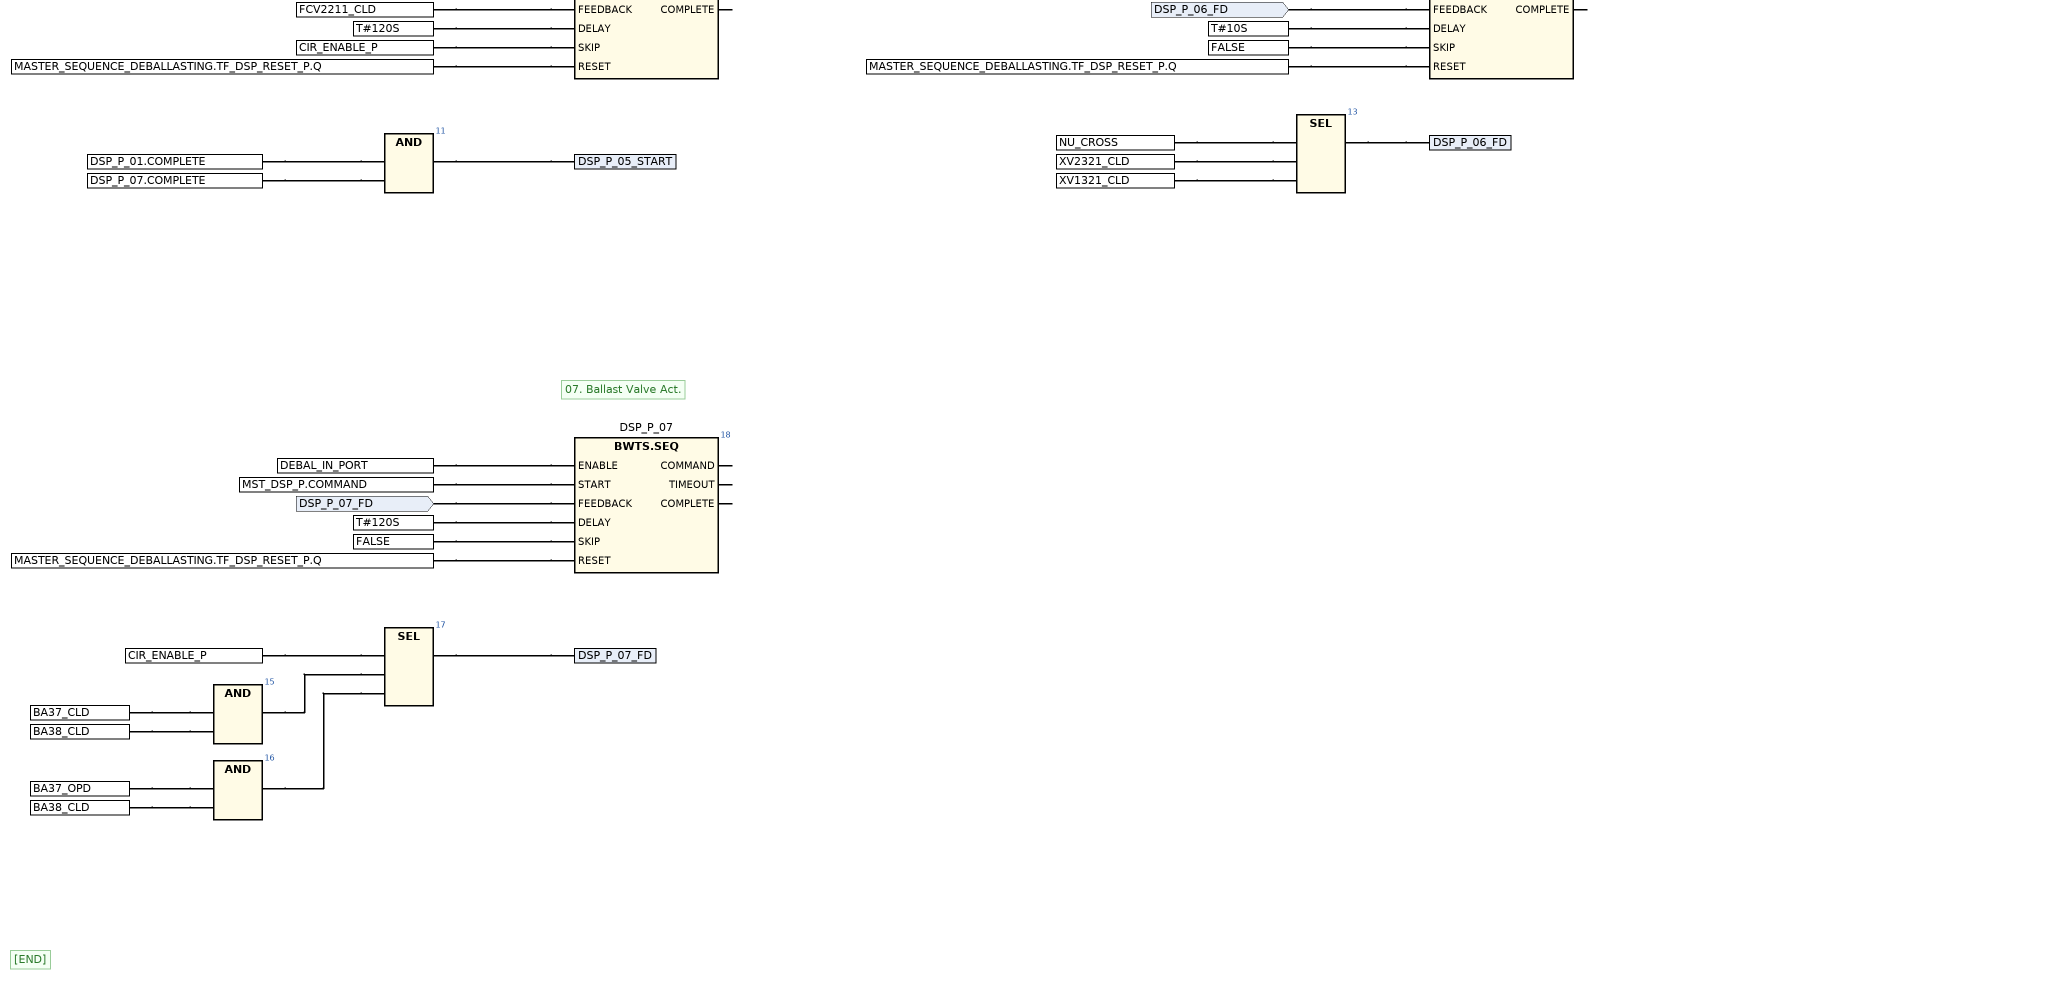
DST_S_ON := DEBAL_IN_STBD AND NOT MST_DSP_S.COMMAND;
(* DSP_P_01.COMPLETE AND DSP_P_07.COMPLETE; result not used *)
(* SEL(NU_CROSS, P232_SPD, P132_SPD); result not used *)
// 02. N/U Pump Stop
DSP_P_02(
    ENABLE := DEBAL_IN_PORT,
    START := _w1,
    FEEDBACK := _w2,
    DELAY := T#10S,
    SKIP := FALSE,
    RESET := MASTER_SEQUENCE_DEBALLASTING.TF_DSP_RESET_P.Q); // BWTS.SEQ
// WATING TIME FOR WBP
TON_0(IN := MST_DSP_P.COMMAND, PT := MS_WBP_SP); // TON
// 01. WBP Stop Request
DSP_P_01(
    ENABLE := DEBAL_IN_PORT,
    START := TON_0.Q,
    FEEDBACK := _w3,
    DELAY := T#120S,
    SKIP := CIR_ENABLE_P,
    RESET := MASTER_SEQUENCE_DEBALLASTING.TF_DSP_RESET_P.Q); // BWTS.SEQ
(* SEL(TRO_CROSS, AIT251_SPD AND XV2512_CLD, AIT151_SPD AND XV1512_CLD); result not used *)
// 03. TRO UNIT STOP
DSP_P_03(
    ENABLE := DEBAL_IN_PORT,
    START := MST_DSP_P.COMMAND,
    FEEDBACK := _w4,
    DELAY := T#10S,
    SKIP := _w4,
    RESET := MASTER_SEQUENCE_DEBALLASTING.TF_DSP_RESET_P.Q); // BWTS.SEQ
(* DSP_P_01.COMPLETE AND DSP_P_07.COMPLETE; result not used *)
// 05. TRC Valve Close
DSP_P_05(
    ENABLE := DEBAL_IN_PORT,
    START := _w5,
    FEEDBACK := FCV2211_CLD,
    DELAY := T#120S,
    SKIP := CIR_ENABLE_P,
    RESET := MASTER_SEQUENCE_DEBALLASTING.TF_DSP_RESET_P.Q); // BWTS.SEQ
(* SEL(NU_CROSS, XV2321_CLD, XV1321_CLD); result not used *)
// 06. N/U Inj. Valve Close
DSP_P_06(
    ENABLE := DEBAL_IN_PORT,
    START := DSP_P_02.COMPLETE,
    FEEDBACK := _w6,
    DELAY := T#10S,
    SKIP := FALSE,
    RESET := MASTER_SEQUENCE_DEBALLASTING.TF_DSP_RESET_P.Q); // BWTS.SEQ
// [END]
(* SEL(CIR_ENABLE_P, BA37_CLD AND BA38_CLD, BA37_OPD AND BA38_CLD); result not used *)
// 07. Ballast Valve Act.
DSP_P_07(
    ENABLE := DEBAL_IN_PORT,
    START := MST_DSP_P.COMMAND,
    FEEDBACK := _w7,
    DELAY := T#120S,
    SKIP := FALSE,
    RESET := MASTER_SEQUENCE_DEBALLASTING.TF_DSP_RESET_P.Q); // BWTS.SEQ

END_PROGRAM

// Device/Application/Logic/2.Sequence/SEQ_DEBAL_SP_S
PROGRAM SEQ_DEBAL_SP_S
VAR
	TON_0: TON;
	DST_P_ON: BOOL;
END_VAR
VAR // added by the converter: edge detectors and wires of the graphical bodies
    _w1, _w2, _w3, _w4, _w5, _w6, _w7 : ANY;
END_VAR

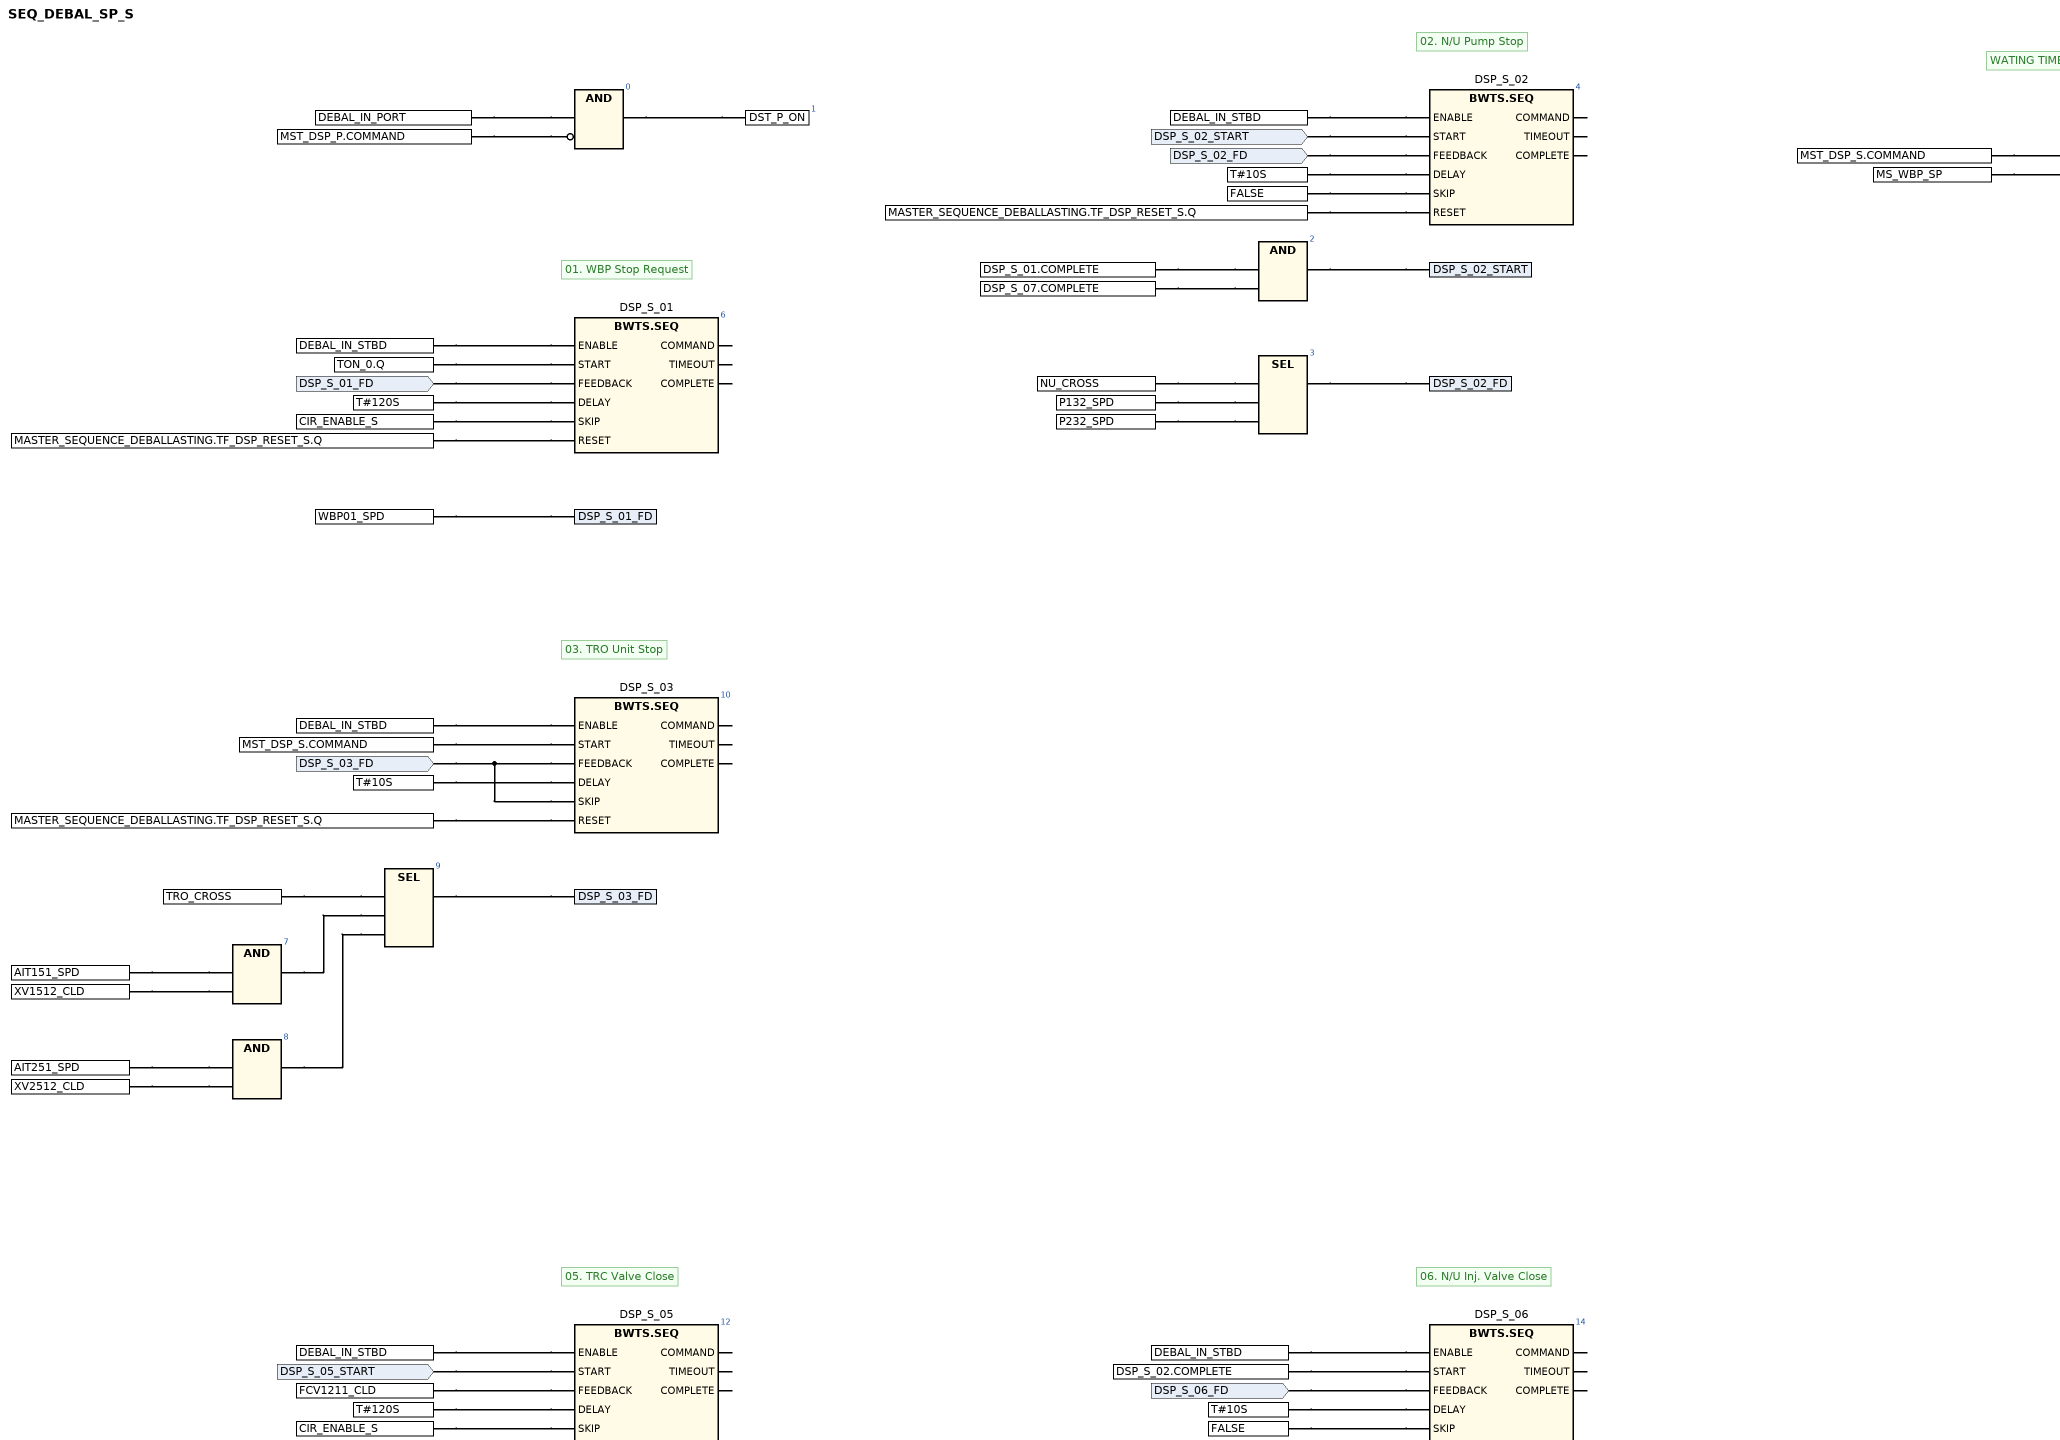
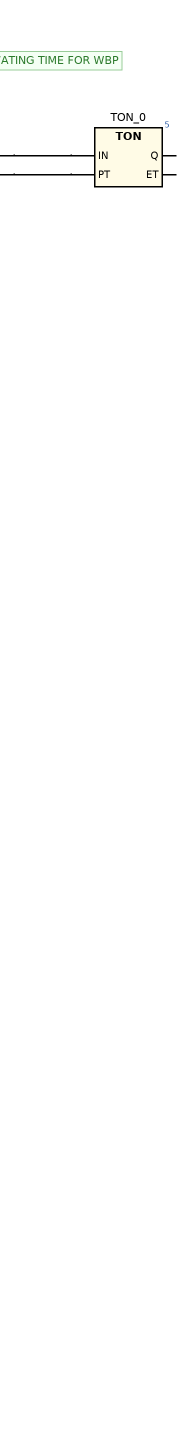
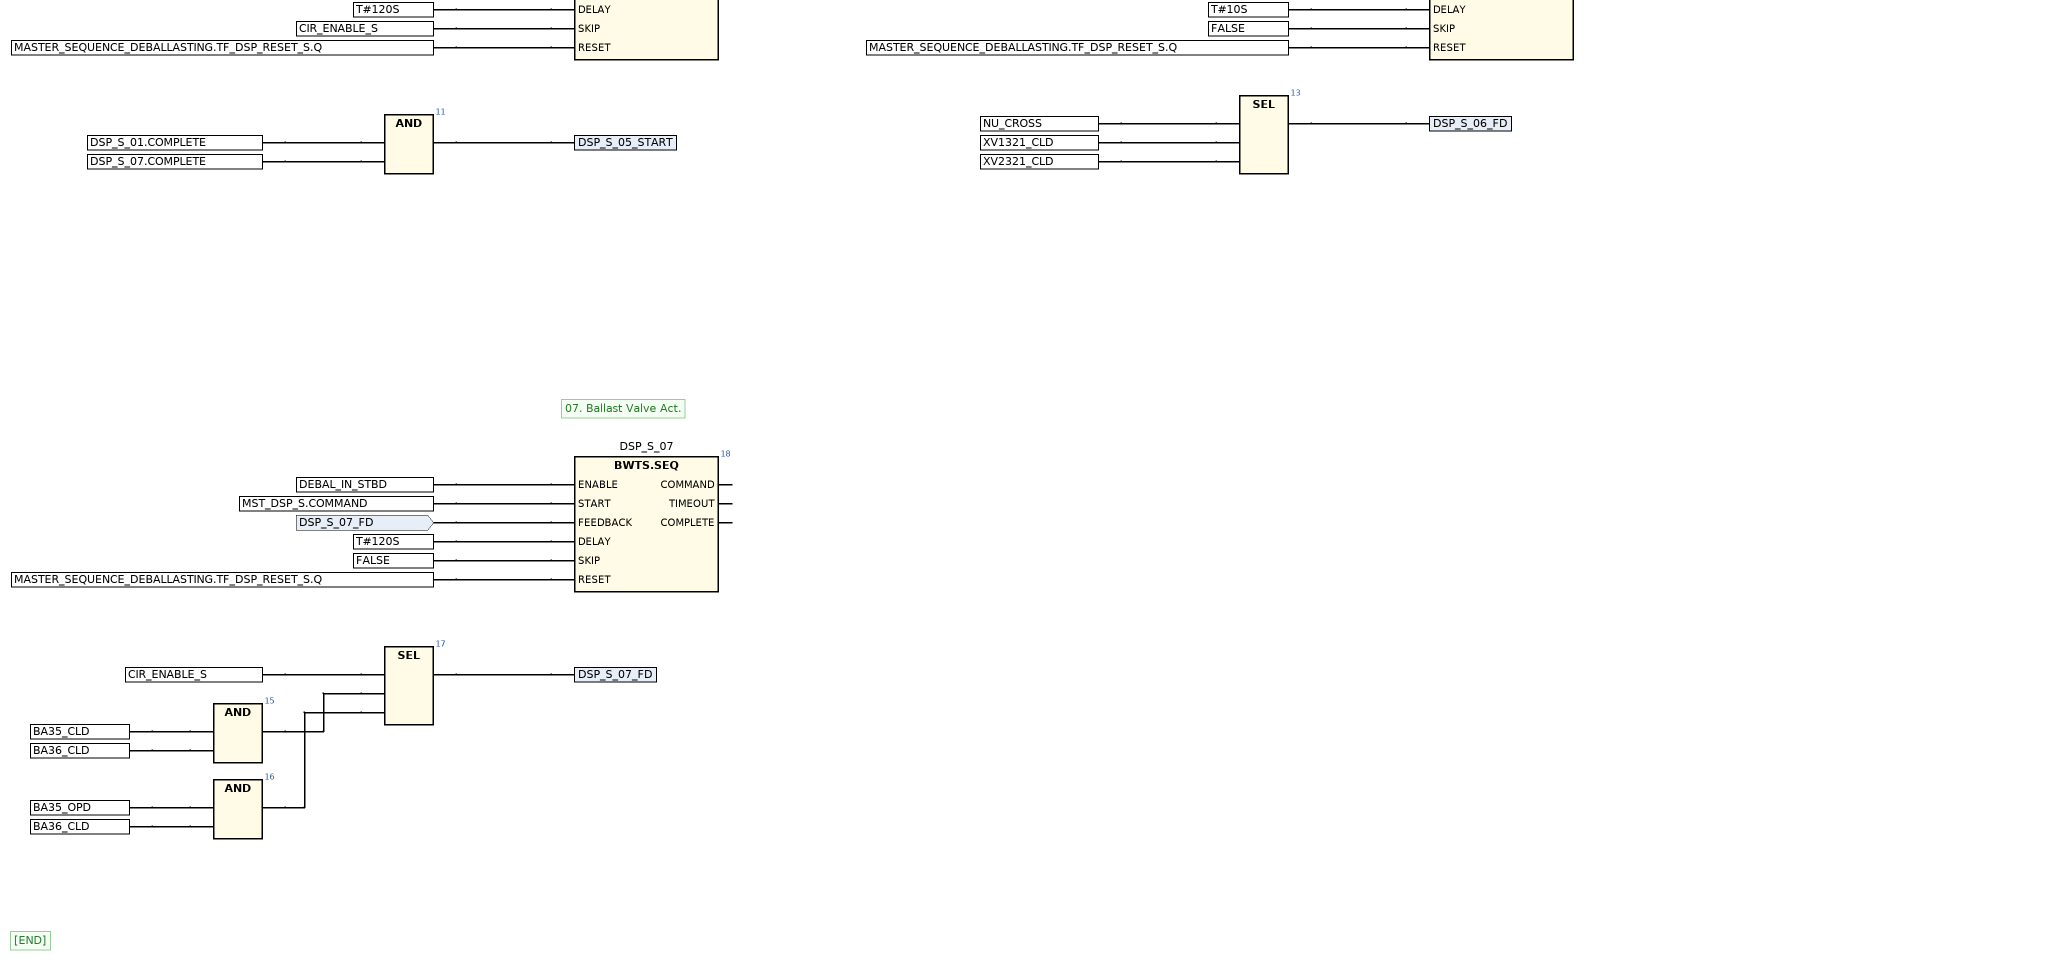
DST_P_ON := DEBAL_IN_PORT AND NOT MST_DSP_P.COMMAND;
(* DSP_S_01.COMPLETE AND DSP_S_07.COMPLETE; result not used *)
(* SEL(NU_CROSS, P132_SPD, P232_SPD); result not used *)
// 02. N/U Pump Stop
DSP_S_02(
    ENABLE := DEBAL_IN_STBD,
    START := _w1,
    FEEDBACK := _w2,
    DELAY := T#10S,
    SKIP := FALSE,
    RESET := MASTER_SEQUENCE_DEBALLASTING.TF_DSP_RESET_S.Q); // BWTS.SEQ
// WATING TIME FOR WBP
TON_0(IN := MST_DSP_S.COMMAND, PT := MS_WBP_SP); // TON
// 01. WBP Stop Request
DSP_S_01(
    ENABLE := DEBAL_IN_STBD,
    START := TON_0.Q,
    FEEDBACK := _w3,
    DELAY := T#120S,
    SKIP := CIR_ENABLE_S,
    RESET := MASTER_SEQUENCE_DEBALLASTING.TF_DSP_RESET_S.Q); // BWTS.SEQ
(* SEL(TRO_CROSS, AIT151_SPD AND XV1512_CLD, AIT251_SPD AND XV2512_CLD); result not used *)
// 03. TRO Unit Stop
DSP_S_03(
    ENABLE := DEBAL_IN_STBD,
    START := MST_DSP_S.COMMAND,
    FEEDBACK := _w4,
    DELAY := T#10S,
    SKIP := _w4,
    RESET := MASTER_SEQUENCE_DEBALLASTING.TF_DSP_RESET_S.Q); // BWTS.SEQ
(* DSP_S_01.COMPLETE AND DSP_S_07.COMPLETE; result not used *)
// 05. TRC Valve Close
DSP_S_05(
    ENABLE := DEBAL_IN_STBD,
    START := _w5,
    FEEDBACK := FCV1211_CLD,
    DELAY := T#120S,
    SKIP := CIR_ENABLE_S,
    RESET := MASTER_SEQUENCE_DEBALLASTING.TF_DSP_RESET_S.Q); // BWTS.SEQ
(* SEL(NU_CROSS, XV1321_CLD, XV2321_CLD); result not used *)
// 06. N/U Inj. Valve Close
DSP_S_06(
    ENABLE := DEBAL_IN_STBD,
    START := DSP_S_02.COMPLETE,
    FEEDBACK := _w6,
    DELAY := T#10S,
    SKIP := FALSE,
    RESET := MASTER_SEQUENCE_DEBALLASTING.TF_DSP_RESET_S.Q); // BWTS.SEQ
// [END]
(* SEL(CIR_ENABLE_S, BA35_CLD AND BA36_CLD, BA35_OPD AND BA36_CLD); result not used *)
// 07. Ballast Valve Act.
DSP_S_07(
    ENABLE := DEBAL_IN_STBD,
    START := MST_DSP_S.COMMAND,
    FEEDBACK := _w7,
    DELAY := T#120S,
    SKIP := FALSE,
    RESET := MASTER_SEQUENCE_DEBALLASTING.TF_DSP_RESET_S.Q); // BWTS.SEQ

END_PROGRAM

// Device/Application/Logic/2.Sequence/SEQ_DEBAL_ST_P
PROGRAM SEQ_DEBAL_ST_P
VAR
	TON_0: TON; //N.A PUMP PRE RUNNING TIME
	TON_2: TON; //TRO SENSOR WAITING TIME
	TON_3: TON;	//RECIRCULATION TIME
END_VAR
VAR // added by the converter: edge detectors and wires of the graphical bodies
    _w1, _w2, _w3, _w4, _w5, _w6, _w7 : ANY;
END_VAR

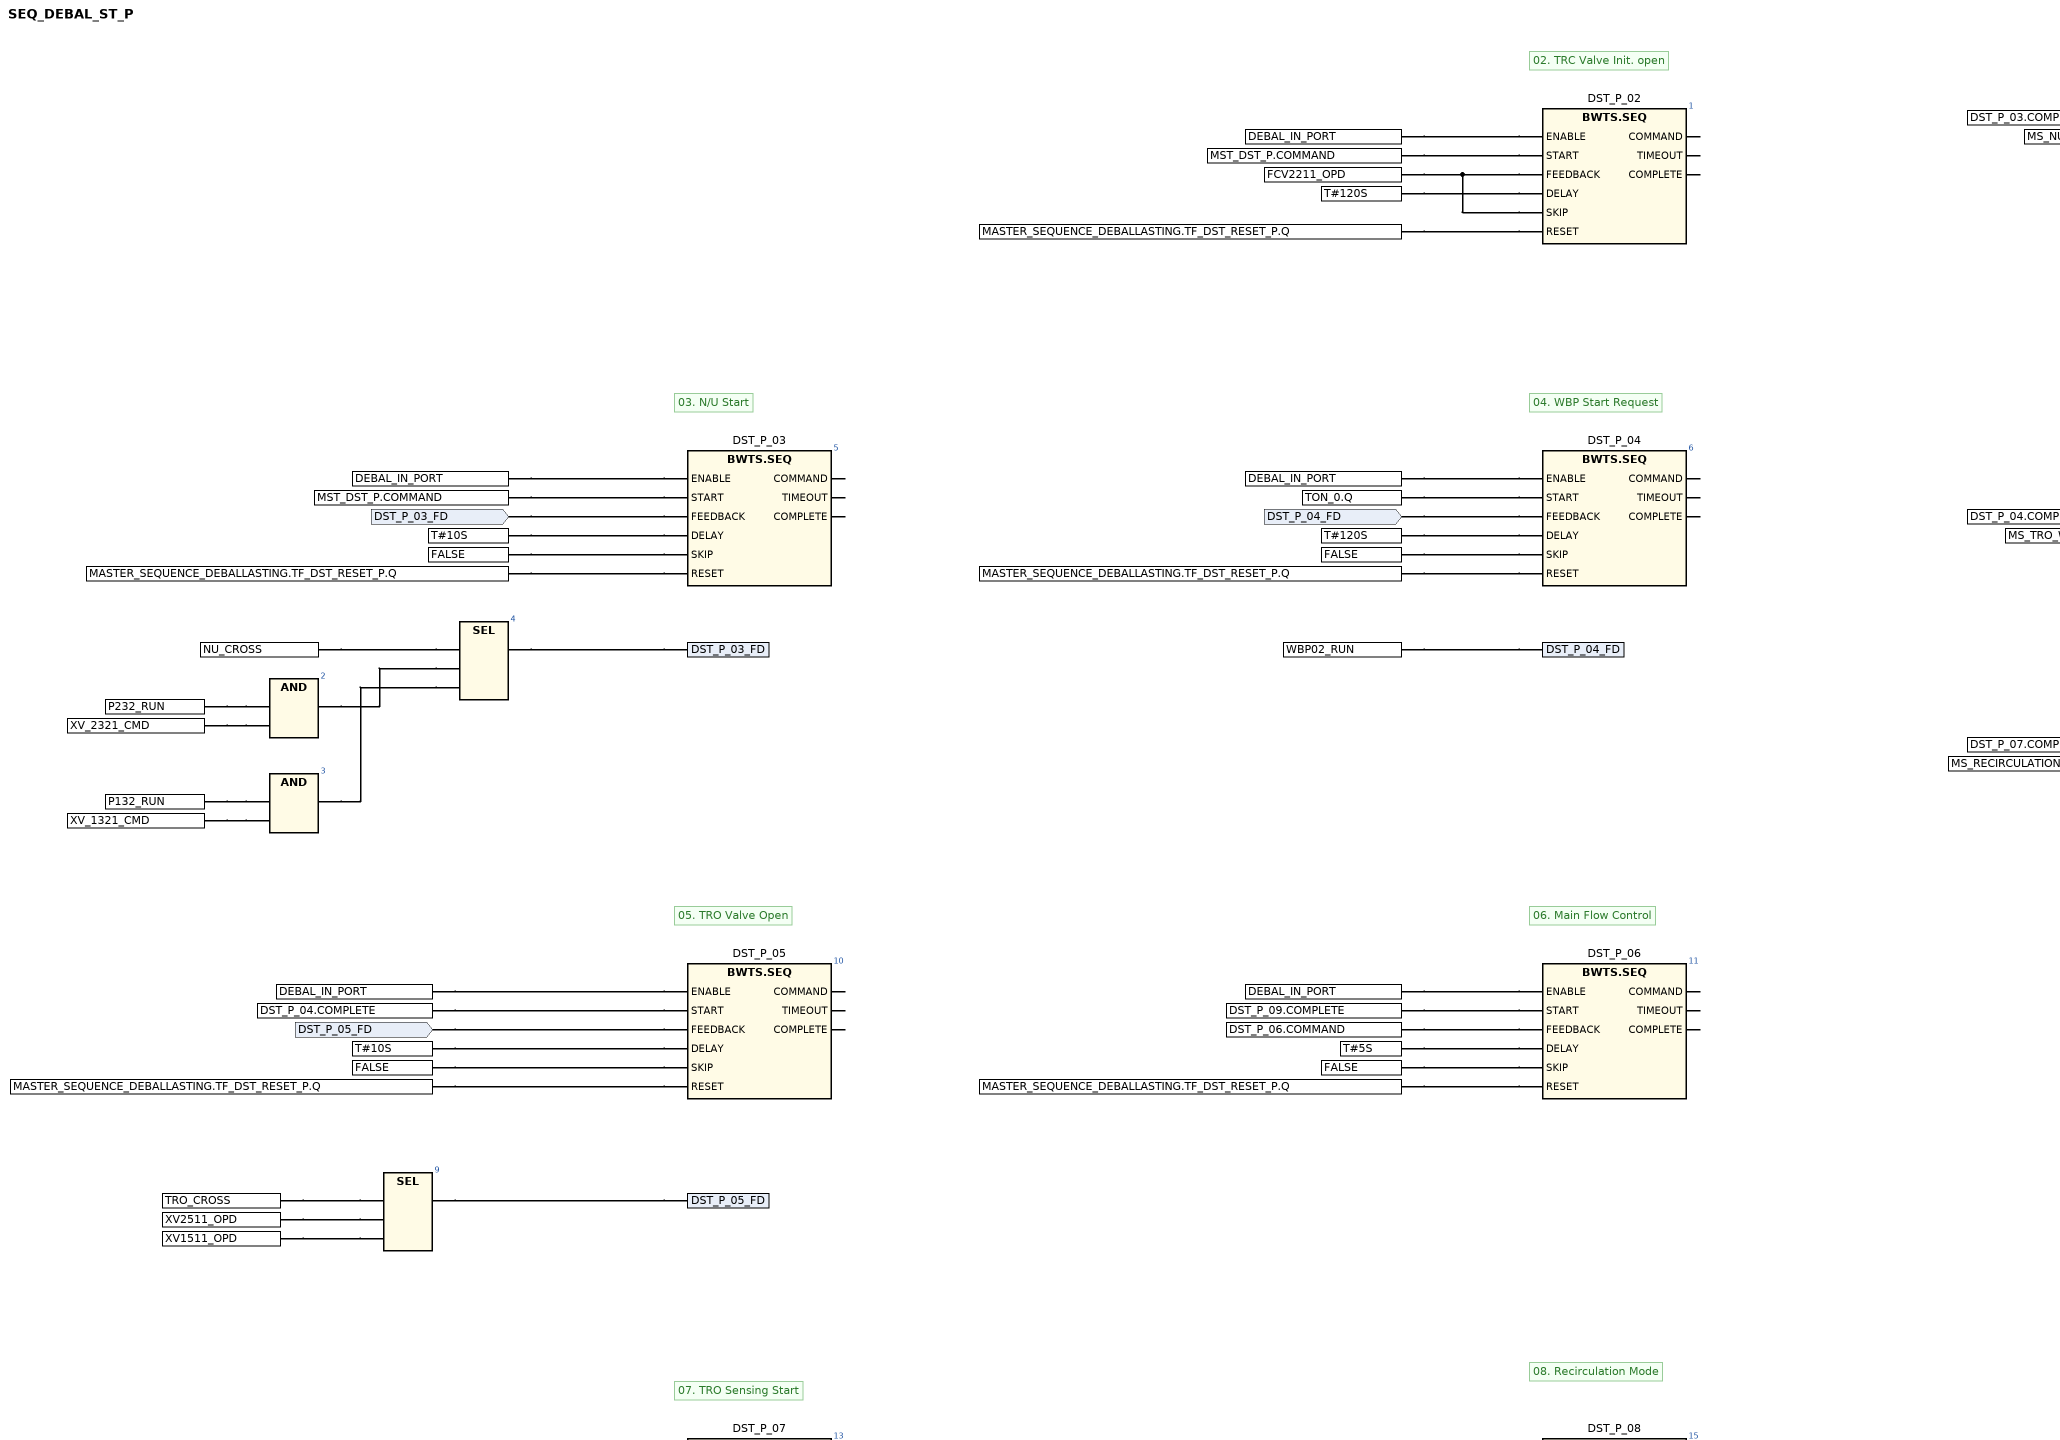
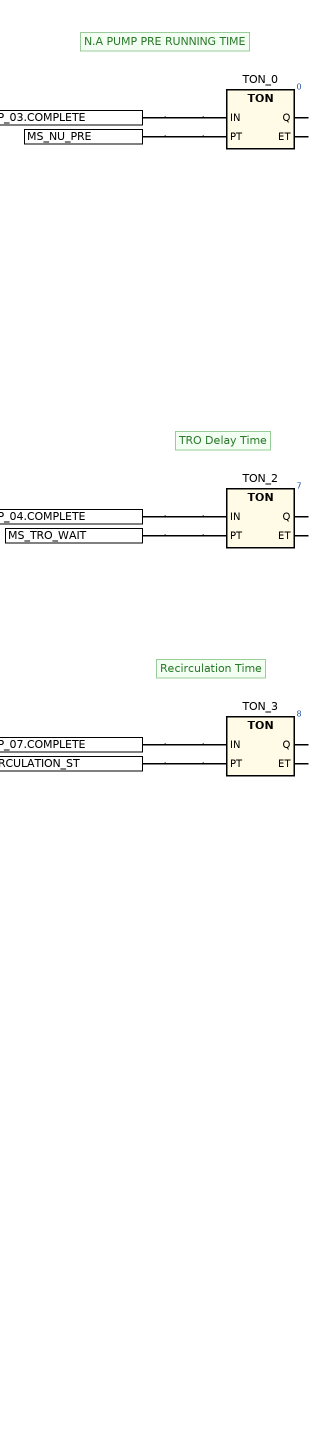
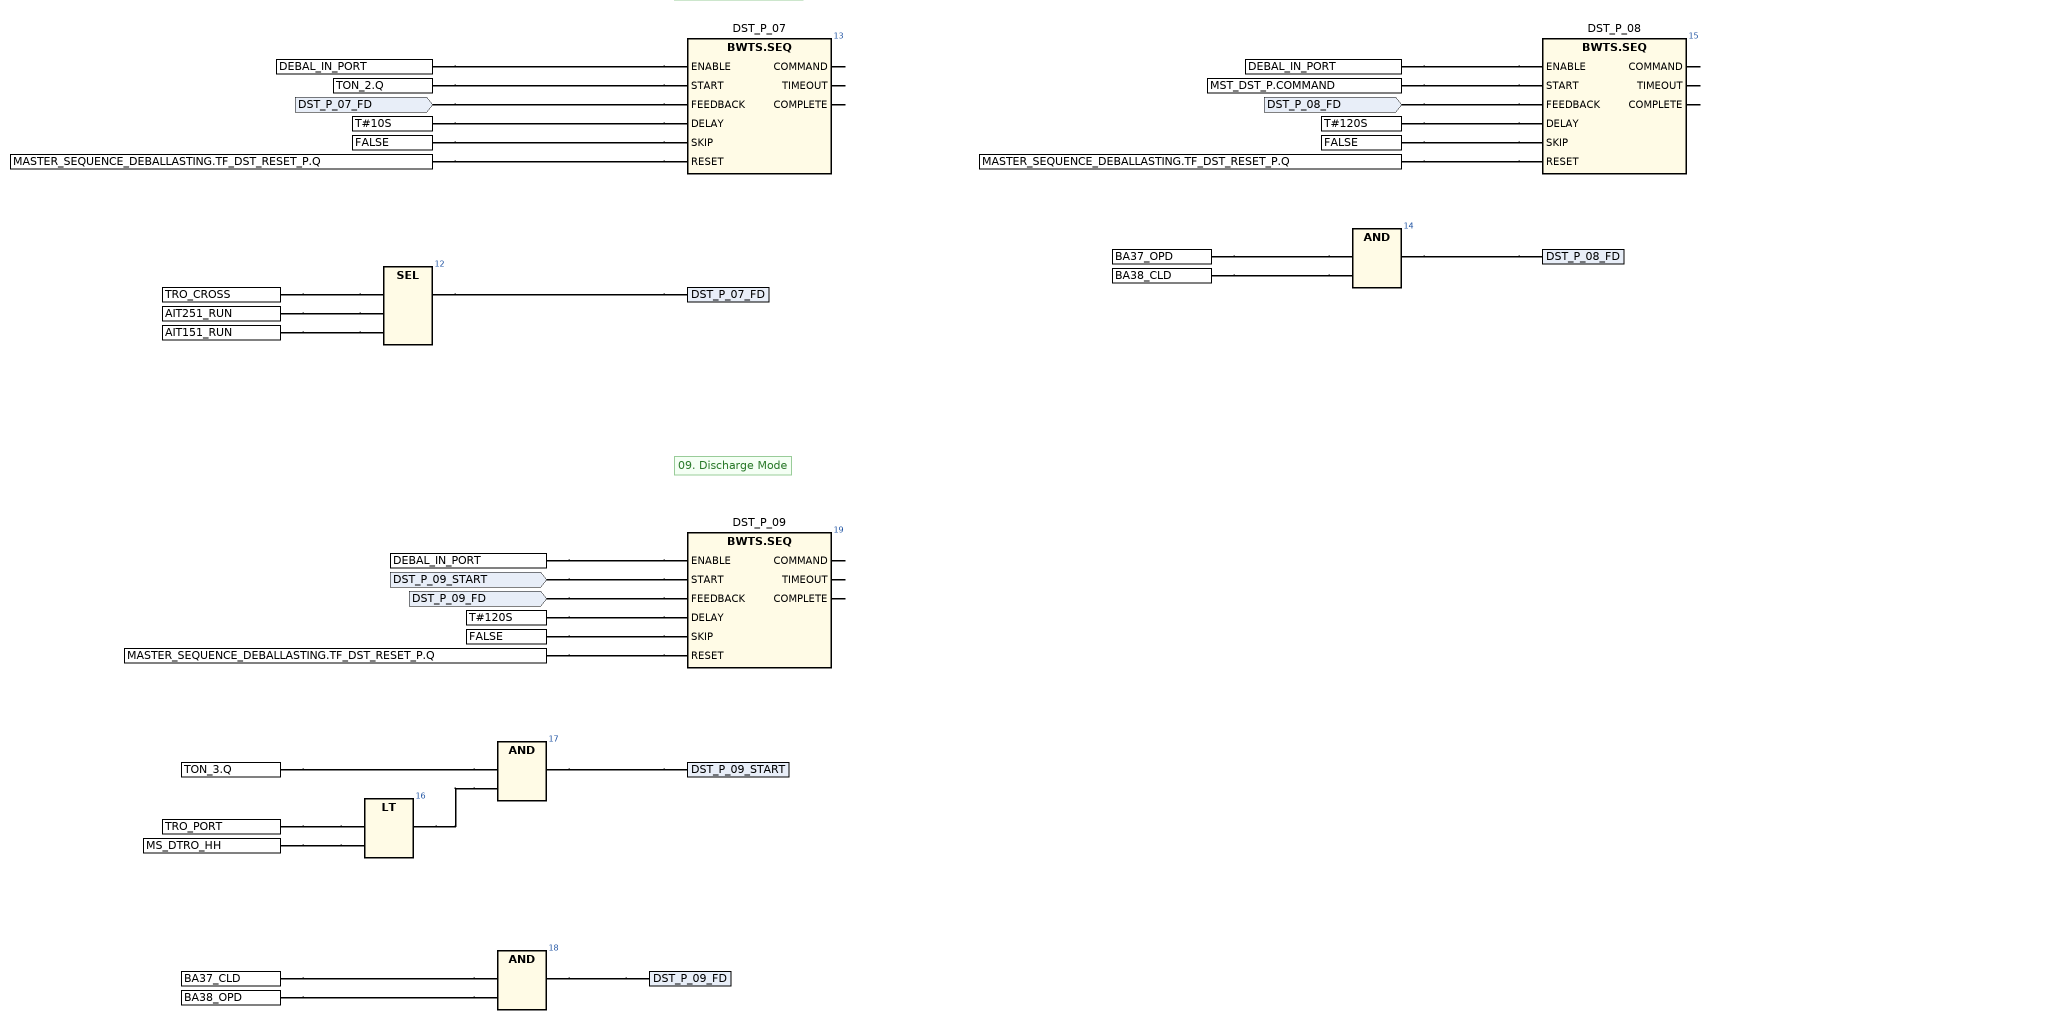
// N.A PUMP PRE RUNNING TIME
TON_0(IN := DST_P_03.COMPLETE, PT := MS_NU_PRE); // TON
// 02. TRC Valve Init. open
DST_P_02(
    ENABLE := DEBAL_IN_PORT,
    START := MST_DST_P.COMMAND,
    FEEDBACK := FCV2211_OPD,
    DELAY := T#120S,
    SKIP := FCV2211_OPD,
    RESET := MASTER_SEQUENCE_DEBALLASTING.TF_DST_RESET_P.Q); // BWTS.SEQ
(* SEL(NU_CROSS, P232_RUN AND XV_2321_CMD, P132_RUN AND XV_1321_CMD); result not used *)
// 03. N/U Start
DST_P_03(
    ENABLE := DEBAL_IN_PORT,
    START := MST_DST_P.COMMAND,
    FEEDBACK := _w1,
    DELAY := T#10S,
    SKIP := FALSE,
    RESET := MASTER_SEQUENCE_DEBALLASTING.TF_DST_RESET_P.Q); // BWTS.SEQ
// 04. WBP Start Request
DST_P_04(
    ENABLE := DEBAL_IN_PORT,
    START := TON_0.Q,
    FEEDBACK := _w2,
    DELAY := T#120S,
    SKIP := FALSE,
    RESET := MASTER_SEQUENCE_DEBALLASTING.TF_DST_RESET_P.Q); // BWTS.SEQ
// TRO Delay Time
TON_2(IN := DST_P_04.COMPLETE, PT := MS_TRO_WAIT); // TON
// Recirculation Time
TON_3(IN := DST_P_07.COMPLETE, PT := MS_RECIRCULATION_ST); // TON
(* SEL(TRO_CROSS, XV2511_OPD, XV1511_OPD); result not used *)
// 05. TRO Valve Open
DST_P_05(
    ENABLE := DEBAL_IN_PORT,
    START := DST_P_04.COMPLETE,
    FEEDBACK := _w3,
    DELAY := T#10S,
    SKIP := FALSE,
    RESET := MASTER_SEQUENCE_DEBALLASTING.TF_DST_RESET_P.Q); // BWTS.SEQ
// 06. Main Flow Control
DST_P_06(
    ENABLE := DEBAL_IN_PORT,
    START := DST_P_09.COMPLETE,
    FEEDBACK := DST_P_06.COMMAND,
    DELAY := T#5S,
    SKIP := FALSE,
    RESET := MASTER_SEQUENCE_DEBALLASTING.TF_DST_RESET_P.Q); // BWTS.SEQ
(* SEL(TRO_CROSS, AIT251_RUN, AIT151_RUN); result not used *)
// 07. TRO Sensing Start
DST_P_07(
    ENABLE := DEBAL_IN_PORT,
    START := TON_2.Q,
    FEEDBACK := _w4,
    DELAY := T#10S,
    SKIP := FALSE,
    RESET := MASTER_SEQUENCE_DEBALLASTING.TF_DST_RESET_P.Q); // BWTS.SEQ
(* BA37_OPD AND BA38_CLD; result not used *)
// 08. Recirculation Mode
DST_P_08(
    ENABLE := DEBAL_IN_PORT,
    START := MST_DST_P.COMMAND,
    FEEDBACK := _w5,
    DELAY := T#120S,
    SKIP := FALSE,
    RESET := MASTER_SEQUENCE_DEBALLASTING.TF_DST_RESET_P.Q); // BWTS.SEQ
(* TON_3.Q AND TRO_PORT < MS_DTRO_HH; result not used *)
(* BA37_CLD AND BA38_OPD; result not used *)
// 09. Discharge Mode
DST_P_09(
    ENABLE := DEBAL_IN_PORT,
    START := _w6,
    FEEDBACK := _w7,
    DELAY := T#120S,
    SKIP := FALSE,
    RESET := MASTER_SEQUENCE_DEBALLASTING.TF_DST_RESET_P.Q); // BWTS.SEQ

END_PROGRAM

// Device/Application/Logic/2.Sequence/SEQ_DEBAL_ST_S
 PROGRAM SEQ_DEBAL_ST_S
VAR
	TON_0: TON; //N.A PUMP PRE RUNNING TIME
	TON_2: TON; //TRO SENSOR WAITING TIME
	TON_3: TON;
END_VAR
VAR // added by the converter: edge detectors and wires of the graphical bodies
    _w1, _w2, _w3, _w4, _w5, _w6, _w7 : ANY;
END_VAR

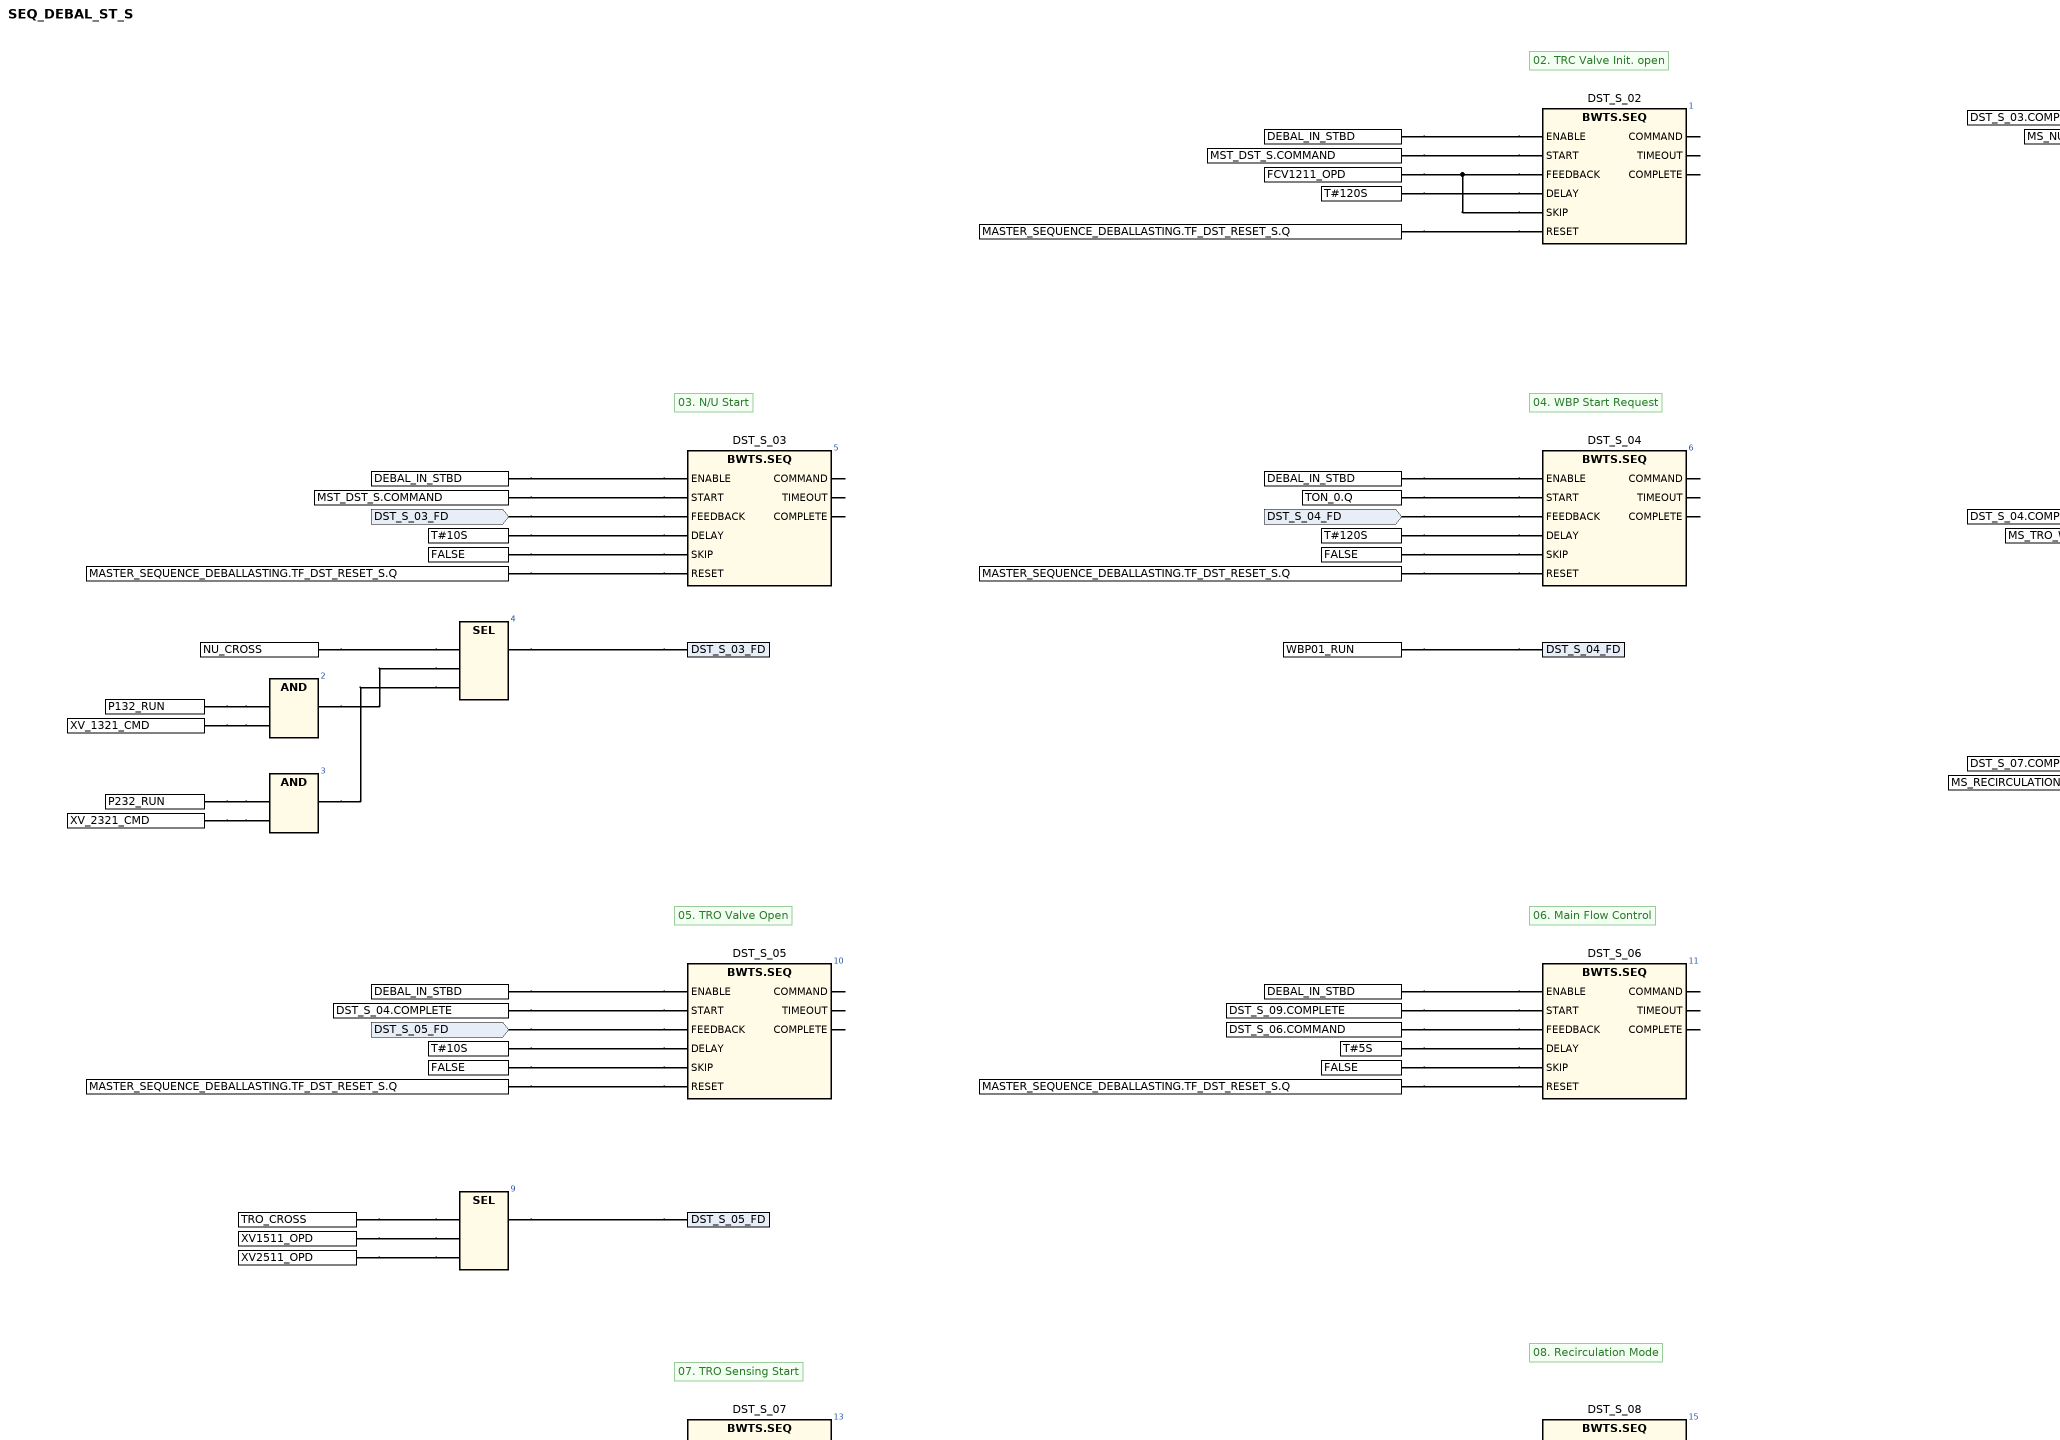
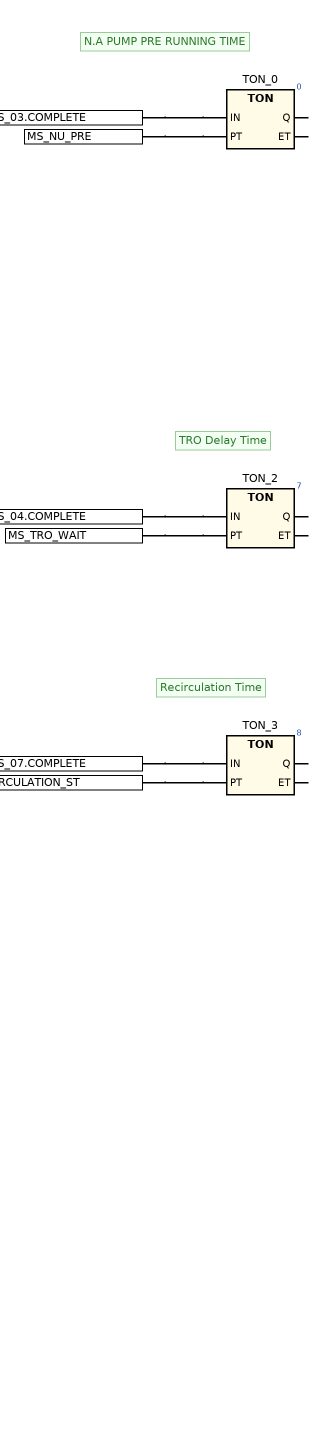
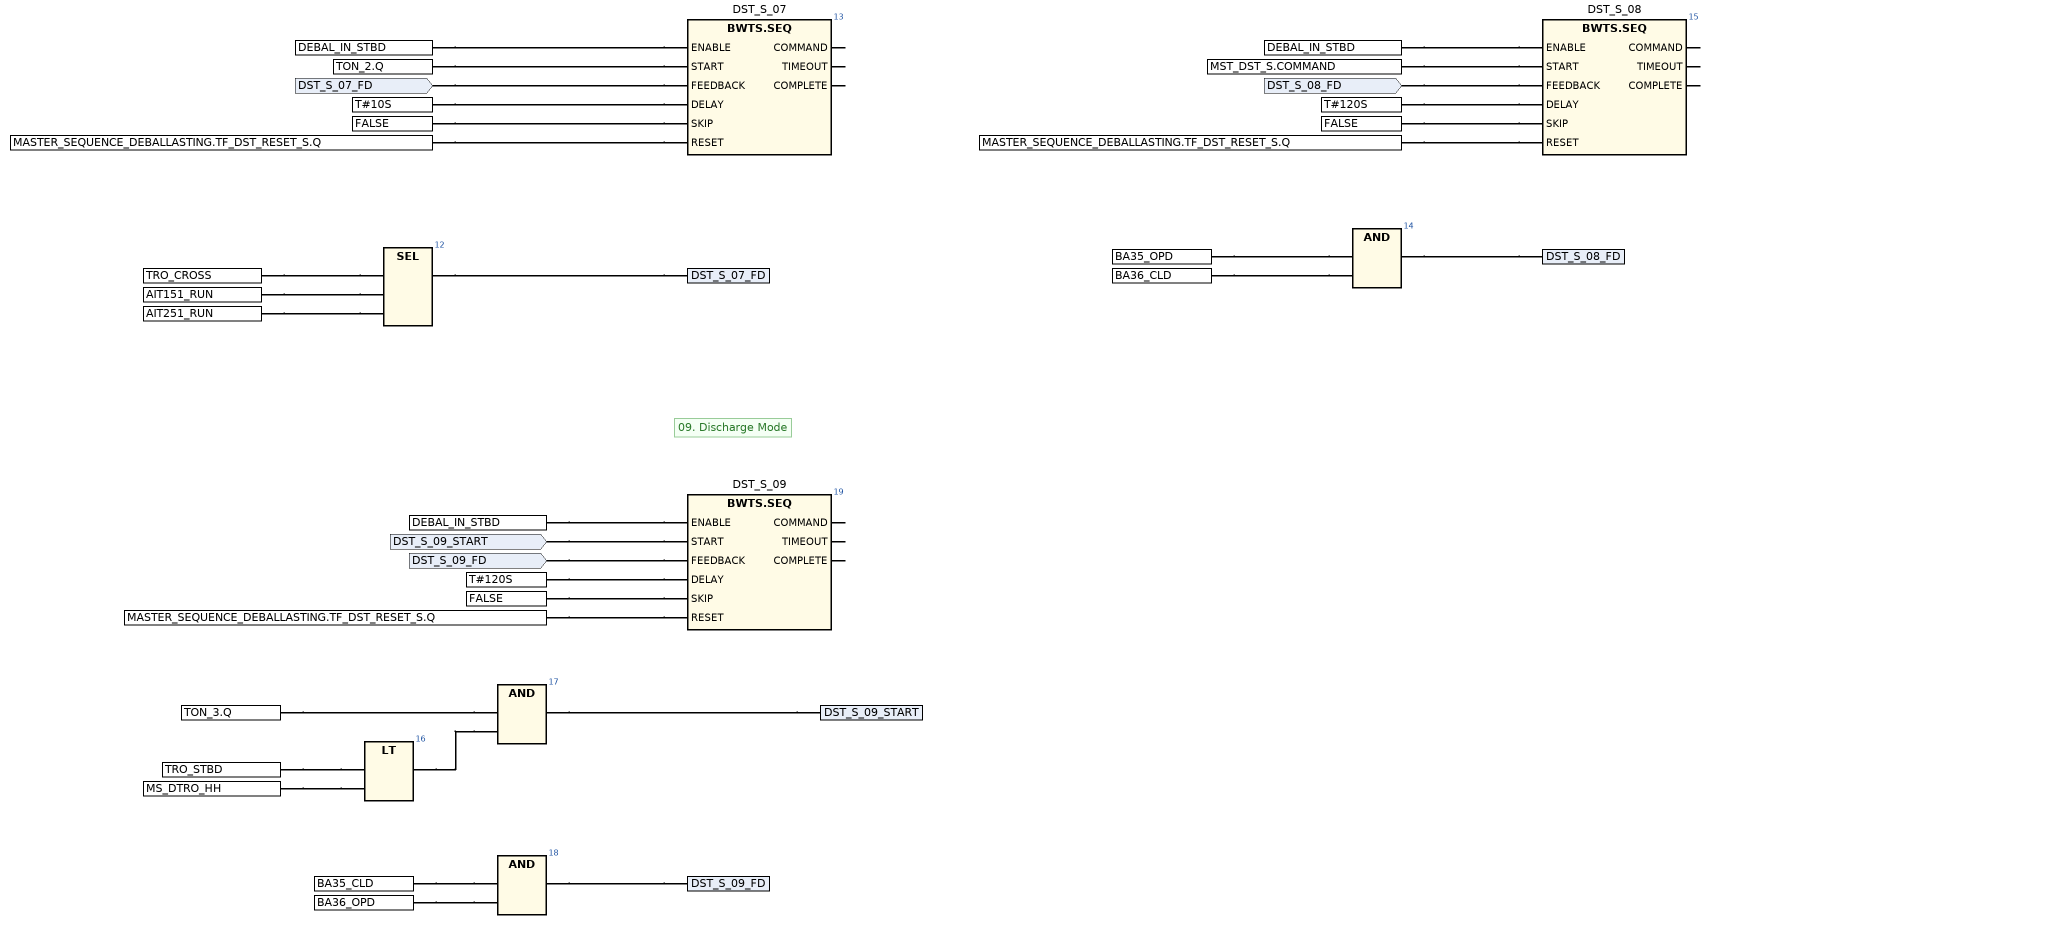
// N.A PUMP PRE RUNNING TIME
TON_0(IN := DST_S_03.COMPLETE, PT := MS_NU_PRE); // TON
// 02. TRC Valve Init. open
DST_S_02(
    ENABLE := DEBAL_IN_STBD,
    START := MST_DST_S.COMMAND,
    FEEDBACK := FCV1211_OPD,
    DELAY := T#120S,
    SKIP := FCV1211_OPD,
    RESET := MASTER_SEQUENCE_DEBALLASTING.TF_DST_RESET_S.Q); // BWTS.SEQ
(* SEL(NU_CROSS, P132_RUN AND XV_1321_CMD, P232_RUN AND XV_2321_CMD); result not used *)
// 03. N/U Start
DST_S_03(
    ENABLE := DEBAL_IN_STBD,
    START := MST_DST_S.COMMAND,
    FEEDBACK := _w1,
    DELAY := T#10S,
    SKIP := FALSE,
    RESET := MASTER_SEQUENCE_DEBALLASTING.TF_DST_RESET_S.Q); // BWTS.SEQ
// 04. WBP Start Request
DST_S_04(
    ENABLE := DEBAL_IN_STBD,
    START := TON_0.Q,
    FEEDBACK := _w2,
    DELAY := T#120S,
    SKIP := FALSE,
    RESET := MASTER_SEQUENCE_DEBALLASTING.TF_DST_RESET_S.Q); // BWTS.SEQ
// TRO Delay Time
TON_2(IN := DST_S_04.COMPLETE, PT := MS_TRO_WAIT); // TON
// Recirculation Time
TON_3(IN := DST_S_07.COMPLETE, PT := MS_RECIRCULATION_ST); // TON
(* SEL(TRO_CROSS, XV1511_OPD, XV2511_OPD); result not used *)
// 05. TRO Valve Open
DST_S_05(
    ENABLE := DEBAL_IN_STBD,
    START := DST_S_04.COMPLETE,
    FEEDBACK := _w3,
    DELAY := T#10S,
    SKIP := FALSE,
    RESET := MASTER_SEQUENCE_DEBALLASTING.TF_DST_RESET_S.Q); // BWTS.SEQ
// 06. Main Flow Control
DST_S_06(
    ENABLE := DEBAL_IN_STBD,
    START := DST_S_09.COMPLETE,
    FEEDBACK := DST_S_06.COMMAND,
    DELAY := T#5S,
    SKIP := FALSE,
    RESET := MASTER_SEQUENCE_DEBALLASTING.TF_DST_RESET_S.Q); // BWTS.SEQ
(* SEL(TRO_CROSS, AIT151_RUN, AIT251_RUN); result not used *)
// 07. TRO Sensing Start
DST_S_07(
    ENABLE := DEBAL_IN_STBD,
    START := TON_2.Q,
    FEEDBACK := _w4,
    DELAY := T#10S,
    SKIP := FALSE,
    RESET := MASTER_SEQUENCE_DEBALLASTING.TF_DST_RESET_S.Q); // BWTS.SEQ
(* BA35_OPD AND BA36_CLD; result not used *)
// 08. Recirculation Mode
DST_S_08(
    ENABLE := DEBAL_IN_STBD,
    START := MST_DST_S.COMMAND,
    FEEDBACK := _w5,
    DELAY := T#120S,
    SKIP := FALSE,
    RESET := MASTER_SEQUENCE_DEBALLASTING.TF_DST_RESET_S.Q); // BWTS.SEQ
(* TON_3.Q AND TRO_STBD < MS_DTRO_HH; result not used *)
(* BA35_CLD AND BA36_OPD; result not used *)
// 09. Discharge Mode
DST_S_09(
    ENABLE := DEBAL_IN_STBD,
    START := _w6,
    FEEDBACK := _w7,
    DELAY := T#120S,
    SKIP := FALSE,
    RESET := MASTER_SEQUENCE_DEBALLASTING.TF_DST_RESET_S.Q); // BWTS.SEQ

END_PROGRAM

// Device/Application/Logic/2.Sequence/SEQ_STRIP_SP
PROGRAM SEQ_STRIP_SP
VAR
	TON_0: TON; //N.A PUMP PRE RUNNING TIME
END_VAR
VAR // added by the converter: edge detectors and wires of the graphical bodies
    _w1, _w2, _w3, _w4, _w5 : ANY;
END_VAR

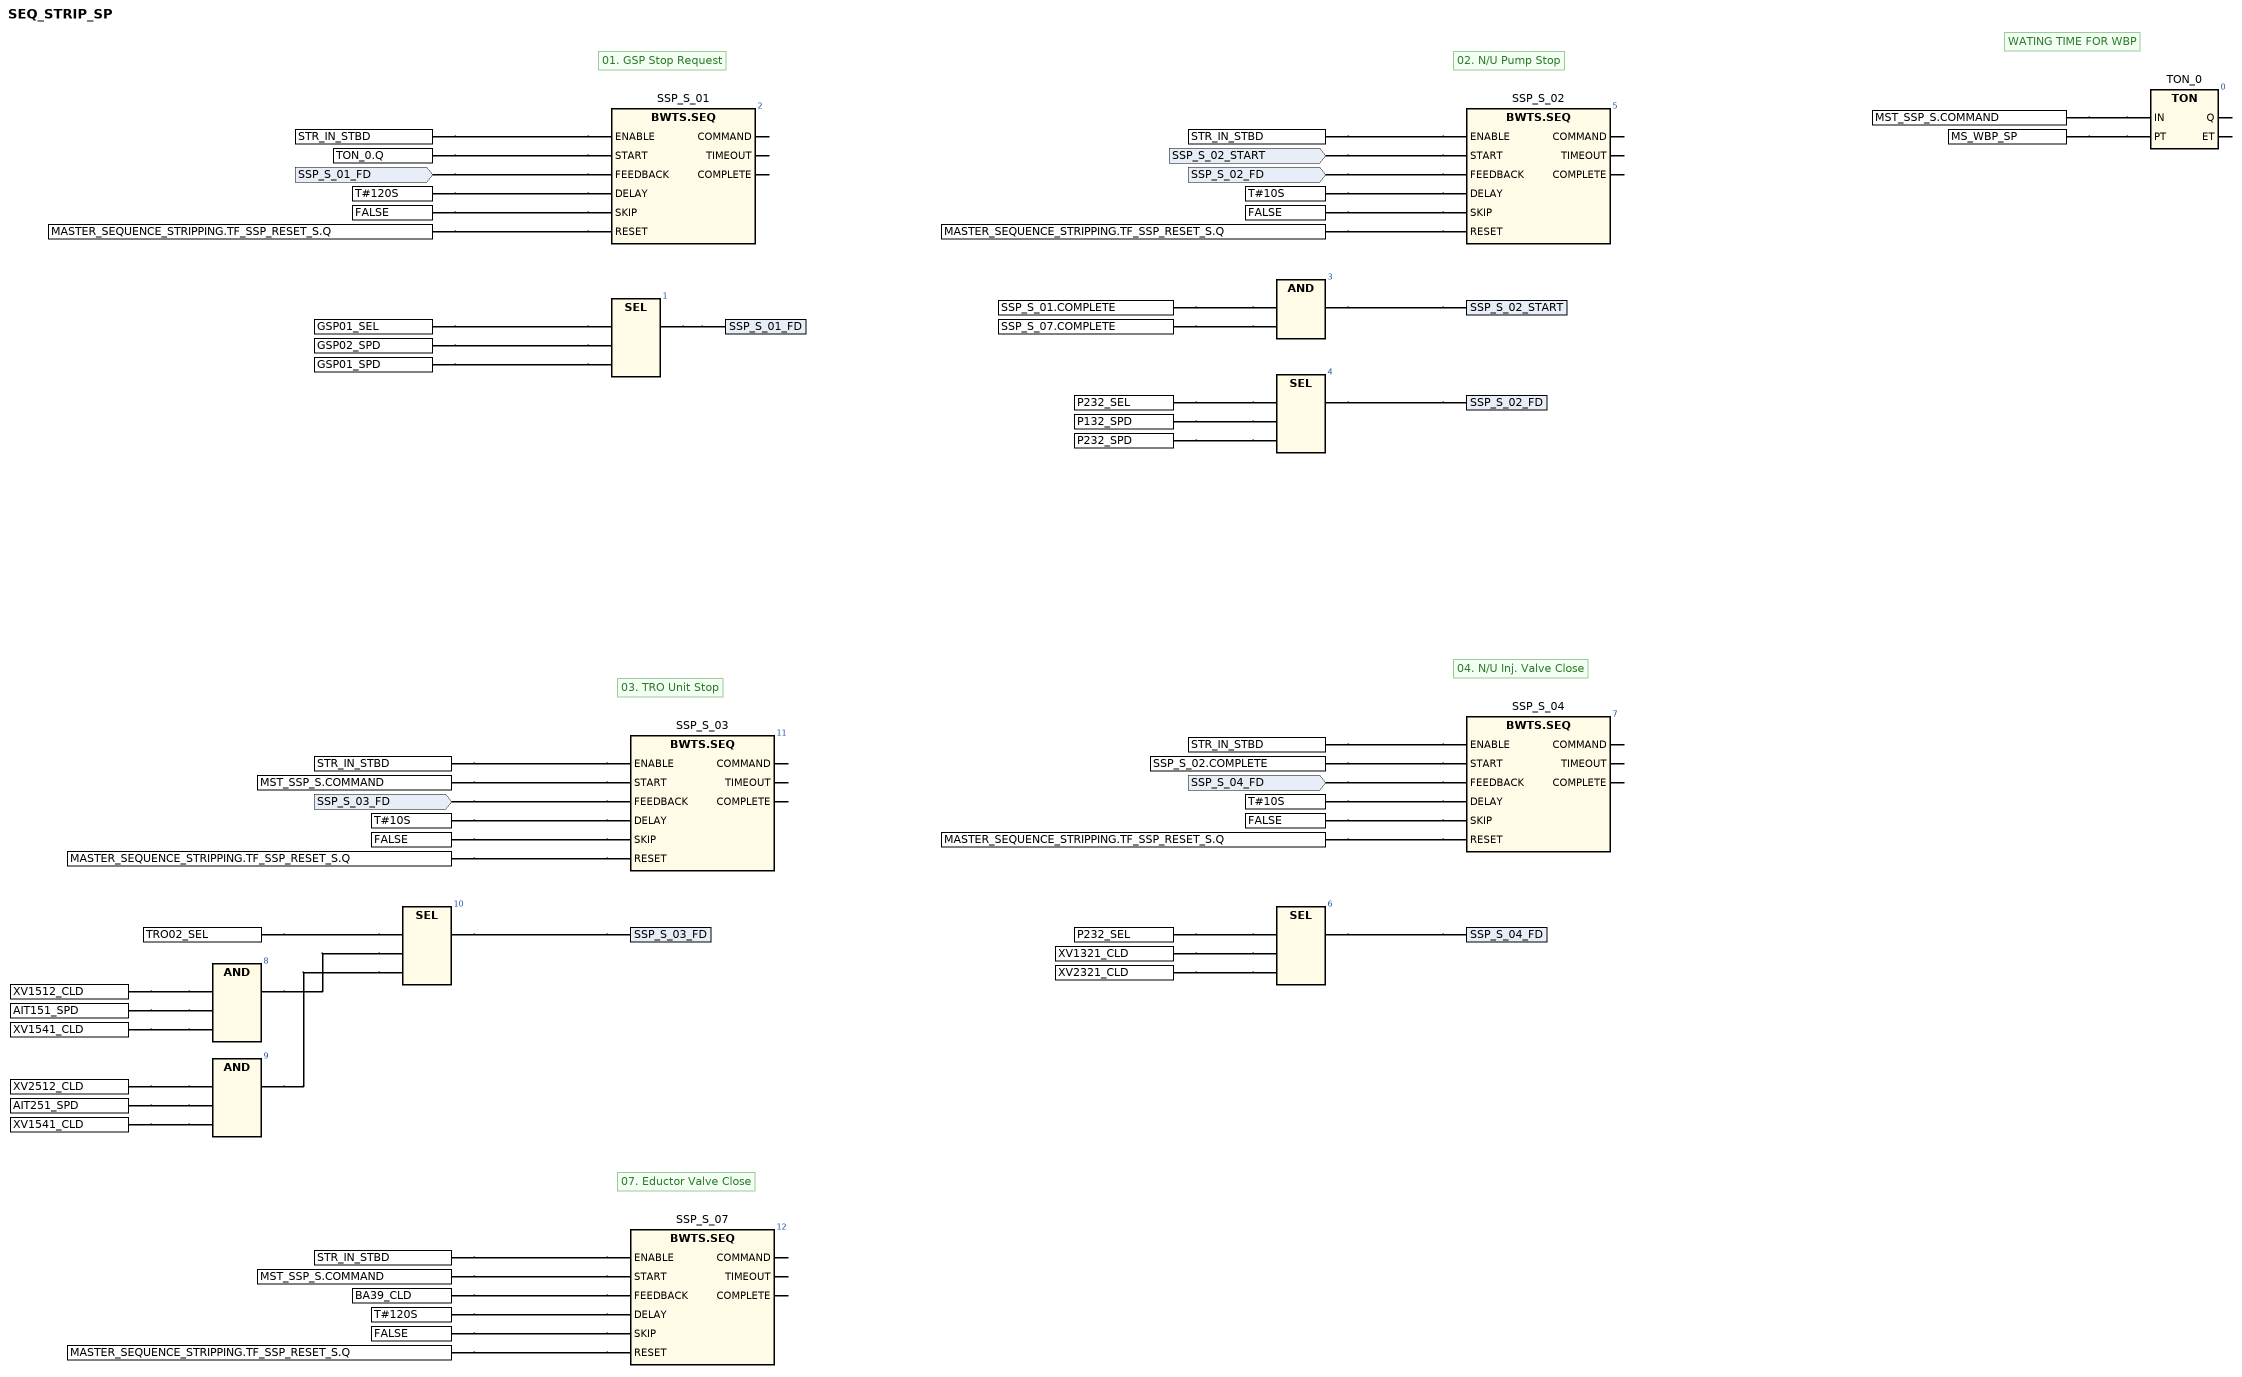
// WATING TIME FOR WBP
TON_0(IN := MST_SSP_S.COMMAND, PT := MS_WBP_SP); // TON
(* SEL(GSP01_SEL, GSP02_SPD, GSP01_SPD); result not used *)
// 01. GSP Stop Request
SSP_S_01(
    ENABLE := STR_IN_STBD,
    START := TON_0.Q,
    FEEDBACK := _w1,
    DELAY := T#120S,
    SKIP := FALSE,
    RESET := MASTER_SEQUENCE_STRIPPING.TF_SSP_RESET_S.Q); // BWTS.SEQ
(* SSP_S_01.COMPLETE AND SSP_S_07.COMPLETE; result not used *)
(* SEL(P232_SEL, P132_SPD, P232_SPD); result not used *)
// 02. N/U Pump Stop
SSP_S_02(
    ENABLE := STR_IN_STBD,
    START := _w2,
    FEEDBACK := _w3,
    DELAY := T#10S,
    SKIP := FALSE,
    RESET := MASTER_SEQUENCE_STRIPPING.TF_SSP_RESET_S.Q); // BWTS.SEQ
(* SEL(P232_SEL, XV1321_CLD, XV2321_CLD); result not used *)
// 04. N/U Inj. Valve Close
SSP_S_04(
    ENABLE := STR_IN_STBD,
    START := SSP_S_02.COMPLETE,
    FEEDBACK := _w4,
    DELAY := T#10S,
    SKIP := FALSE,
    RESET := MASTER_SEQUENCE_STRIPPING.TF_SSP_RESET_S.Q); // BWTS.SEQ
(* SEL(TRO02_SEL, XV1512_CLD AND AIT151_SPD AND XV1541_CLD, XV2512_CLD AND AIT251_SPD AND XV1541_CLD); result not used *)
// 03. TRO Unit Stop
SSP_S_03(
    ENABLE := STR_IN_STBD,
    START := MST_SSP_S.COMMAND,
    FEEDBACK := _w5,
    DELAY := T#10S,
    SKIP := FALSE,
    RESET := MASTER_SEQUENCE_STRIPPING.TF_SSP_RESET_S.Q); // BWTS.SEQ
// 07. Eductor Valve Close
SSP_S_07(
    ENABLE := STR_IN_STBD,
    START := MST_SSP_S.COMMAND,
    FEEDBACK := BA39_CLD,
    DELAY := T#120S,
    SKIP := FALSE,
    RESET := MASTER_SEQUENCE_STRIPPING.TF_SSP_RESET_S.Q); // BWTS.SEQ

END_PROGRAM

// Device/Application/Logic/2.Sequence/SEQ_STRIP_ST
PROGRAM SEQ_STRIP_ST
VAR
	TON_0: TON; //N.A PUMP PRE RUNNING TIME
	TON_1: TON; //TRO Sampling pipe filling time
	TON_2: TON; //TRO SENSOR WAITING TIME
END_VAR
VAR // added by the converter: edge detectors and wires of the graphical bodies
    _w1, _w2, _w3, _w4, _w5 : ANY;
END_VAR

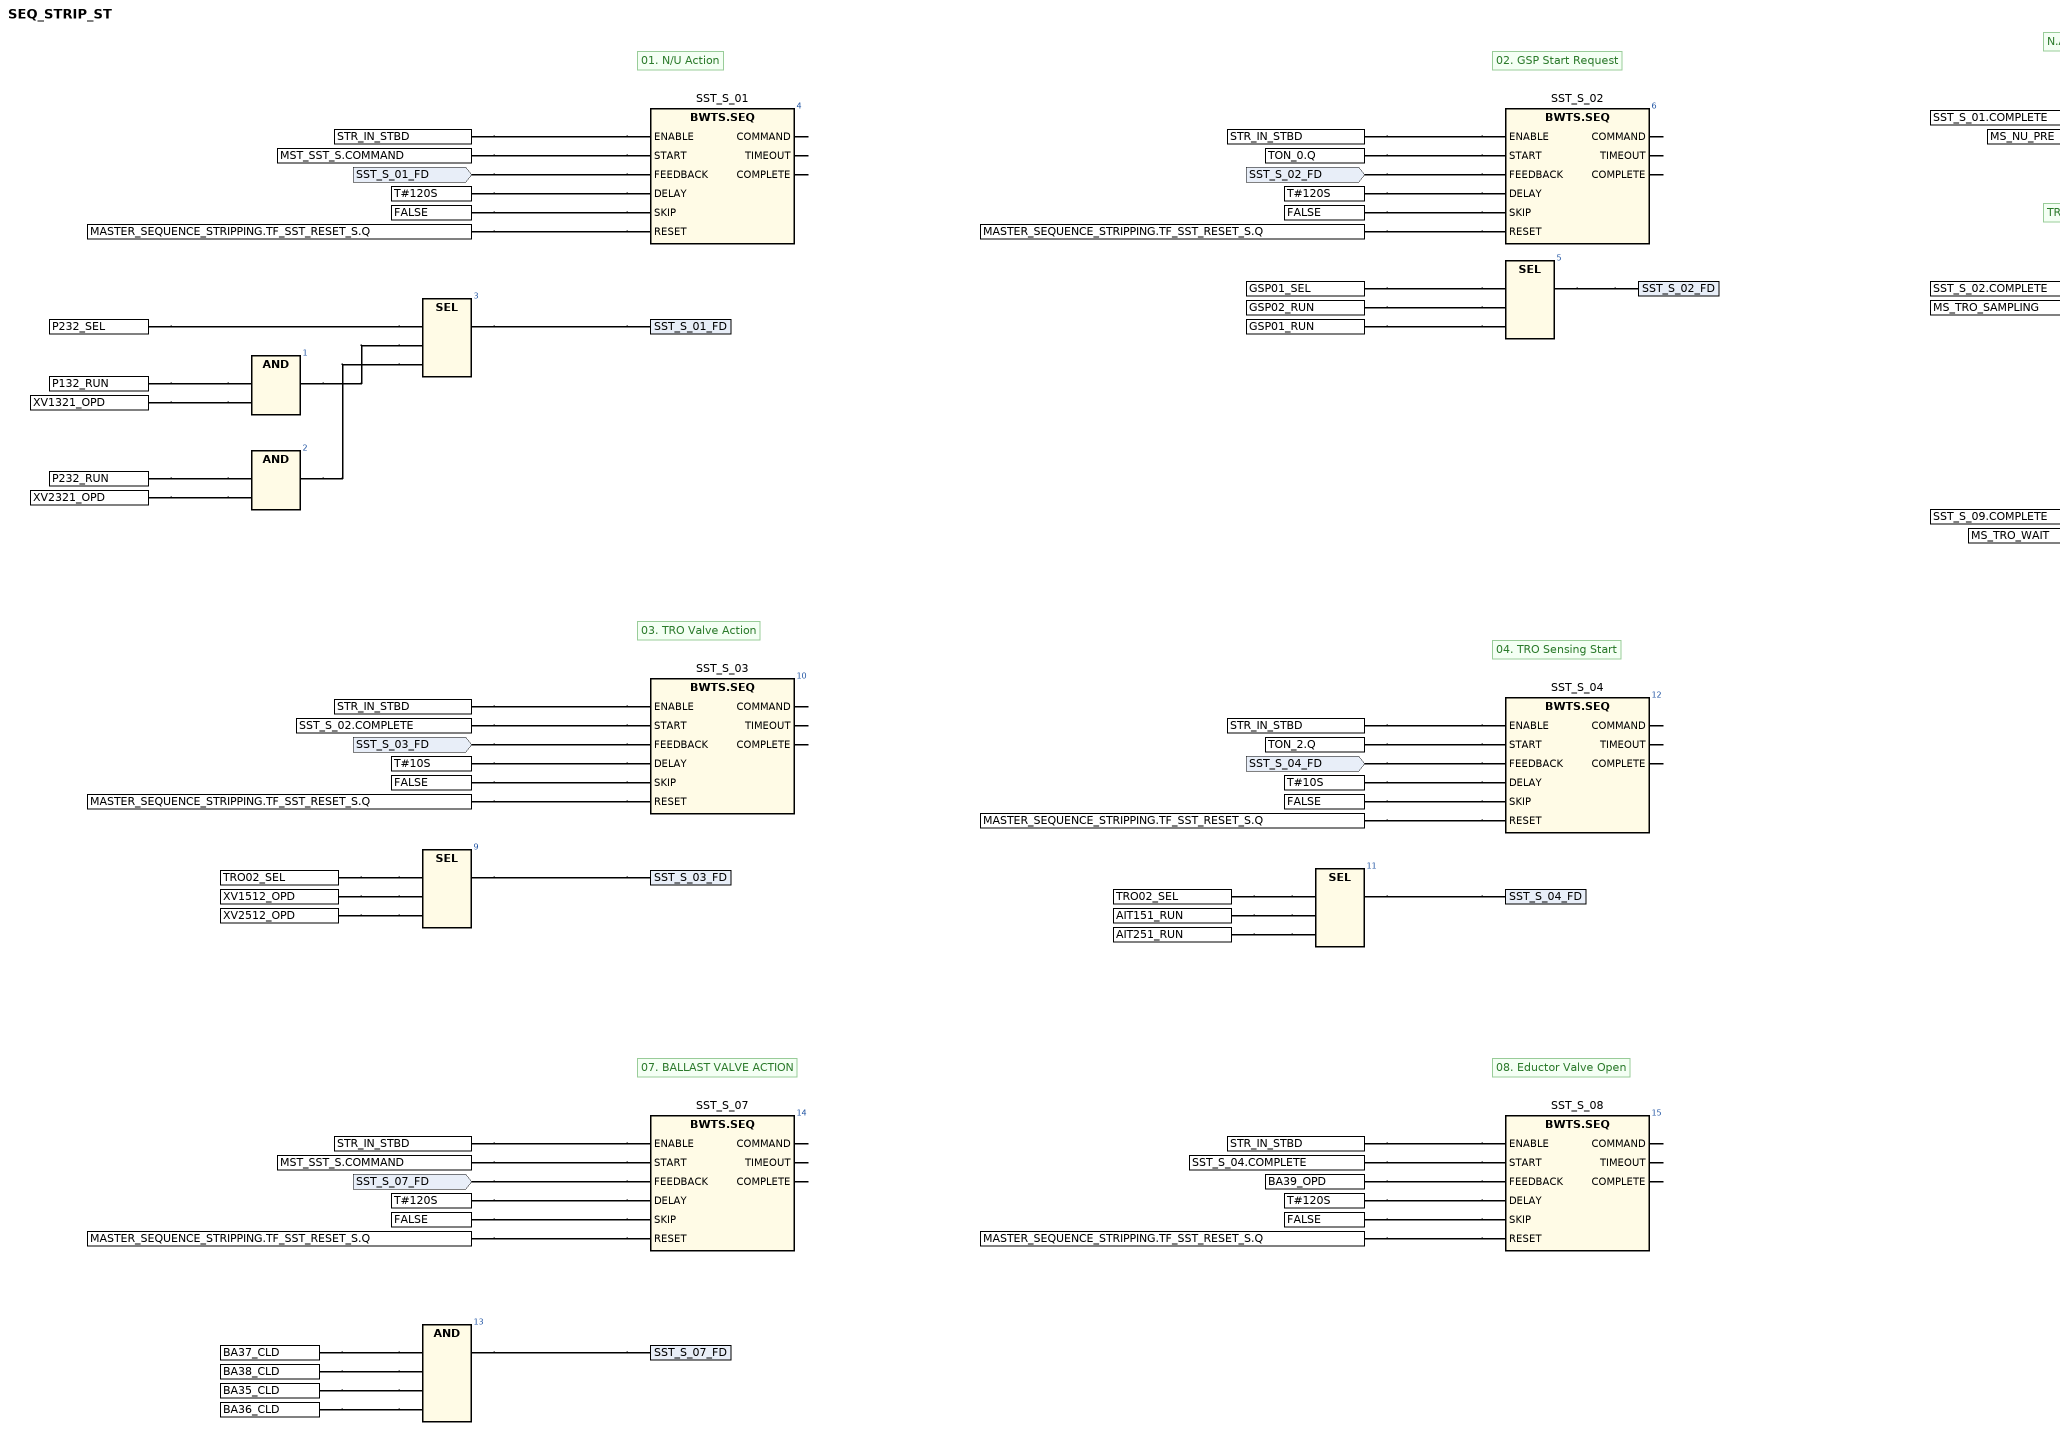
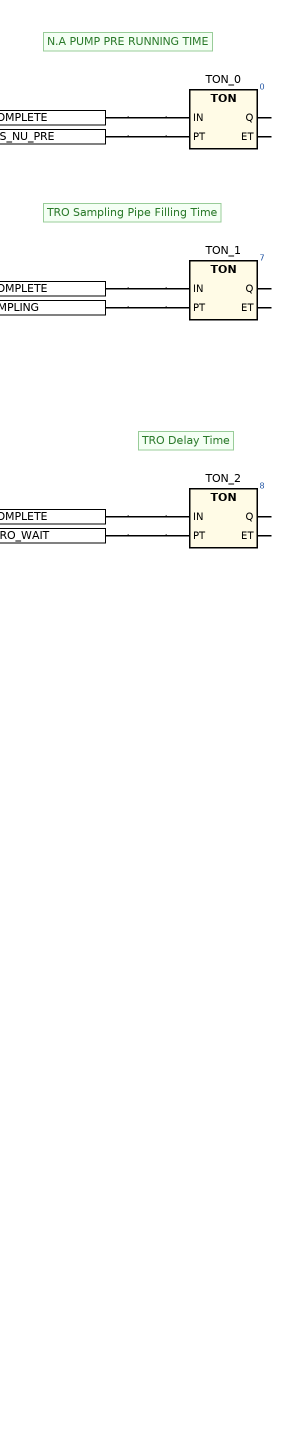
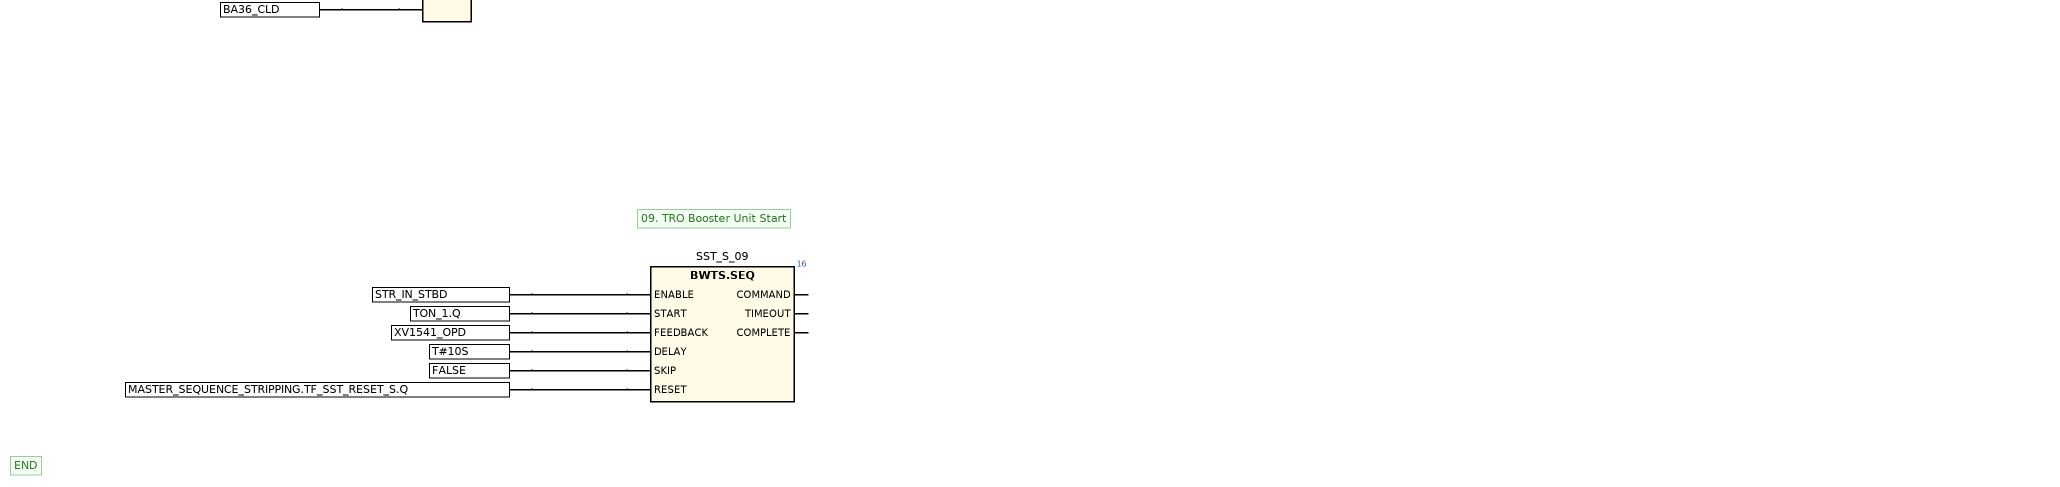
// N.A PUMP PRE RUNNING TIME
TON_0(IN := SST_S_01.COMPLETE, PT := MS_NU_PRE); // TON
(* SEL(P232_SEL, P132_RUN AND XV1321_OPD, P232_RUN AND XV2321_OPD); result not used *)
// 01. N/U Action
SST_S_01(
    ENABLE := STR_IN_STBD,
    START := MST_SST_S.COMMAND,
    FEEDBACK := _w1,
    DELAY := T#120S,
    SKIP := FALSE,
    RESET := MASTER_SEQUENCE_STRIPPING.TF_SST_RESET_S.Q); // BWTS.SEQ
(* SEL(GSP01_SEL, GSP02_RUN, GSP01_RUN); result not used *)
// 02. GSP Start Request
SST_S_02(
    ENABLE := STR_IN_STBD,
    START := TON_0.Q,
    FEEDBACK := _w2,
    DELAY := T#120S,
    SKIP := FALSE,
    RESET := MASTER_SEQUENCE_STRIPPING.TF_SST_RESET_S.Q); // BWTS.SEQ
// TRO Sampling Pipe Filling Time
TON_1(IN := SST_S_02.COMPLETE, PT := MS_TRO_SAMPLING); // TON
// TRO Delay Time
TON_2(IN := SST_S_09.COMPLETE, PT := MS_TRO_WAIT); // TON
(* SEL(TRO02_SEL, XV1512_OPD, XV2512_OPD); result not used *)
// 03. TRO Valve Action
SST_S_03(
    ENABLE := STR_IN_STBD,
    START := SST_S_02.COMPLETE,
    FEEDBACK := _w3,
    DELAY := T#10S,
    SKIP := FALSE,
    RESET := MASTER_SEQUENCE_STRIPPING.TF_SST_RESET_S.Q); // BWTS.SEQ
(* SEL(TRO02_SEL, AIT151_RUN, AIT251_RUN); result not used *)
// 04. TRO Sensing Start
SST_S_04(
    ENABLE := STR_IN_STBD,
    START := TON_2.Q,
    FEEDBACK := _w4,
    DELAY := T#10S,
    SKIP := FALSE,
    RESET := MASTER_SEQUENCE_STRIPPING.TF_SST_RESET_S.Q); // BWTS.SEQ
(* BA37_CLD AND BA38_CLD AND BA35_CLD AND BA36_CLD; result not used *)
// 07. BALLAST VALVE ACTION
SST_S_07(
    ENABLE := STR_IN_STBD,
    START := MST_SST_S.COMMAND,
    FEEDBACK := _w5,
    DELAY := T#120S,
    SKIP := FALSE,
    RESET := MASTER_SEQUENCE_STRIPPING.TF_SST_RESET_S.Q); // BWTS.SEQ
// 08. Eductor Valve Open
SST_S_08(
    ENABLE := STR_IN_STBD,
    START := SST_S_04.COMPLETE,
    FEEDBACK := BA39_OPD,
    DELAY := T#120S,
    SKIP := FALSE,
    RESET := MASTER_SEQUENCE_STRIPPING.TF_SST_RESET_S.Q); // BWTS.SEQ
// 09. TRO Booster Unit Start
// END
SST_S_09(
    ENABLE := STR_IN_STBD,
    START := TON_1.Q,
    FEEDBACK := XV1541_OPD,
    DELAY := T#10S,
    SKIP := FALSE,
    RESET := MASTER_SEQUENCE_STRIPPING.TF_SST_RESET_S.Q); // BWTS.SEQ

END_PROGRAM

// Device/Application/Logic/2.Sequence/MASTER_SEQUENCE_DIAGNOSIS
PROGRAM MASTER_SEQUENCE_DIAGNOSIS  // ADDED BY VER.1
VAR
	
	TON_0: TON;
	TON_DIAG_RESET: TON;
END_VAR

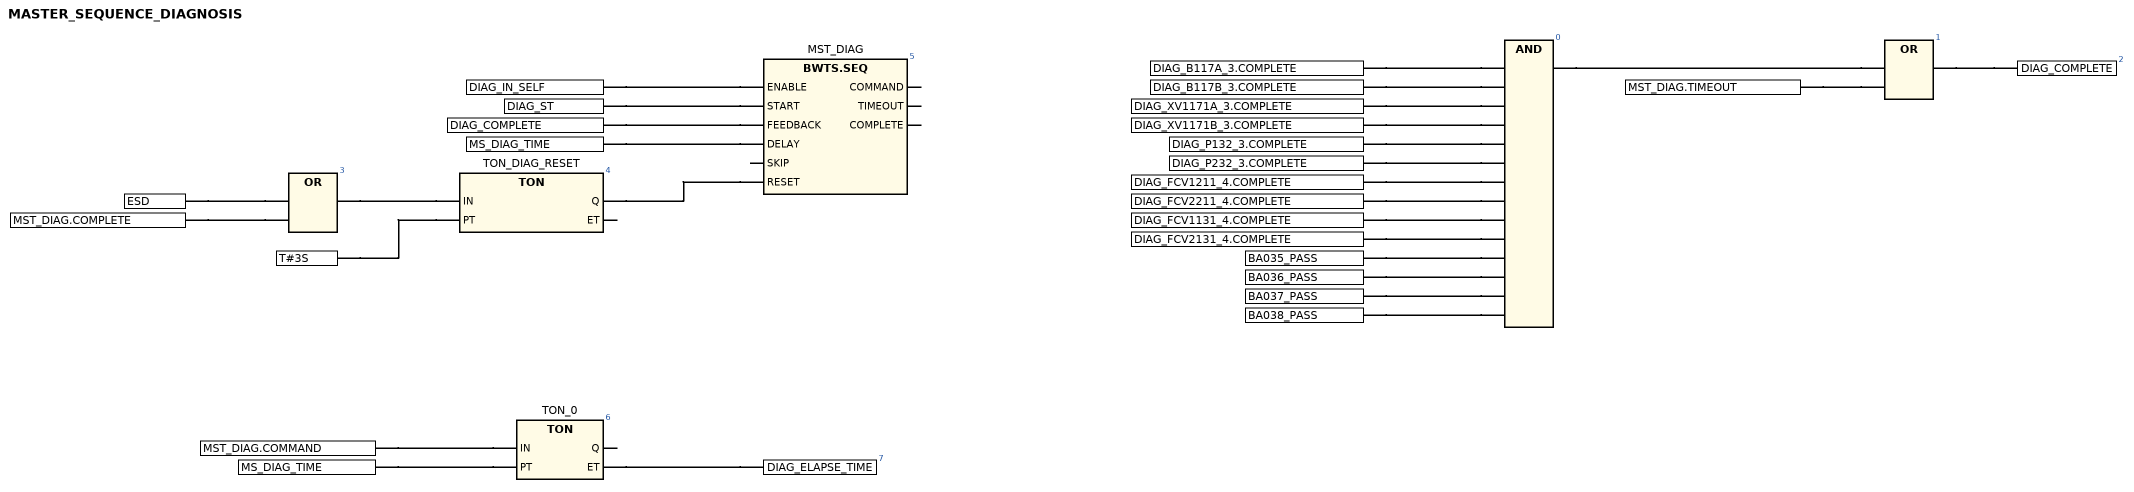
DIAG_COMPLETE := DIAG_B117A_3.COMPLETE AND DIAG_B117B_3.COMPLETE AND DIAG_XV1171A_3.COMPLETE AND DIAG_XV1171B_3.COMPLETE AND DIAG_P132_3.COMPLETE AND DIAG_P232_3.COMPLETE AND DIAG_FCV1211_4.COMPLETE AND DIAG_FCV2211_4.COMPLETE AND DIAG_FCV1131_4.COMPLETE AND DIAG_FCV2131_4.COMPLETE AND BA035_PASS AND BA036_PASS AND BA037_PASS AND BA038_PASS OR MST_DIAG.TIMEOUT;
TON_DIAG_RESET(IN := ESD OR MST_DIAG.COMPLETE, PT := T#3S); // TON
MST_DIAG(
    ENABLE := DIAG_IN_SELF,
    START := DIAG_ST,
    FEEDBACK := DIAG_COMPLETE,
    DELAY := MS_DIAG_TIME,
    RESET := TON_DIAG_RESET.Q); // BWTS.SEQ
TON_0(IN := MST_DIAG.COMMAND, PT := MS_DIAG_TIME); // TON
DIAG_ELAPSE_TIME := TON_0.ET;

END_PROGRAM

// Device/Application/Logic/2.Sequence/SEQ_DIAG_DEVICE
PROGRAM SEQ_DIAG_DEVICE
VAR
	B117A_1_TON: TON;
	B117A_2_TON: TON;
	B117A_RS : RS;
	B117B_1_TON: TON;
	B117B_2_TON: TON;
	B117B_RS : RS;
	
	XV1171A_1_TON: TON;
	XV1171A_2_TON: TON;
	XV1171A_RS : RS;
	XV1171B_1_TON: TON;
	XV1171B_2_TON: TON;
	XV1171B_RS : RS;
	
	P132_1_TON: TON;
	P132_2_TON: TON;
	P132_RS: RS;
	P232_1_TON: TON;
	P232_2_TON: TON;
	P232_RS: RS;
	
	FCV1211_1_TON: TON;
	FCV1211_2_TON: TON;
	FCV1211_3_TON: TON;
	FCV1211_RS: RS;
	FCV2211_1_TON: TON;
	FCV2211_2_TON: TON;
	FCV2211_3_TON: TON;
	FCV2211_RS: RS;
	
	FCV1131_1_TON: TON;
	FCV1131_2_TON: TON;
	FCV1131_3_TON: TON;
	FCV1131_RS: RS;
	FCV2131_1_TON: TON;
	FCV2131_2_TON: TON;
	FCV2131_3_TON: TON;
	FCV2131_RS: RS;
	
	BA35_1_TON: TON;
	BA35_2_TON: TON;
	BA35_RS : RS;
	BA36_1_TON: TON;
	BA36_2_TON: TON;
	BA36_RS : RS;
	BA37_1_TON: TON;
	BA37_2_TON: TON;
	BA37_RS : RS;
	BA38_1_TON: TON;
	BA38_2_TON: TON;
	BA38_RS : RS;
END_VAR

// B117A
DIAG_B117A_1(ENABLE:=DIAG_IN_SELF, START:=DIAG_ST, FEEDBACK:=B117A_SPD, RESET:=MASTER_SEQUENCE_DIAGNOSIS.TON_DIAG_RESET.Q);
B117A_1_TON(IN:=DIAG_B117A_1.COMPLETE, PT:=T#5S);
DIAG_B117A_2(ENABLE:=DIAG_IN_SELF, START:=B117A_1_TON.Q, FEEDBACK:=B117A_RUN, RESET:=MASTER_SEQUENCE_DIAGNOSIS.TON_DIAG_RESET.Q);
B117A_2_TON(IN:=DIAG_B117A_2.COMPLETE, PT:=T#5S);
DIAG_B117A_3(ENABLE:=DIAG_IN_SELF, START:=B117A_2_TON.Q, FEEDBACK:=B117A_SPD, RESET:=MASTER_SEQUENCE_DIAGNOSIS.TON_DIAG_RESET.Q);
B117A_RS(SET:=DIAG_B117A_3.COMPLETE, RESET1:= DIAG_ST, Q1=> B117A_PASS);
// B117B
DIAG_B117B_1(ENABLE:=DIAG_IN_SELF, START:=DIAG_ST, FEEDBACK:=B117B_SPD, RESET:=MASTER_SEQUENCE_DIAGNOSIS.TON_DIAG_RESET.Q);
B117B_1_TON(IN:=DIAG_B117B_1.COMPLETE, PT:=T#5S);
DIAG_B117B_2(ENABLE:=DIAG_IN_SELF, START:=B117B_1_TON.Q, FEEDBACK:=B117B_RUN, RESET:=MASTER_SEQUENCE_DIAGNOSIS.TON_DIAG_RESET.Q);
B117B_2_TON(IN:=DIAG_B117B_2.COMPLETE, PT:=T#5S);
DIAG_B117B_3(ENABLE:=DIAG_IN_SELF, START:=B117B_2_TON.Q, FEEDBACK:=B117B_SPD, RESET:=MASTER_SEQUENCE_DIAGNOSIS.TON_DIAG_RESET.Q);
B117B_RS(SET:=DIAG_B117B_3.COMPLETE, RESET1:= DIAG_ST, Q1=> B117B_PASS);
// XV1171A
DIAG_XV1171A_1(ENABLE:=DIAG_IN_SELF, START:=DIAG_ST, FEEDBACK:=XV1171A_CLD, RESET:=MASTER_SEQUENCE_DIAGNOSIS.TON_DIAG_RESET.Q);
XV1171A_1_TON(IN:=DIAG_XV1171A_1.COMPLETE, PT:=T#5S);
DIAG_XV1171A_2(ENABLE:=DIAG_IN_SELF, START:=XV1171A_1_TON.Q, FEEDBACK:=XV1171A_OPD, RESET:=MASTER_SEQUENCE_DIAGNOSIS.TON_DIAG_RESET.Q);
XV1171A_2_TON(IN:=DIAG_XV1171A_2.COMPLETE, PT:=T#5S);
DIAG_XV1171A_3(ENABLE:=DIAG_IN_SELF, START:=XV1171A_2_TON.Q, FEEDBACK:=XV1171A_CLD, RESET:=MASTER_SEQUENCE_DIAGNOSIS.TON_DIAG_RESET.Q);
XV1171A_RS(SET:=DIAG_XV1171A_3.COMPLETE, RESET1:= DIAG_ST, Q1=> XV1171A_PASS);
// XV1171B
DIAG_XV1171B_1(ENABLE:=DIAG_IN_SELF, START:=DIAG_ST, FEEDBACK:=XV1171B_CLD, RESET:=MASTER_SEQUENCE_DIAGNOSIS.TON_DIAG_RESET.Q);
XV1171B_1_TON(IN:=DIAG_XV1171B_1.COMPLETE, PT:=T#5S);
DIAG_XV1171B_2(ENABLE:=DIAG_IN_SELF, START:=XV1171B_1_TON.Q, FEEDBACK:=XV1171B_OPD, RESET:=MASTER_SEQUENCE_DIAGNOSIS.TON_DIAG_RESET.Q);
XV1171B_2_TON(IN:=DIAG_XV1171B_2.COMPLETE, PT:=T#5S);
DIAG_XV1171B_3(ENABLE:=DIAG_IN_SELF, START:=XV1171B_2_TON.Q, FEEDBACK:=XV1171B_CLD, RESET:=MASTER_SEQUENCE_DIAGNOSIS.TON_DIAG_RESET.Q);
XV1171B_RS(SET:=DIAG_XV1171B_3.COMPLETE, RESET1:= DIAG_ST, Q1=> XV1171B_PASS);
// P132
DIAG_P132_1(ENABLE:=DIAG_IN_SELF, START:=DIAG_ST, FEEDBACK:=P132_SPD, RESET:=MASTER_SEQUENCE_DIAGNOSIS.TON_DIAG_RESET.Q);
P132_1_TON(IN:=DIAG_P132_1.COMPLETE, PT:=T#5S);
DIAG_P132_2(ENABLE:=DIAG_IN_SELF, START:=P132_1_TON.Q, FEEDBACK:=P132_RUN, RESET:=MASTER_SEQUENCE_DIAGNOSIS.TON_DIAG_RESET.Q);
P132_2_TON(IN:=DIAG_P132_2.COMPLETE, PT:=T#5S);
DIAG_P132_3(ENABLE:=DIAG_IN_SELF, START:=P132_2_TON.Q, FEEDBACK:=P132_SPD, RESET:=MASTER_SEQUENCE_DIAGNOSIS.TON_DIAG_RESET.Q);
P132_RS(SET:=DIAG_P132_3.COMPLETE, RESET1:= DIAG_ST, Q1=> P132_PASS);
// P232
DIAG_P232_1(ENABLE:=DIAG_IN_SELF, START:=DIAG_ST, FEEDBACK:=P232_SPD, RESET:=MASTER_SEQUENCE_DIAGNOSIS.TON_DIAG_RESET.Q);
P232_1_TON(IN:=DIAG_P232_1.COMPLETE, PT:=T#5S);
DIAG_P232_2(ENABLE:=DIAG_IN_SELF, START:=P232_1_TON.Q, FEEDBACK:=P232_RUN, RESET:=MASTER_SEQUENCE_DIAGNOSIS.TON_DIAG_RESET.Q);
P232_2_TON(IN:=DIAG_P232_2.COMPLETE, PT:=T#5S);
DIAG_P232_3(ENABLE:=DIAG_IN_SELF, START:=P232_2_TON.Q, FEEDBACK:=P232_SPD, RESET:=MASTER_SEQUENCE_DIAGNOSIS.TON_DIAG_RESET.Q);
P232_RS(SET:=DIAG_P232_3.COMPLETE, RESET1:= DIAG_ST, Q1=> P232_PASS);

// FCV1211
DIAG_FCV1211_1(ENABLE:=DIAG_IN_SELF, START:=DIAG_ST, FEEDBACK:=FCV_1211_FD<=5, RESET:=MASTER_SEQUENCE_DIAGNOSIS.TON_DIAG_RESET.Q);
FCV1211_1_TON(IN:=DIAG_FCV1211_1.COMPLETE, PT:=T#5S);
DIAG_FCV1211_2(ENABLE:=DIAG_IN_SELF, START:=FCV1211_1_TON.Q, FEEDBACK:=FCV_1211_FD>=45 AND FCV_1211_FD<=55, RESET:=MASTER_SEQUENCE_DIAGNOSIS.TON_DIAG_RESET.Q);
FCV1211_2_TON(IN:=DIAG_FCV1211_2.COMPLETE, PT:=T#5S);
DIAG_FCV1211_3(ENABLE:=DIAG_IN_SELF, START:=FCV1211_2_TON.Q, FEEDBACK:=FCV_1211_FD>=95, RESET:=MASTER_SEQUENCE_DIAGNOSIS.TON_DIAG_RESET.Q);
FCV1211_3_TON(IN:=DIAG_FCV1211_3.COMPLETE, PT:=T#5S);
DIAG_FCV1211_4(ENABLE:=DIAG_IN_SELF, START:=FCV1211_3_TON.Q, FEEDBACK:=FCV_1211_FD<=5, RESET:=MASTER_SEQUENCE_DIAGNOSIS.TON_DIAG_RESET.Q);
FCV1211_RS(SET:=DIAG_FCV1211_4.COMPLETE, RESET1:= DIAG_ST, Q1=> FCV1211_PASS);
// FCV2211
DIAG_FCV2211_1(ENABLE:=DIAG_IN_SELF, START:=DIAG_ST, FEEDBACK:=FCV_2211_FD<=5, RESET:=MASTER_SEQUENCE_DIAGNOSIS.TON_DIAG_RESET.Q);
FCV2211_1_TON(IN:=DIAG_FCV2211_1.COMPLETE, PT:=T#5S);
DIAG_FCV2211_2(ENABLE:=DIAG_IN_SELF, START:=FCV2211_1_TON.Q, FEEDBACK:=FCV_2211_FD>=45 AND FCV_2211_FD<=55, RESET:=MASTER_SEQUENCE_DIAGNOSIS.TON_DIAG_RESET.Q);
FCV2211_2_TON(IN:=DIAG_FCV2211_2.COMPLETE, PT:=T#5S);
DIAG_FCV2211_3(ENABLE:=DIAG_IN_SELF, START:=FCV2211_2_TON.Q, FEEDBACK:=FCV_2211_FD>=95, RESET:=MASTER_SEQUENCE_DIAGNOSIS.TON_DIAG_RESET.Q);
FCV2211_3_TON(IN:=DIAG_FCV2211_3.COMPLETE, PT:=T#5S);
DIAG_FCV2211_4(ENABLE:=DIAG_IN_SELF, START:=FCV2211_3_TON.Q, FEEDBACK:=FCV_2211_FD<=5, RESET:=MASTER_SEQUENCE_DIAGNOSIS.TON_DIAG_RESET.Q);
FCV2211_RS(SET:=DIAG_FCV2211_4.COMPLETE, RESET1:= DIAG_ST, Q1=> FCV2211_PASS);

// FCV1131
DIAG_FCV1131_1(ENABLE:=DIAG_IN_SELF, START:=DIAG_ST, FEEDBACK:=FCV_1131_FD<=5, RESET:=MASTER_SEQUENCE_DIAGNOSIS.TON_DIAG_RESET.Q);
FCV1131_1_TON(IN:=DIAG_FCV1131_1.COMPLETE, PT:=T#5S);
DIAG_FCV1131_2(ENABLE:=DIAG_IN_SELF, START:=FCV1131_1_TON.Q, FEEDBACK:=FCV_1131_FD>=45 AND FCV_1131_FD<=55, RESET:=MASTER_SEQUENCE_DIAGNOSIS.TON_DIAG_RESET.Q);
FCV1131_2_TON(IN:=DIAG_FCV1131_2.COMPLETE, PT:=T#5S);
DIAG_FCV1131_3(ENABLE:=DIAG_IN_SELF, START:=FCV1131_2_TON.Q, FEEDBACK:=FCV_1131_FD>=95, RESET:=MASTER_SEQUENCE_DIAGNOSIS.TON_DIAG_RESET.Q);
FCV1131_3_TON(IN:=DIAG_FCV1131_3.COMPLETE, PT:=T#5S);
DIAG_FCV1131_4(ENABLE:=DIAG_IN_SELF, START:=FCV1131_3_TON.Q, FEEDBACK:=FCV_1131_FD<=5, RESET:=MASTER_SEQUENCE_DIAGNOSIS.TON_DIAG_RESET.Q);
FCV1131_RS(SET:=DIAG_FCV1131_4.COMPLETE, RESET1:= DIAG_ST, Q1=> FCV1131_PASS);
// FCV2131
DIAG_FCV2131_1(ENABLE:=DIAG_IN_SELF, START:=DIAG_ST, FEEDBACK:=FCV_2131_FD<=5, RESET:=MASTER_SEQUENCE_DIAGNOSIS.TON_DIAG_RESET.Q);
FCV2131_1_TON(IN:=DIAG_FCV2131_1.COMPLETE, PT:=T#5S);
DIAG_FCV2131_2(ENABLE:=DIAG_IN_SELF, START:=FCV2131_1_TON.Q, FEEDBACK:=FCV_2131_FD>=45 AND FCV_2131_FD<=55, RESET:=MASTER_SEQUENCE_DIAGNOSIS.TON_DIAG_RESET.Q);
FCV2131_2_TON(IN:=DIAG_FCV2131_2.COMPLETE, PT:=T#5S);
DIAG_FCV2131_3(ENABLE:=DIAG_IN_SELF, START:=FCV2131_2_TON.Q, FEEDBACK:=FCV_2131_FD>=95, RESET:=MASTER_SEQUENCE_DIAGNOSIS.TON_DIAG_RESET.Q);
FCV2131_3_TON(IN:=DIAG_FCV2131_3.COMPLETE, PT:=T#5S);
DIAG_FCV2131_4(ENABLE:=DIAG_IN_SELF, START:=FCV2131_3_TON.Q, FEEDBACK:=FCV_2131_FD<=5, RESET:=MASTER_SEQUENCE_DIAGNOSIS.TON_DIAG_RESET.Q);
FCV2131_RS(SET:=DIAG_FCV2131_4.COMPLETE, RESET1:= DIAG_ST, Q1=> FCV2131_PASS);

// BA35
DIAG_BA35_1(ENABLE:=DIAG_IN_SELF, START:=DIAG_ST, FEEDBACK:=BA35_CLD, RESET:=MASTER_SEQUENCE_DIAGNOSIS.TON_DIAG_RESET.Q);
BA35_1_TON(IN:=DIAG_BA35_1.COMPLETE, PT:=T#5S);
DIAG_BA35_2(ENABLE:=DIAG_IN_SELF, START:=BA35_1_TON.Q, FEEDBACK:=BA35_OPD, RESET:=MASTER_SEQUENCE_DIAGNOSIS.TON_DIAG_RESET.Q);
BA35_2_TON(IN:=DIAG_BA35_2.COMPLETE, PT:=T#5S);
DIAG_BA35_3(ENABLE:=DIAG_IN_SELF, START:=BA35_2_TON.Q, FEEDBACK:=BA35_CLD, RESET:=MASTER_SEQUENCE_DIAGNOSIS.TON_DIAG_RESET.Q);
BA35_RS(SET:=DIAG_BA35_3.COMPLETE, RESET1:= DIAG_ST, Q1=> BA035_PASS);

// BA36
DIAG_BA36_1(ENABLE:=DIAG_IN_SELF, START:=DIAG_ST, FEEDBACK:=BA36_CLD, RESET:=MASTER_SEQUENCE_DIAGNOSIS.TON_DIAG_RESET.Q);
BA36_1_TON(IN:=DIAG_BA36_1.COMPLETE, PT:=T#5S);
DIAG_BA36_2(ENABLE:=DIAG_IN_SELF, START:=BA36_1_TON.Q, FEEDBACK:=BA36_OPD, RESET:=MASTER_SEQUENCE_DIAGNOSIS.TON_DIAG_RESET.Q);
BA36_2_TON(IN:=DIAG_BA36_2.COMPLETE, PT:=T#5S);
DIAG_BA36_3(ENABLE:=DIAG_IN_SELF, START:=BA36_2_TON.Q, FEEDBACK:=BA36_CLD, RESET:=MASTER_SEQUENCE_DIAGNOSIS.TON_DIAG_RESET.Q);
BA36_RS(SET:=DIAG_BA36_3.COMPLETE, RESET1:= DIAG_ST, Q1=> BA036_PASS);

// BA37
DIAG_BA37_1(ENABLE:=DIAG_IN_SELF, START:=DIAG_ST, FEEDBACK:=BA37_CLD, RESET:=MASTER_SEQUENCE_DIAGNOSIS.TON_DIAG_RESET.Q);
BA37_1_TON(IN:=DIAG_BA37_1.COMPLETE, PT:=T#5S);
DIAG_BA37_2(ENABLE:=DIAG_IN_SELF, START:=BA37_1_TON.Q, FEEDBACK:=BA37_OPD, RESET:=MASTER_SEQUENCE_DIAGNOSIS.TON_DIAG_RESET.Q);
BA37_2_TON(IN:=DIAG_BA37_2.COMPLETE, PT:=T#5S);
DIAG_BA37_3(ENABLE:=DIAG_IN_SELF, START:=BA37_2_TON.Q, FEEDBACK:=BA37_CLD, RESET:=MASTER_SEQUENCE_DIAGNOSIS.TON_DIAG_RESET.Q);
BA37_RS(SET:=DIAG_BA37_3.COMPLETE, RESET1:= DIAG_ST, Q1=> BA037_PASS);

// BA38
DIAG_BA38_1(ENABLE:=DIAG_IN_SELF, START:=DIAG_ST, FEEDBACK:=BA38_CLD, RESET:=MASTER_SEQUENCE_DIAGNOSIS.TON_DIAG_RESET.Q);
BA38_1_TON(IN:=DIAG_BA38_1.COMPLETE, PT:=T#5S);
DIAG_BA38_2(ENABLE:=DIAG_IN_SELF, START:=BA38_1_TON.Q, FEEDBACK:=BA38_OPD, RESET:=MASTER_SEQUENCE_DIAGNOSIS.TON_DIAG_RESET.Q);
BA38_2_TON(IN:=DIAG_BA38_2.COMPLETE, PT:=T#5S);
DIAG_BA38_3(ENABLE:=DIAG_IN_SELF, START:=BA38_2_TON.Q, FEEDBACK:=BA38_CLD, RESET:=MASTER_SEQUENCE_DIAGNOSIS.TON_DIAG_RESET.Q);
BA38_RS(SET:=DIAG_BA38_3.COMPLETE, RESET1:= DIAG_ST, Q1=> BA038_PASS);

END_PROGRAM

// Device/Application/Logic/2.Sequence/SEQ_DIAG_INSTRUMENT
PROGRAM SEQ_DIAG_INSTRUMENT
VAR
END_VAR

RF142A_PASS := 1 ;
RF142B_PASS := 1 ;
RF142C_PASS := 1 ;

AIT151_PASS := 1 ;
AIT251_PASS := 1 ;

TE1111_PASS := 1 ;
CT1111_PASS := 1 ;

PT1721_PASS := 1 ;
PT1722_PASS := 1 ;

AIT1121_PASS := 1 ;
AIT1122_PASS := 1 ;
AIT1123_PASS := 1 ;

PT1121_PASS := 1 ;

FIT1211_PASS := 1 ;
FIT2211_PASS := 1 ;

FIT1131_PASS := 1 ;
FIT2131_PASS := 1 ;

LIT1311_PASS := 1 ;

END_PROGRAM

// Device/Application/Logic/0.ALARM/ALARM_BUZZER_1
PROGRAM ALARM_BUZZER_1
VAR
	// EU
	R_TRIG_B117A_STF, R_TRIG_B117A_SPF, R_TRIG_B117B_STF, R_TRIG_B117B_SPF, R_TRIG_XV1171A_OPF, R_TRIG_XV1171A_CLF, R_TRIG_XV1171B_OPF, R_TRIG_XV1171B_CLF,
	R_TRIG_B_117A_F, R_TRIG_B_117B_F, R_TRIG_B_117A_OFF, R_TRIG_B_117B_OFF, R_TRIG_BLR_BYPASS, R_TRIG_BLR_BOTH_F,
	R_TRIG_PT_1121_HI, R_TRIG_PT_1121_LO, R_TRIG_PT_1121_LL, R_TRIG_LS_1111_LL, R_TRIG_LS_1141_HI, R_TRIG_ER_FAN_OFF,
	R_TRIG_AIT_1121_HH, R_TRIG_AIT_1121_HI, R_TRIG_AIT_1122_HH, R_TRIG_AIT_1122_HI, R_TRIG_AIT_1123_HH, R_TRIG_AIT_1123_HI, 
	R_TRIG_TE_1111_HI, R_TRIG_TE_1111_LO, R_TRIG_TE_1111_LL, R_TRIG_CT_1111_LO, R_TRIG_CT_1111_LL,
	R_TRIG_ZS_1112A_CL, R_TRIG_ZS_1112A_OP, R_TRIG_ZS_1113A_CL, R_TRIG_ZS_1113A_OP, R_TRIG_ZS_1114A_CL, R_TRIG_ZS_1114A_OP, 
	
	// SWFU
	R_TRIG_P171A_STF, R_TRIG_P171A_SPF, R_TRIG_P171B_STF, R_TRIG_P171B_SPF, R_TRIG_SWFP_BOTH_F,
	R_TRIG_P_171A_F, R_TRIG_P_171B_F, R_TRIG_P_171A_OFF, R_TRIG_P_171B_OFF,
	R_TRIG_PT_1721_HI, R_TRIG_PT_1721_LO, R_TRIG_PT_1721_LL, R_TRIG_PT_1722_HH, R_TRIG_PT_1722_HI, R_TRIG_PT_1722_LO, R_TRIG_SWFU_DP_HI,  R_TRIG_SWFU_DP_HH,

	// INJECTION
	R_TRIG_FCV1131_CF, R_TRIG_FIT_1131_LO, R_TRIG_FIT_1131_LL, R_TRIG_RFS_1131,
	R_TRIG_FCV2131_CF, R_TRIG_FIT_2131_LO, R_TRIG_FIT_2131_LL, R_TRIG_RFS_2131,
	
 
	// MAIN TRC
	R_TRIG_FCV1211_CF,	R_TRIG_FIT_1211_HH, R_TRIG_FIT_1211_HI, R_TRIG_FIT_1211_LO,
	R_TRIG_FCV2211_CF,	R_TRIG_FIT_2211_HH, R_TRIG_FIT_2211_HI, R_TRIG_FIT_2211_LO,
		
	// NU
	R_TRIG_P_132_TRIP, R_TRIG_P132_STF, R_TRIG_P132_SPF, R_TRIG_DPS_1321,
	R_TRIG_P_232_TRIP, R_TRIG_P232_STF, R_TRIG_P232_SPF, R_TRIG_DPS_2321,   
	
	R_TRIG_LIT_1311_HI, R_TRIG_LIT_1311_LO, R_TRIG_LIT_1311_LL,
	
	// RECTIFIER
	R_TRIG_RF142A_STF, R_TRIG_RF142A_SPF, R_TRIG_RF142B_STF, R_TRIG_RF142B_SPF, R_TRIG_RF142C_STF, R_TRIG_RF142C_SPF,  
	R_TRIG_RF_142A_E, R_TRIG_RF_142B_E, R_TRIG_RF_142C_E, R_TRIG_RF_ALL_SPD,
	R_TRIG_REC1001, R_TRIG_REC1002, R_TRIG_REC1003, R_TRIG_REC1004, R_TRIG_REC1005, R_TRIG_REC1006, R_TRIG_REC1007, R_TRIG_REC1008, R_TRIG_REC1009, R_TRIG_REC1010, R_TRIG_REC1011,
	R_TRIG_REC1012, R_TRIG_REC1013, R_TRIG_REC1014, R_TRIG_REC1015, R_TRIG_REC1022, R_TRIG_REC1023, R_TRIG_REC1024, R_TRIG_REC1025, R_TRIG_REC1026, R_TRIG_REC1032, R_TRIG_REC1033,
	R_TRIG_REC1017_HH, R_TRIG_REC1017_HI, R_TRIG_REC1018_HH, R_TRIG_REC1018_HI, R_TRIG_REC1019_HH, R_TRIG_REC1019_HI,
	R_TRIG_REC1020_HH, R_TRIG_REC1020_HI, R_TRIG_REC1021_HH, R_TRIG_REC1021_HI, R_TRIG_REC1027_HH, R_TRIG_REC1027_HI,
	R_TRIG_REC2001, R_TRIG_REC2002, R_TRIG_REC2003, R_TRIG_REC2004, R_TRIG_REC2005, R_TRIG_REC2006, R_TRIG_REC2007, R_TRIG_REC2008, R_TRIG_REC2009, R_TRIG_REC2010, R_TRIG_REC2011,
	R_TRIG_REC2012, R_TRIG_REC2013, R_TRIG_REC2014, R_TRIG_REC2015, R_TRIG_REC2022, R_TRIG_REC2023, R_TRIG_REC2024, R_TRIG_REC2025, R_TRIG_REC2026, R_TRIG_REC2032, R_TRIG_REC2033,
	R_TRIG_REC2017_HH, R_TRIG_REC2017_HI, R_TRIG_REC2018_HH, R_TRIG_REC2018_HI, R_TRIG_REC2019_HH, R_TRIG_REC2019_HI,
	R_TRIG_REC2020_HH, R_TRIG_REC2020_HI, R_TRIG_REC2021_HH, R_TRIG_REC2021_HI, R_TRIG_REC2027_HH, R_TRIG_REC2027_HI,
	R_TRIG_REC3001, R_TRIG_REC3002, R_TRIG_REC3003, R_TRIG_REC3004, R_TRIG_REC3005, R_TRIG_REC3006, R_TRIG_REC3007, R_TRIG_REC3008, R_TRIG_REC3009, R_TRIG_REC3010, R_TRIG_REC3011,
	R_TRIG_REC3012, R_TRIG_REC3013, R_TRIG_REC3014, R_TRIG_REC3015, R_TRIG_REC3022, R_TRIG_REC3023, R_TRIG_REC3024, R_TRIG_REC3025, R_TRIG_REC3026, R_TRIG_REC3032, R_TRIG_REC3033,
	R_TRIG_REC3017_HH, R_TRIG_REC3017_HI, R_TRIG_REC3018_HH, R_TRIG_REC3018_HI, R_TRIG_REC3019_HH, R_TRIG_REC3019_HI,
	R_TRIG_REC3020_HH, R_TRIG_REC3020_HI, R_TRIG_REC3021_HH, R_TRIG_REC3021_HI, R_TRIG_REC3027_HH, R_TRIG_REC3027_HI,
		
	// TRO
	R_TRIG_AIT_151_E, R_TRIG_AIT_151_F,
	R_TRIG_AIT_251_E, R_TRIG_AIT_251_F,
	R_TRIG_BTRO_HH_S, R_TRIG_BTRO_HI_S, R_TRIG_BTRO_LO_S, R_TRIG_BTRO_LL_S, R_TRIG_DTRO_HH_S, R_TRIG_DTRO_HI_S,
	R_TRIG_BTRO_HH_P, R_TRIG_BTRO_HI_P, R_TRIG_BTRO_LO_P, R_TRIG_BTRO_LL_P, R_TRIG_DTRO_HH_P, R_TRIG_DTRO_HI_P,
	R_TRIG_STRO_HH, R_TRIG_STRO_HI,
	R_TRIG_LS_1901_HH,
		
	// BALLAST SYSTEM
	R_TRIG_WBP01_STF, R_TRIG_WBP01_SPF, R_TRIG_WBP_01_AL, R_TRIG_WBP_01_FAULT,
	R_TRIG_WBP02_STF, R_TRIG_WBP02_SPF, R_TRIG_WBP_02_AL, R_TRIG_WBP_02_FAULT,
	R_TRIG_GSP01_STF, R_TRIG_GSP01_SPF, R_TRIG_GSP_01_AL, R_TRIG_GSP_01_FAULT,
	R_TRIG_GSP02_STF, R_TRIG_GSP02_SPF, R_TRIG_GSP_02_AL, R_TRIG_GSP_02_FAULT,
	
	R_TRIG_SYS_BYPASS_1, R_TRIG_SYS_BYPASS_2, R_TRIG_SYS_BYPASS_3, R_TRIG_SYS_BYPASS_4,
	 
	R_TRIG_BAL_VV_AL_S, R_TRIG_BAL_VV_AL_P, R_TRIG_DEBAL_VV_AL_S, R_TRIG_DEBAL_VV_AL_P, R_TRIG_STR_VV_AL_S,
	
	R_TRIG_AP_LVL_LO, R_TRIG_AP_LVL_LL,
	R_GAS_LEAK_AL, 
		
	R_FU_BYPASS_1, R_FU_BYPASS_2, R_FU_BYPASS_3,  
	
	// SD
	R_TRIG_ESD, R_TRIG_PSD_11, R_TRIG_PSD_12, R_TRIG_PSD_21, R_TRIG_PSD_22, R_TRIG_PSD_31, R_TRIG_PSD_41, R_TRIG_PSD_42,
	
	// SYSTEM
	R_TRIG_DISABLE1,
	R_TRIG_DISABLE2,
	R_TRIG_DISABLE3,
	R_TRIG_DISABLE4, 
	R_TRIG_MM_AIT1121, 
	R_TRIG_MM_AIT1122, 
	R_TRIG_MM_AIT1123, 
	R_TRIG_MM_REPAIR,

	R_TRIG_MCC_100_OFF,
	R_TRIG_PR_FAN_OFF,
	R_TRIG_RH_EU_AL, 
	R_TRIG_RH_AIT1121_AL,
	R_TRIG_RH_AIT1122_AL, 
	R_TRIG_RH_AIT1123_AL, 
	R_TRIG_RH_AIT151_AL, 
	R_TRIG_RH_AIT251_AL, 

	R_TRIG_RH_P132_AL, 
	R_TRIG_RH_P232_AL, 
	
	R_TRIG_RH_P171A_AL, 
	R_TRIG_RH_P171B_AL,
	R_TRIG_CC100_TEMP_HI, 
	R_TRIG_ESTOP_HMI, 
	R_TRIG_ESTOP_CC, 
	R_TRIG_ESTOP_RF, 
	R_TRIG_GPS_ALARM,
		
	// SEQUENCE TIME-OUT BALLASTING START
	R_TRIG_BST_S_T01, R_TRIG_BST_P_T01,
	R_TRIG_BST_S_T03, R_TRIG_BST_P_T03,
	R_TRIG_BST_S_T04, R_TRIG_BST_P_T04,
	R_TRIG_BST_S_T05, R_TRIG_BST_P_T05,
	R_TRIG_BST_S_T06, R_TRIG_BST_P_T06,
	R_TRIG_BST_S_T07, R_TRIG_BST_P_T07,
	R_TRIG_BST_S_T08, R_TRIG_BST_P_T08,
	R_TRIG_BST_S_T10, R_TRIG_BST_P_T10,
	R_TRIG_BST_S_T12, R_TRIG_BST_P_T12,
	R_TRIG_BST_S_T13, R_TRIG_BST_P_T13,
	R_TRIG_BST_S_T14, R_TRIG_BST_P_T14,
	R_TRIG_BST_S_T15, R_TRIG_BST_P_T15,
	R_TRIG_BST_S_T16, R_TRIG_BST_P_T16,
	R_TRIG_BST_S_T18, R_TRIG_BST_P_T18,
	
	// SEQUENCE TIME-OUT BALLASTING STOP
	R_TRIG_BSP_S_T01, R_TRIG_BSP_P_T01,
	R_TRIG_BSP_S_T03, R_TRIG_BSP_P_T03,
	R_TRIG_BSP_S_T04, R_TRIG_BSP_P_T04,
	R_TRIG_BSP_S_T05, R_TRIG_BSP_P_T05,
	R_TRIG_BSP_S_T07, R_TRIG_BSP_P_T07,
	R_TRIG_BSP_S_T08, R_TRIG_BSP_P_T08,
	R_TRIG_BSP_S_T09, R_TRIG_BSP_P_T09,
	R_TRIG_BSP_S_T10, R_TRIG_BSP_P_T10,
	R_TRIG_BSP_S_T12, R_TRIG_BSP_P_T12,
	
	// SEQUENCE TIME-OUT DEBALLASTING START
	
	R_TRIG_DST_S_T02, R_TRIG_DST_P_T02, 
	R_TRIG_DST_S_T03, R_TRIG_DST_P_T03, 
	R_TRIG_DST_S_T04, R_TRIG_DST_P_T04, 
	R_TRIG_DST_S_T05, R_TRIG_DST_P_T05, 
	R_TRIG_DST_S_T06, R_TRIG_DST_P_T06, 
	R_TRIG_DST_S_T07, R_TRIG_DST_P_T07, 
	R_TRIG_DST_S_T08, R_TRIG_DST_P_T08, 
	R_TRIG_DST_S_T09, R_TRIG_DST_P_T09, 
	
	// SEQUENCE TIME-OUT DEBALLASTING STOP
	R_TRIG_DSP_S_T01, R_TRIG_DSP_P_T01, 
	R_TRIG_DSP_S_T02, R_TRIG_DSP_P_T02, 
	R_TRIG_DSP_S_T03, R_TRIG_DSP_P_T03, 
	
	R_TRIG_DSP_S_T05, R_TRIG_DSP_P_T05, 
	R_TRIG_DSP_S_T06, R_TRIG_DSP_P_T06, 
	R_TRIG_DSP_S_T07, R_TRIG_DSP_P_T07, 
	
	// SEQUENCE TIME-OUT STRIPPING START
	R_TRIG_SST_S_T01,
	R_TRIG_SST_S_T02,
	R_TRIG_SST_S_T03,
	R_TRIG_SST_S_T04,
	R_TRIG_SST_S_T06,
	R_TRIG_SST_S_T07,
	R_TRIG_SST_S_T08,
	R_TRIG_SST_S_T09,
	
	// SEQUENCE TIME-OUT STRIPPING STOP
	R_TRIG_SSP_S_T01,
	R_TRIG_SSP_S_T02,
	R_TRIG_SSP_S_T03,
	R_TRIG_SSP_S_T04,
	R_TRIG_SSP_S_T06,
	R_TRIG_SSP_S_T07
	: R_TRIG; 
END_VAR

// EU
R_TRIG_B117A_STF(CLK:=B117A_STF);
R_TRIG_B117A_SPF(CLK:=B117A_SPF);
R_TRIG_B117B_STF(CLK:=B117B_STF);
R_TRIG_B117B_SPF(CLK:=B117B_SPF);
R_TRIG_XV1171A_OPF(CLK:=XV1171A_OPF);
R_TRIG_XV1171A_CLF(CLK:=XV1171A_CLF);
R_TRIG_XV1171B_OPF(CLK:=XV1171B_OPF);
R_TRIG_XV1171B_CLF(CLK:=XV1171B_CLF);
R_TRIG_B_117A_F(CLK:=B_117A_F);
R_TRIG_B_117A_OFF(CLK:=B_117A_OFF);
R_TRIG_B_117B_F(CLK:=B_117B_F);
R_TRIG_B_117B_OFF(CLK:=B_117B_OFF); R_TRIG_BLR_BYPASS(CLK:=BLR_BYPASS); R_TRIG_BLR_BOTH_F(CLK:=BLR_BOTH_F);
R_TRIG_PT_1121_HI(CLK:=PT_1121_HI); R_TRIG_PT_1121_LO(CLK:=PT_1121_LO); R_TRIG_PT_1121_LL(CLK:=PT_1121_LL); R_TRIG_LS_1111_LL(CLK:=LS_1111_LL); R_TRIG_LS_1141_HI(CLK:=LS_1141_HI); R_TRIG_ER_FAN_OFF(CLK:=ER_FAN_OFF);
R_TRIG_AIT_1121_HH(CLK:=AIT_1121_HH); R_TRIG_AIT_1121_HI(CLK:=AIT_1121_HI); R_TRIG_AIT_1122_HH(CLK:=AIT_1122_HH); R_TRIG_AIT_1122_HI(CLK:=AIT_1122_HI); R_TRIG_AIT_1123_HH(CLK:=AIT_1123_HH); R_TRIG_AIT_1123_HI(CLK:=AIT_1123_HI);
R_TRIG_TE_1111_HI(CLK:=TE_1111_HI); R_TRIG_TE_1111_LO(CLK:=TE_1111_LO); R_TRIG_TE_1111_LL(CLK:=TE_1111_LL); R_TRIG_CT_1111_LO(CLK:=CT_1111_LO); R_TRIG_CT_1111_LL(CLK:=CT_1111_LL);
R_TRIG_ZS_1112A_CL(CLK:=ZS_1112A_CL); R_TRIG_ZS_1112A_OP(CLK:=ZS_1112A_OP);
R_TRIG_ZS_1113A_CL(CLK:=ZS_1113A_CL); R_TRIG_ZS_1113A_OP(CLK:=ZS_1113A_OP);
R_TRIG_ZS_1114A_CL(CLK:=ZS_1114A_CL); R_TRIG_ZS_1114A_OP(CLK:=ZS_1114A_OP); 

// SWFU
R_TRIG_P171A_STF(CLK:=P171A_STF);
R_TRIG_P171A_SPF(CLK:=P171A_SPF);
R_TRIG_P171B_STF(CLK:=P171B_STF);
R_TRIG_P171B_SPF(CLK:=P171B_SPF);

R_TRIG_SWFP_BOTH_F(CLK:=SWFP_BOTH_F);
R_TRIG_P_171A_F(CLK:=P_171A_F);
R_TRIG_P_171A_OFF(CLK:=P_171A_OFF);
R_TRIG_P_171B_F(CLK:=P_171B_F);
R_TRIG_P_171B_OFF(CLK:=P_171B_OFF);

R_TRIG_PT_1721_HI(CLK:=PT_1721_HI);
R_TRIG_PT_1721_LO(CLK:=PT_1721_LO);
R_TRIG_PT_1721_LL(CLK:=PT_1721_LL);
R_TRIG_PT_1722_HH(CLK:=PT_1722_HH);
R_TRIG_PT_1722_HI(CLK:=PT_1722_HI);
R_TRIG_PT_1722_LO(CLK:=PT_1722_LO);

R_TRIG_SWFU_DP_HI(CLK:=SWFU_DP_HI);
R_TRIG_SWFU_DP_HH(CLK:=SWFU_DP_HH);

// INJECTION
R_TRIG_FCV1131_CF(CLK:=FCV1131_CF);
R_TRIG_FIT_1131_LO(CLK:=FIT_1131_LO);
R_TRIG_FIT_1131_LL(CLK:=FIT_1131_LL);
R_TRIG_RFS_1131(CLK:=RFS_1131);

R_TRIG_FCV2131_CF(CLK:=FCV2131_CF);
R_TRIG_FIT_2131_LO(CLK:=FIT_2131_LO);
R_TRIG_FIT_2131_LL(CLK:=FIT_2131_LL);
R_TRIG_RFS_2131(CLK:=RFS_2131);

// MAIN TRC
R_TRIG_FCV1211_CF(CLK:=FCV1211_CF);
R_TRIG_FIT_1211_HH(CLK:=FIT_1211_HH);
R_TRIG_FIT_1211_HI(CLK:=FIT_1211_HI);
R_TRIG_FIT_1211_LO(CLK:=FIT_1211_LO);

R_TRIG_FCV2211_CF(CLK:=FCV2211_CF);
R_TRIG_FIT_2211_HH(CLK:=FIT_2211_HH);
R_TRIG_FIT_2211_HI(CLK:=FIT_2211_HI);
R_TRIG_FIT_2211_LO(CLK:=FIT_2211_LO);

// NU
R_TRIG_P_132_TRIP(CLK:=P_132_TRIP);
R_TRIG_P132_STF(CLK:=P132_STF);
R_TRIG_P132_SPF(CLK:=P132_SPF);
R_TRIG_DPS_1321(CLK:=DPS_1321);

R_TRIG_P_232_TRIP(CLK:=P_232_TRIP); 
R_TRIG_P232_STF(CLK:=P232_STF);
R_TRIG_P232_SPF(CLK:=P232_SPF);
R_TRIG_DPS_2321(CLK:=DPS_2321);

R_TRIG_LIT_1311_HI(CLK:=LIT_1311_HI);
R_TRIG_LIT_1311_LO(CLK:=LIT_1311_LO);
R_TRIG_LIT_1311_LL(CLK:=LIT_1311_LL);

// RECTIFIER
R_TRIG_RF142A_STF(CLK:=RF142A_STF);
R_TRIG_RF142A_SPF(CLK:=RF142A_SPF);
R_TRIG_RF142B_STF(CLK:=RF142B_STF);
R_TRIG_RF142B_SPF(CLK:=RF142B_SPF);
R_TRIG_RF142C_STF(CLK:=RF142C_STF);
R_TRIG_RF142C_SPF(CLK:=RF142C_SPF);
R_TRIG_RF_142A_E(CLK:=RF_142A_E);
R_TRIG_RF_142B_E(CLK:=RF_142B_E);
R_TRIG_RF_142C_E(CLK:=RF_142C_E);
R_TRIG_RF_ALL_SPD(CLK:=RF_ALL_SPD);

R_TRIG_REC1001(CLK:=REC1001);
R_TRIG_REC1002(CLK:=REC1002);
R_TRIG_REC1003(CLK:=REC1003);
R_TRIG_REC1004(CLK:=REC1004);
R_TRIG_REC1005(CLK:=REC1005);
R_TRIG_REC1006(CLK:=REC1006);
R_TRIG_REC1007(CLK:=REC1007);
R_TRIG_REC1008(CLK:=REC1008);
R_TRIG_REC1009(CLK:=REC1009);
R_TRIG_REC1010(CLK:=REC1010);
R_TRIG_REC1011(CLK:=REC1011);
R_TRIG_REC1012(CLK:=REC1012);
R_TRIG_REC1013(CLK:=REC1013);
R_TRIG_REC1014(CLK:=REC1014);
R_TRIG_REC1015(CLK:=REC1015);
R_TRIG_REC1022(CLK:=REC1022);
R_TRIG_REC1023(CLK:=REC1023);
R_TRIG_REC1024(CLK:=REC1024);
R_TRIG_REC1025(CLK:=REC1025);
R_TRIG_REC1026(CLK:=REC1026);
R_TRIG_REC1032(CLK:=REC1032);
R_TRIG_REC1033(CLK:=REC1033);
R_TRIG_REC1017_HH(CLK:=REC1017_HH);
R_TRIG_REC1017_HI(CLK:=REC1017_HI);
R_TRIG_REC1018_HH(CLK:=REC1018_HH);
R_TRIG_REC1018_HI(CLK:=REC1018_HI);
R_TRIG_REC1019_HH(CLK:=REC1019_HH);
R_TRIG_REC1019_HI(CLK:=REC1019_HI);
R_TRIG_REC1020_HH(CLK:=REC1020_HH);
R_TRIG_REC1020_HI(CLK:=REC1020_HI);
R_TRIG_REC1021_HH(CLK:=REC1021_HH);
R_TRIG_REC1021_HI(CLK:=REC1021_HI);
R_TRIG_REC1027_HH(CLK:=REC1027_HH);
R_TRIG_REC1027_HI(CLK:=REC1027_HI);

R_TRIG_REC2001(CLK:=REC2001);
R_TRIG_REC2002(CLK:=REC2002);
R_TRIG_REC2003(CLK:=REC2003);
R_TRIG_REC2004(CLK:=REC2004);
R_TRIG_REC2005(CLK:=REC2005);
R_TRIG_REC2006(CLK:=REC2006);
R_TRIG_REC2007(CLK:=REC2007);
R_TRIG_REC2008(CLK:=REC2008);
R_TRIG_REC2009(CLK:=REC2009);
R_TRIG_REC2010(CLK:=REC2010);
R_TRIG_REC2011(CLK:=REC2011);
R_TRIG_REC2012(CLK:=REC2012);
R_TRIG_REC2013(CLK:=REC2013);
R_TRIG_REC2014(CLK:=REC2014);
R_TRIG_REC2015(CLK:=REC2015);
R_TRIG_REC2022(CLK:=REC2022);
R_TRIG_REC2023(CLK:=REC2023);
R_TRIG_REC2024(CLK:=REC2024);
R_TRIG_REC2025(CLK:=REC2025);
R_TRIG_REC2026(CLK:=REC2026);
R_TRIG_REC2032(CLK:=REC2032);
R_TRIG_REC2033(CLK:=REC2033);
R_TRIG_REC2017_HH(CLK:=REC2017_HH);
R_TRIG_REC2017_HI(CLK:=REC2017_HI);
R_TRIG_REC2018_HH(CLK:=REC2018_HH);
R_TRIG_REC2018_HI(CLK:=REC2018_HI);
R_TRIG_REC2019_HH(CLK:=REC2019_HH);
R_TRIG_REC2019_HI(CLK:=REC2019_HI);
R_TRIG_REC2020_HH(CLK:=REC2020_HH);
R_TRIG_REC2020_HI(CLK:=REC2020_HI);
R_TRIG_REC2021_HH(CLK:=REC2021_HH);
R_TRIG_REC2021_HI(CLK:=REC2021_HI);
R_TRIG_REC2027_HH(CLK:=REC2027_HH);
R_TRIG_REC2027_HI(CLK:=REC2027_HI);

R_TRIG_REC3001(CLK:=REC3001);
R_TRIG_REC3002(CLK:=REC3002);
R_TRIG_REC3003(CLK:=REC3003);
R_TRIG_REC3004(CLK:=REC3004);
R_TRIG_REC3005(CLK:=REC3005);
R_TRIG_REC3006(CLK:=REC3006);
R_TRIG_REC3007(CLK:=REC3007);
R_TRIG_REC3008(CLK:=REC3008);
R_TRIG_REC3009(CLK:=REC3009);
R_TRIG_REC3010(CLK:=REC3010);
R_TRIG_REC3011(CLK:=REC3011);
R_TRIG_REC3012(CLK:=REC3012);
R_TRIG_REC3013(CLK:=REC3013);
R_TRIG_REC3014(CLK:=REC3014);
R_TRIG_REC3015(CLK:=REC3015);
R_TRIG_REC3022(CLK:=REC3022);
R_TRIG_REC3023(CLK:=REC3023);
R_TRIG_REC3024(CLK:=REC3024);
R_TRIG_REC3025(CLK:=REC3025);
R_TRIG_REC3026(CLK:=REC3026);
R_TRIG_REC3032(CLK:=REC3032);
R_TRIG_REC3033(CLK:=REC3033);
R_TRIG_REC3017_HH(CLK:=REC3017_HH);
R_TRIG_REC3017_HI(CLK:=REC3017_HI);
R_TRIG_REC3018_HH(CLK:=REC3018_HH);
R_TRIG_REC3018_HI(CLK:=REC3018_HI);
R_TRIG_REC3019_HH(CLK:=REC3019_HH);
R_TRIG_REC3019_HI(CLK:=REC3019_HI);
R_TRIG_REC3020_HH(CLK:=REC3020_HH);
R_TRIG_REC3020_HI(CLK:=REC3020_HI);
R_TRIG_REC3021_HH(CLK:=REC3021_HH);
R_TRIG_REC3021_HI(CLK:=REC3021_HI);
R_TRIG_REC3027_HH(CLK:=REC3027_HH);
R_TRIG_REC3027_HI(CLK:=REC3027_HI);

// TRO
R_TRIG_AIT_151_E(CLK:=AIT_151_E);
R_TRIG_AIT_151_F(CLK:=AIT_151_F);
R_TRIG_AIT_251_E(CLK:=AIT_251_E);
R_TRIG_AIT_251_F(CLK:=AIT_251_F);

R_TRIG_BTRO_HH_S(CLK:=BTRO_HH_S);
R_TRIG_BTRO_HI_S(CLK:=BTRO_HI_S);
R_TRIG_BTRO_LO_S(CLK:=BTRO_LO_S);
R_TRIG_BTRO_LL_S(CLK:=BTRO_LL_S);
R_TRIG_DTRO_HH_S(CLK:=DTRO_HH_S);
R_TRIG_DTRO_HI_S(CLK:=DTRO_HI_S);

R_TRIG_BTRO_HH_P(CLK:=BTRO_HH_P);
R_TRIG_BTRO_HI_P(CLK:=BTRO_HI_P);
R_TRIG_BTRO_LO_P(CLK:=BTRO_LO_P);
R_TRIG_BTRO_LL_P(CLK:=BTRO_LL_P);
R_TRIG_DTRO_HH_P(CLK:=DTRO_HH_P);
R_TRIG_DTRO_HI_P(CLK:=DTRO_HI_P);

R_TRIG_STRO_HH(CLK:=STRO_HH);
R_TRIG_STRO_HI(CLK:=STRO_HI);


R_TRIG_LS_1901_HH(CLK:=LS_1901_HH);

// BALLAST SYSTEM
R_TRIG_WBP01_STF(CLK:=WBP01_STF);
R_TRIG_WBP01_SPF(CLK:=WBP01_SPF);
R_TRIG_WBP_01_AL(CLK:=WBP_01_AL);
R_TRIG_WBP_01_FAULT(CLK:=WBP_01_FAULT);

R_TRIG_WBP02_STF(CLK:=WBP02_STF);
R_TRIG_WBP02_SPF(CLK:=WBP02_SPF); 
R_TRIG_WBP_02_AL(CLK:=WBP_02_AL);
R_TRIG_WBP_02_FAULT(CLK:=WBP_02_FAULT);

R_TRIG_GSP01_STF(CLK:=GSP01_STF);
R_TRIG_GSP01_SPF(CLK:=GSP01_SPF);
R_TRIG_GSP_01_AL(CLK:=GSP_01_AL);
R_TRIG_GSP_01_FAULT(CLK:=GSP_01_FAULT);

R_TRIG_GSP02_STF(CLK:=GSP02_STF);
R_TRIG_GSP02_SPF(CLK:=GSP02_SPF); 
R_TRIG_GSP_02_AL(CLK:=GSP_02_AL);
R_TRIG_GSP_02_FAULT(CLK:=GSP_02_FAULT);

R_TRIG_SYS_BYPASS_1(CLK:=SYS_BYPASS_1);
R_TRIG_SYS_BYPASS_2(CLK:=SYS_BYPASS_2);
R_TRIG_SYS_BYPASS_3(CLK:=SYS_BYPASS_3);
R_TRIG_SYS_BYPASS_4(CLK:=SYS_BYPASS_4);

R_TRIG_BAL_VV_AL_S(CLK:=BAL_VV_AL_S);
R_TRIG_BAL_VV_AL_P(CLK:=BAL_VV_AL_P);

R_TRIG_DEBAL_VV_AL_S(CLK:=DEBAL_VV_AL_S);
R_TRIG_DEBAL_VV_AL_P(CLK:=DEBAL_VV_AL_P);

R_TRIG_STR_VV_AL_S(CLK:=STR_VV_AL_S);

R_TRIG_AP_LVL_LO(CLK:=AP_LVL_LO);
R_TRIG_AP_LVL_LL(CLK:=AP_LVL_LL);

R_GAS_LEAK_AL(CLK:=GAS_LEAK_AL);

// SD
R_TRIG_ESD(CLK:=ESD);
R_TRIG_PSD_11(CLK:=PSD_11);
R_TRIG_PSD_12(CLK:=PSD_12);

R_TRIG_PSD_21(CLK:=PSD_21);
R_TRIG_PSD_22(CLK:=PSD_22);

R_TRIG_PSD_31(CLK:=PSD_31);
R_TRIG_PSD_41(CLK:=PSD_41);
R_TRIG_PSD_42(CLK:=PSD_42);

// SYSTEM
R_TRIG_CC100_TEMP_HI(CLK:=CC100_TEMP_HI); R_TRIG_ESTOP_HMI(CLK:=ESTOP_HMI); R_TRIG_ESTOP_CC(CLK:=ESTOP_CC); R_TRIG_ESTOP_RF(CLK:=ESTOP_RF);
R_TRIG_DISABLE1(CLK:=DISABLE1); R_TRIG_DISABLE2(CLK:=DISABLE2); R_TRIG_DISABLE3(CLK:=DISABLE3); R_TRIG_DISABLE4(CLK:=DISABLE4);
R_TRIG_MM_AIT1121(CLK:=MM_AIT1121); R_TRIG_MM_AIT1122(CLK:=MM_AIT1122); R_TRIG_MM_AIT1123(CLK:=MM_AIT1123); R_TRIG_MM_REPAIR(CLK:=MM_REPAIR);

R_TRIG_MCC_100_OFF(CLK:=MCC_100_OFF); 
R_TRIG_PR_FAN_OFF(CLK:=PR_FAN_OFF);
R_TRIG_GPS_ALARM(CLK:=GPS_ALARM);

R_TRIG_RH_EU_AL(CLK:=RH_EU_AL);
R_TRIG_RH_AIT1121_AL(CLK:=RH_AIT1121_AL);
R_TRIG_RH_AIT1122_AL(CLK:=RH_AIT1122_AL);
R_TRIG_RH_AIT1123_AL(CLK:=RH_AIT1123_AL);
R_TRIG_RH_AIT151_AL(CLK:=RH_AIT151_AL);
R_TRIG_RH_AIT251_AL(CLK:=RH_AIT251_AL);


R_TRIG_RH_P132_AL(CLK:=RH_P132_AL);
R_TRIG_RH_P232_AL(CLK:=RH_P232_AL);

R_TRIG_RH_P171A_AL(CLK:=RH_P171A_AL);
R_TRIG_RH_P171B_AL(CLK:=RH_P171B_AL);

// SEQUENCE TIME-OUT BALLASTING START
R_TRIG_BST_S_T01(CLK:=BST_S_01.TIMEOUT);     R_TRIG_BST_P_T01(CLK:=BST_P_01.TIMEOUT);
R_TRIG_BST_S_T03(CLK:=BST_S_03.TIMEOUT);     R_TRIG_BST_P_T03(CLK:=BST_P_03.TIMEOUT);
R_TRIG_BST_S_T04(CLK:=BST_S_04.TIMEOUT);     R_TRIG_BST_P_T04(CLK:=BST_P_04.TIMEOUT);
R_TRIG_BST_S_T05(CLK:=BST_S_05.TIMEOUT);     R_TRIG_BST_P_T05(CLK:=BST_P_05.TIMEOUT);
R_TRIG_BST_S_T06(CLK:=BST_S_06.TIMEOUT);     R_TRIG_BST_P_T06(CLK:=BST_P_06.TIMEOUT);
R_TRIG_BST_S_T07(CLK:=BST_S_07.TIMEOUT);     R_TRIG_BST_P_T07(CLK:=BST_P_07.TIMEOUT);
R_TRIG_BST_S_T08(CLK:=BST_S_08.TIMEOUT);     R_TRIG_BST_P_T08(CLK:=BST_P_08.TIMEOUT);
R_TRIG_BST_S_T10(CLK:=BST_S_10.TIMEOUT);     R_TRIG_BST_P_T10(CLK:=BST_P_10.TIMEOUT);
R_TRIG_BST_S_T12(CLK:=BST_S_12.TIMEOUT);     R_TRIG_BST_P_T12(CLK:=BST_P_12.TIMEOUT);
R_TRIG_BST_S_T13(CLK:=BST_S_13.TIMEOUT);     R_TRIG_BST_P_T13(CLK:=BST_P_13.TIMEOUT);
R_TRIG_BST_S_T14(CLK:=BST_S_14.TIMEOUT);     R_TRIG_BST_P_T14(CLK:=BST_P_14.TIMEOUT);
R_TRIG_BST_S_T15(CLK:=BST_S_15.TIMEOUT);     R_TRIG_BST_P_T15(CLK:=BST_P_15.TIMEOUT);
R_TRIG_BST_S_T16(CLK:=BST_S_16.TIMEOUT);     R_TRIG_BST_P_T16(CLK:=BST_P_16.TIMEOUT);
R_TRIG_BST_S_T18(CLK:=BST_S_18.TIMEOUT);     R_TRIG_BST_P_T18(CLK:=BST_P_18.TIMEOUT);
                                                                                     
// SEQUENCE TIME-OUT BALLASTING STOP                                                 
R_TRIG_BSP_S_T01(CLK:=BSP_S_01.TIMEOUT);     R_TRIG_BSP_P_T01(CLK:=BSP_P_01.TIMEOUT);
R_TRIG_BSP_S_T03(CLK:=BSP_S_03.TIMEOUT);     R_TRIG_BSP_P_T03(CLK:=BSP_P_03.TIMEOUT);
R_TRIG_BSP_S_T04(CLK:=BSP_S_04.TIMEOUT);     R_TRIG_BSP_P_T04(CLK:=BSP_P_04.TIMEOUT);
R_TRIG_BSP_S_T05(CLK:=BSP_S_05.TIMEOUT);     R_TRIG_BSP_P_T05(CLK:=BSP_P_05.TIMEOUT);
R_TRIG_BSP_S_T07(CLK:=BSP_S_07.TIMEOUT);     R_TRIG_BSP_P_T07(CLK:=BSP_P_07.TIMEOUT);
R_TRIG_BSP_S_T08(CLK:=BSP_S_08.TIMEOUT);     R_TRIG_BSP_P_T08(CLK:=BSP_P_08.TIMEOUT);
R_TRIG_BSP_S_T09(CLK:=BSP_S_09.TIMEOUT);     R_TRIG_BSP_P_T09(CLK:=BSP_P_09.TIMEOUT);
R_TRIG_BSP_S_T10(CLK:=BSP_S_10.TIMEOUT);     R_TRIG_BSP_P_T10(CLK:=BSP_P_10.TIMEOUT);
R_TRIG_BSP_S_T12(CLK:=BSP_S_12.TIMEOUT);     R_TRIG_BSP_P_T12(CLK:=BSP_P_12.TIMEOUT);

// SEQUENCE TIME-OUT DEBALLASTING START

R_TRIG_DST_S_T02(CLK:=DST_S_02.TIMEOUT);     R_TRIG_DST_P_T02(CLK:=DST_P_02.TIMEOUT);
R_TRIG_DST_S_T03(CLK:=DST_S_03.TIMEOUT);     R_TRIG_DST_P_T03(CLK:=DST_P_03.TIMEOUT);
R_TRIG_DST_S_T04(CLK:=DST_S_04.TIMEOUT);     R_TRIG_DST_P_T04(CLK:=DST_P_04.TIMEOUT);
R_TRIG_DST_S_T05(CLK:=DST_S_05.TIMEOUT);     R_TRIG_DST_P_T05(CLK:=DST_P_05.TIMEOUT);
R_TRIG_DST_S_T06(CLK:=DST_S_06.TIMEOUT);     R_TRIG_DST_P_T06(CLK:=DST_P_06.TIMEOUT);
R_TRIG_DST_S_T07(CLK:=DST_S_07.TIMEOUT);     R_TRIG_DST_P_T07(CLK:=DST_P_07.TIMEOUT);
R_TRIG_DST_S_T08(CLK:=DST_S_08.TIMEOUT);     R_TRIG_DST_P_T08(CLK:=DST_P_08.TIMEOUT);
R_TRIG_DST_S_T09(CLK:=DST_S_09.TIMEOUT);     R_TRIG_DST_P_T09(CLK:=DST_P_09.TIMEOUT);
                                                                                     
// SEQUENCE TIME-OUT DEBALLASTING STOP                                               
R_TRIG_DSP_S_T01(CLK:=DSP_S_01.TIMEOUT);     R_TRIG_DSP_P_T01(CLK:=DSP_P_01.TIMEOUT);
R_TRIG_DSP_S_T02(CLK:=DSP_S_02.TIMEOUT);     R_TRIG_DSP_P_T02(CLK:=DSP_P_02.TIMEOUT);
R_TRIG_DSP_S_T03(CLK:=DSP_S_03.TIMEOUT);     R_TRIG_DSP_P_T03(CLK:=DSP_P_03.TIMEOUT);
R_TRIG_DSP_S_T05(CLK:=DSP_S_05.TIMEOUT);     R_TRIG_DSP_P_T05(CLK:=DSP_P_05.TIMEOUT);
R_TRIG_DSP_S_T06(CLK:=DSP_S_06.TIMEOUT);     R_TRIG_DSP_P_T06(CLK:=DSP_P_06.TIMEOUT);
R_TRIG_DSP_S_T07(CLK:=DSP_S_07.TIMEOUT);     R_TRIG_DSP_P_T07(CLK:=DSP_P_07.TIMEOUT);

// SEQUENCE TIME-OUT STRIPPING START
R_TRIG_SST_S_T01(CLK:=SST_S_01.TIMEOUT);
R_TRIG_SST_S_T02(CLK:=SST_S_02.TIMEOUT);
R_TRIG_SST_S_T03(CLK:=SST_S_03.TIMEOUT);
R_TRIG_SST_S_T04(CLK:=SST_S_04.TIMEOUT);
R_TRIG_SST_S_T06(CLK:=SST_S_06.TIMEOUT);
R_TRIG_SST_S_T07(CLK:=SST_S_07.TIMEOUT);
R_TRIG_SST_S_T08(CLK:=SST_S_08.TIMEOUT);
R_TRIG_SST_S_T09(CLK:=SST_S_09.TIMEOUT);

// SEQUENCE TIME-OUT STRIPPING STOP
R_TRIG_SSP_S_T01(CLK:=SSP_S_01.TIMEOUT);
R_TRIG_SSP_S_T02(CLK:=SSP_S_02.TIMEOUT);
R_TRIG_SSP_S_T03(CLK:=SSP_S_03.TIMEOUT);
R_TRIG_SSP_S_T04(CLK:=SSP_S_04.TIMEOUT);
R_TRIG_SSP_S_T06(CLK:=SSP_S_06.TIMEOUT);
R_TRIG_SSP_S_T07(CLK:=SSP_S_07.TIMEOUT);

END_PROGRAM

// Device/Application/Logic/0.ALARM/ALARM_BUZZER_2
PROGRAM ALARM_BUZZER_2
VAR
	BUZZER_ON : BOOL;
	SR_0 : SR;
	SR_1 : SR;
	SR_2 : SR;
	SR_3 : SR;
	SR_4 : SR;
	SR_5 : SR;
	SR_6 : SR;
	SR_7 : SR;
	SR_8 : SR;
	SR_9 : SR;
	SR_10 : SR;
	SR_11 : SR;
	SR_12 : SR;
	SR_13 : SR;
	// SENSOR FAULT
	GROUP01, GROUP01_1, GROUP01_2 : BOOL;		
	// EU
    GROUP02, GROUP02_1, GROUP02_2 : BOOL;
	// SWFU	
	GROUP03 : BOOL;
	// INJECTION
	GROUP04 : BOOL;
	// MAIN TRC
	GROUP05 : BOOL;
	// NU	
	GROUP06 : BOOL;
	// RECTIFIER
	GROUP07, GROUP07_1, GROUP07_2, GROUP07_3, GROUP07_4, GROUP07_5, GROUP07_6, GROUP07_7, GROUP07_8 : BOOL;
	// FU
	GROUP08, GROUP08_1, GROUP08_2 : BOOL;
	// TRO
	GROUP09 : BOOL;
	// BALLAST SYSTEM
	GROUP10, GROUP10_1, GROUP10_2 : BOOL;
	// SD
	GROUP11 : BOOL;
	// SYSTEM
	GROUP12, GROUP12_1, GROUP12_2, GROUP12_3, GROUP12_4, GROUP12_5 : BOOL; 
	// SEQUENCE FAIL
	GROUP13, GROUP13_1, GROUP13_2, GROUP13_3, GROUP13_4, GROUP13_5, GROUP13_6, GROUP13_7, GROUP13_8, GROUP13_9, GROUP13_10,	GROUP13_11, GROUP13_12, GROUP13_13, GROUP13_14 : BOOL;
END_VAR

SR_0(SET1:= BUZZER_ON, RESET := MP_SOUNDOFF OR BWTS_002, Q1=> BWTS_007);
 
BUZZER_ON :=
GROUP01 OR GROUP02 OR GROUP03 OR GROUP04 OR GROUP05 OR GROUP06 OR GROUP07 OR GROUP08 OR GROUP09 OR GROUP10 OR GROUP11 OR GROUP12 OR GROUP13;

// SENSOR FAIL

// EU
GROUP02 := GROUP02_1 OR GROUP02_2;
GROUP02_1 :=
ALARM_BUZZER_1.R_TRIG_B117A_STF.Q OR ALARM_BUZZER_1.R_TRIG_B117A_SPF.Q OR ALARM_BUZZER_1.R_TRIG_B117B_STF.Q OR ALARM_BUZZER_1.R_TRIG_B117B_SPF.Q OR ALARM_BUZZER_1.R_TRIG_XV1171A_OPF.Q OR
ALARM_BUZZER_1.R_TRIG_XV1171A_CLF.Q OR ALARM_BUZZER_1.R_TRIG_XV1171B_OPF.Q OR ALARM_BUZZER_1.R_TRIG_XV1171B_CLF.Q OR ALARM_BUZZER_1.R_TRIG_B_117A_F.Q OR ALARM_BUZZER_1.R_TRIG_B_117B_F.Q OR
ALARM_BUZZER_1.R_TRIG_B_117A_OFF.Q OR ALARM_BUZZER_1.R_TRIG_B_117B_OFF.Q OR ALARM_BUZZER_1.R_TRIG_BLR_BYPASS.Q OR ALARM_BUZZER_1.R_TRIG_BLR_BOTH_F.Q OR ALARM_BUZZER_1.R_TRIG_PT_1121_HI.Q OR
ALARM_BUZZER_1.R_TRIG_PT_1121_LO.Q OR ALARM_BUZZER_1.R_TRIG_PT_1121_LL.Q OR ALARM_BUZZER_1.R_TRIG_LS_1111_LL.Q OR ALARM_BUZZER_1.R_TRIG_LS_1141_HI.Q OR ALARM_BUZZER_1.R_TRIG_ER_FAN_OFF.Q OR 
ALARM_BUZZER_1.R_TRIG_AIT_1121_HH.Q OR ALARM_BUZZER_1.R_TRIG_AIT_1121_HI.Q OR ALARM_BUZZER_1.R_TRIG_AIT_1122_HH.Q OR ALARM_BUZZER_1.R_TRIG_AIT_1122_HI.Q OR ALARM_BUZZER_1.R_TRIG_AIT_1123_HH.Q;
GROUP02_2 :=
ALARM_BUZZER_1.R_TRIG_AIT_1123_HI.Q OR ALARM_BUZZER_1.R_TRIG_TE_1111_HI.Q OR ALARM_BUZZER_1.R_TRIG_TE_1111_LO.Q OR ALARM_BUZZER_1.R_TRIG_TE_1111_LL.Q OR ALARM_BUZZER_1.R_TRIG_CT_1111_LO.Q OR
ALARM_BUZZER_1.R_TRIG_CT_1111_LL.Q OR 
ALARM_BUZZER_1.R_TRIG_ZS_1112A_CL.Q OR ALARM_BUZZER_1.R_TRIG_ZS_1112A_OP.Q OR 
ALARM_BUZZER_1.R_TRIG_ZS_1113A_CL.Q OR ALARM_BUZZER_1.R_TRIG_ZS_1113A_OP.Q OR
ALARM_BUZZER_1.R_TRIG_ZS_1114A_CL.Q OR ALARM_BUZZER_1.R_TRIG_ZS_1114A_OP.Q;

// SWFU
GROUP03 :=
ALARM_BUZZER_1.R_TRIG_P171A_STF.Q OR ALARM_BUZZER_1.R_TRIG_P171A_SPF.Q OR ALARM_BUZZER_1.R_TRIG_P171B_STF.Q OR ALARM_BUZZER_1.R_TRIG_P171B_SPF.Q OR ALARM_BUZZER_1.R_TRIG_SWFP_BOTH_F.Q OR
ALARM_BUZZER_1.R_TRIG_P_171A_F.Q OR ALARM_BUZZER_1.R_TRIG_P_171B_F.Q OR ALARM_BUZZER_1.R_TRIG_P_171A_OFF.Q OR ALARM_BUZZER_1.R_TRIG_P_171B_OFF.Q OR ALARM_BUZZER_1.R_TRIG_PT_1721_HI.Q OR
ALARM_BUZZER_1.R_TRIG_PT_1721_LO.Q OR ALARM_BUZZER_1.R_TRIG_PT_1721_LL.Q OR ALARM_BUZZER_1.R_TRIG_PT_1722_HH.Q OR ALARM_BUZZER_1.R_TRIG_PT_1722_HI.Q OR ALARM_BUZZER_1.R_TRIG_PT_1722_LO.Q OR
ALARM_BUZZER_1.R_TRIG_SWFU_DP_HI.Q OR  ALARM_BUZZER_1.R_TRIG_SWFU_DP_HH.Q;

// INJECTION
GROUP04 := 
ALARM_BUZZER_1.R_TRIG_FCV1131_CF.Q OR ALARM_BUZZER_1.R_TRIG_RFS_1131.Q OR ALARM_BUZZER_1.R_TRIG_FIT_1131_LO.Q OR  ALARM_BUZZER_1.R_TRIG_FIT_1131_LL.Q OR 
ALARM_BUZZER_1.R_TRIG_FCV2131_CF.Q OR ALARM_BUZZER_1.R_TRIG_RFS_2131.Q OR ALARM_BUZZER_1.R_TRIG_FIT_2131_LO.Q OR  ALARM_BUZZER_1.R_TRIG_FIT_2131_LL.Q;


// MAIN TRC
GROUP05 :=
ALARM_BUZZER_1.R_TRIG_FCV1211_CF.Q OR ALARM_BUZZER_1.R_TRIG_FIT_1211_HH.Q OR ALARM_BUZZER_1.R_TRIG_FIT_1211_HI.Q OR ALARM_BUZZER_1.R_TRIG_FIT_1211_LO.Q OR 
ALARM_BUZZER_1.R_TRIG_FCV2211_CF.Q OR ALARM_BUZZER_1.R_TRIG_FIT_2211_HH.Q OR ALARM_BUZZER_1.R_TRIG_FIT_2211_HI.Q OR ALARM_BUZZER_1.R_TRIG_FIT_2211_LO.Q
;

// NU
GROUP06 := 
ALARM_BUZZER_1.R_TRIG_P_132_TRIP.Q OR ALARM_BUZZER_1.R_TRIG_P132_STF.Q OR  ALARM_BUZZER_1.R_TRIG_P132_SPF.Q OR ALARM_BUZZER_1.R_TRIG_DPS_1321.Q OR
ALARM_BUZZER_1.R_TRIG_P_232_TRIP.Q OR ALARM_BUZZER_1.R_TRIG_P232_STF.Q OR  ALARM_BUZZER_1.R_TRIG_P232_SPF.Q OR ALARM_BUZZER_1.R_TRIG_DPS_2321.Q OR
ALARM_BUZZER_1.R_TRIG_LIT_1311_HI.Q OR  ALARM_BUZZER_1.R_TRIG_LIT_1311_LO.Q OR  ALARM_BUZZER_1.R_TRIG_LIT_1311_LL.Q;

// RECTIFIER
GROUP07 := GROUP07_1 OR GROUP07_2 OR GROUP07_3 OR GROUP07_4 OR GROUP07_5 OR GROUP07_6; 
GROUP07_1 :=
ALARM_BUZZER_1.R_TRIG_RF142A_STF.Q OR ALARM_BUZZER_1.R_TRIG_RF142A_SPF.Q OR ALARM_BUZZER_1.R_TRIG_RF142B_STF.Q OR ALARM_BUZZER_1.R_TRIG_RF142B_SPF.Q OR 
ALARM_BUZZER_1.R_TRIG_RF_142A_E.Q OR ALARM_BUZZER_1.R_TRIG_RF_142B_E.Q OR ALARM_BUZZER_1.R_TRIG_RF_ALL_SPD.Q;

GROUP07_2 :=
ALARM_BUZZER_1.R_TRIG_REC1001.Q OR ALARM_BUZZER_1.R_TRIG_REC1002.Q OR ALARM_BUZZER_1.R_TRIG_REC1003.Q OR ALARM_BUZZER_1.R_TRIG_REC1004.Q OR ALARM_BUZZER_1.R_TRIG_REC1005.Q OR
ALARM_BUZZER_1.R_TRIG_REC1006.Q OR ALARM_BUZZER_1.R_TRIG_REC1007.Q OR ALARM_BUZZER_1.R_TRIG_REC1008.Q OR ALARM_BUZZER_1.R_TRIG_REC1009.Q OR ALARM_BUZZER_1.R_TRIG_REC1010.Q OR
ALARM_BUZZER_1.R_TRIG_REC1011.Q OR ALARM_BUZZER_1.R_TRIG_REC1012.Q OR ALARM_BUZZER_1.R_TRIG_REC1013.Q OR ALARM_BUZZER_1.R_TRIG_REC1014.Q OR ALARM_BUZZER_1.R_TRIG_REC1015.Q OR
ALARM_BUZZER_1.R_TRIG_REC1022.Q OR ALARM_BUZZER_1.R_TRIG_REC1023.Q OR ALARM_BUZZER_1.R_TRIG_REC1024.Q OR ALARM_BUZZER_1.R_TRIG_REC1025.Q OR ALARM_BUZZER_1.R_TRIG_REC1026.Q OR
ALARM_BUZZER_1.R_TRIG_REC1032.Q OR ALARM_BUZZER_1.R_TRIG_REC1033.Q;

GROUP07_3 :=
ALARM_BUZZER_1.R_TRIG_REC1017_HH.Q OR ALARM_BUZZER_1.R_TRIG_REC1017_HI.Q OR ALARM_BUZZER_1.R_TRIG_REC1018_HH.Q OR ALARM_BUZZER_1.R_TRIG_REC1018_HI.Q OR
ALARM_BUZZER_1.R_TRIG_REC1019_HH.Q OR ALARM_BUZZER_1.R_TRIG_REC1019_HI.Q OR ALARM_BUZZER_1.R_TRIG_REC1020_HH.Q OR ALARM_BUZZER_1.R_TRIG_REC1020_HI.Q OR
ALARM_BUZZER_1.R_TRIG_REC1021_HH.Q OR ALARM_BUZZER_1.R_TRIG_REC1021_HI.Q OR ALARM_BUZZER_1.R_TRIG_REC1027_HH.Q OR ALARM_BUZZER_1.R_TRIG_REC1027_HI.Q;

GROUP07_4 := 
ALARM_BUZZER_1.R_TRIG_REC2001.Q OR ALARM_BUZZER_1.R_TRIG_REC2002.Q OR ALARM_BUZZER_1.R_TRIG_REC2003.Q OR ALARM_BUZZER_1.R_TRIG_REC2004.Q OR ALARM_BUZZER_1.R_TRIG_REC2005.Q OR
ALARM_BUZZER_1.R_TRIG_REC2006.Q OR ALARM_BUZZER_1.R_TRIG_REC2007.Q OR ALARM_BUZZER_1.R_TRIG_REC2008.Q OR ALARM_BUZZER_1.R_TRIG_REC2009.Q OR ALARM_BUZZER_1.R_TRIG_REC2010.Q OR
ALARM_BUZZER_1.R_TRIG_REC2011.Q OR ALARM_BUZZER_1.R_TRIG_REC2012.Q OR ALARM_BUZZER_1.R_TRIG_REC2013.Q OR ALARM_BUZZER_1.R_TRIG_REC2014.Q OR ALARM_BUZZER_1.R_TRIG_REC2015.Q OR
ALARM_BUZZER_1.R_TRIG_REC2022.Q OR ALARM_BUZZER_1.R_TRIG_REC2023.Q OR ALARM_BUZZER_1.R_TRIG_REC2024.Q OR ALARM_BUZZER_1.R_TRIG_REC2025.Q OR ALARM_BUZZER_1.R_TRIG_REC2026.Q OR
ALARM_BUZZER_1.R_TRIG_REC2032.Q OR ALARM_BUZZER_1.R_TRIG_REC2033.Q;

GROUP07_5 :=
ALARM_BUZZER_1.R_TRIG_REC2017_HH.Q OR ALARM_BUZZER_1.R_TRIG_REC2017_HI.Q OR ALARM_BUZZER_1.R_TRIG_REC2018_HH.Q OR ALARM_BUZZER_1.R_TRIG_REC2018_HI.Q OR
ALARM_BUZZER_1.R_TRIG_REC2019_HH.Q OR ALARM_BUZZER_1.R_TRIG_REC2019_HI.Q OR ALARM_BUZZER_1.R_TRIG_REC2020_HH.Q OR ALARM_BUZZER_1.R_TRIG_REC2020_HI.Q OR
ALARM_BUZZER_1.R_TRIG_REC2021_HH.Q OR ALARM_BUZZER_1.R_TRIG_REC2021_HI.Q OR ALARM_BUZZER_1.R_TRIG_REC2027_HH.Q OR ALARM_BUZZER_1.R_TRIG_REC2027_HI.Q;

GROUP07_7 :=
ALARM_BUZZER_1.R_TRIG_REC3017_HH.Q OR ALARM_BUZZER_1.R_TRIG_REC3017_HI.Q OR ALARM_BUZZER_1.R_TRIG_REC3018_HH.Q OR ALARM_BUZZER_1.R_TRIG_REC3018_HI.Q OR
ALARM_BUZZER_1.R_TRIG_REC3019_HH.Q OR ALARM_BUZZER_1.R_TRIG_REC3019_HI.Q OR ALARM_BUZZER_1.R_TRIG_REC3020_HH.Q OR ALARM_BUZZER_1.R_TRIG_REC3020_HI.Q OR
ALARM_BUZZER_1.R_TRIG_REC3021_HH.Q OR ALARM_BUZZER_1.R_TRIG_REC3021_HI.Q OR ALARM_BUZZER_1.R_TRIG_REC3027_HH.Q OR ALARM_BUZZER_1.R_TRIG_REC3027_HI.Q;

// TRO
GROUP09 :=
ALARM_BUZZER_1.R_TRIG_BTRO_HH_S.Q OR ALARM_BUZZER_1.R_TRIG_BTRO_HI_S.Q OR ALARM_BUZZER_1.R_TRIG_BTRO_LO_S.Q OR ALARM_BUZZER_1.R_TRIG_BTRO_LL_S.Q OR
ALARM_BUZZER_1.R_TRIG_BTRO_HH_P.Q OR ALARM_BUZZER_1.R_TRIG_BTRO_HI_P.Q OR ALARM_BUZZER_1.R_TRIG_BTRO_LO_P.Q OR ALARM_BUZZER_1.R_TRIG_BTRO_LL_P.Q OR

ALARM_BUZZER_1.R_TRIG_DTRO_HH_S.Q OR ALARM_BUZZER_1.R_TRIG_DTRO_HI_S.Q OR ALARM_BUZZER_1.R_TRIG_DTRO_HH_P.Q OR ALARM_BUZZER_1.R_TRIG_DTRO_HI_P.Q OR 
ALARM_BUZZER_1.R_TRIG_STRO_HH.Q OR ALARM_BUZZER_1.R_TRIG_STRO_HI.Q OR  
ALARM_BUZZER_1.R_TRIG_AIT_151_E.Q OR ALARM_BUZZER_1.R_TRIG_AIT_151_F.Q OR ALARM_BUZZER_1.R_TRIG_AIT_251_E.Q OR ALARM_BUZZER_1.R_TRIG_AIT_251_F.Q OR
ALARM_BUZZER_1.R_TRIG_LS_1901_HH.Q
;

// BALLAST SYSTEM
GROUP10 := GROUP10_1 OR GROUP10_2; 

GROUP10_1 := 
ALARM_BUZZER_1.R_TRIG_WBP01_STF.Q OR ALARM_BUZZER_1.R_TRIG_WBP01_SPF.Q OR ALARM_BUZZER_1.R_TRIG_WBP02_STF.Q OR ALARM_BUZZER_1.R_TRIG_WBP02_SPF.Q OR 
ALARM_BUZZER_1.R_TRIG_WBP_01_AL.Q OR ALARM_BUZZER_1.R_TRIG_WBP_02_AL.Q OR ALARM_BUZZER_1.R_TRIG_WBP_01_FAULT.Q OR ALARM_BUZZER_1.R_TRIG_WBP_02_FAULT.Q OR
ALARM_BUZZER_1.R_TRIG_GSP01_STF.Q OR ALARM_BUZZER_1.R_TRIG_GSP01_SPF.Q OR ALARM_BUZZER_1.R_TRIG_GSP02_STF.Q OR ALARM_BUZZER_1.R_TRIG_GSP02_SPF.Q OR 
ALARM_BUZZER_1.R_TRIG_GSP_01_AL.Q OR ALARM_BUZZER_1.R_TRIG_GSP_02_AL.Q OR ALARM_BUZZER_1.R_TRIG_GSP_01_FAULT.Q OR ALARM_BUZZER_1.R_TRIG_GSP_02_FAULT.Q OR
ALARM_BUZZER_1.R_TRIG_SYS_BYPASS_1.Q OR ALARM_BUZZER_1.R_TRIG_SYS_BYPASS_2.Q OR ALARM_BUZZER_1.R_TRIG_SYS_BYPASS_3.Q OR ALARM_BUZZER_1.R_TRIG_SYS_BYPASS_4.Q OR
ALARM_BUZZER_1.R_TRIG_BAL_VV_AL_S.Q OR ALARM_BUZZER_1.R_TRIG_BAL_VV_AL_P.Q OR 
ALARM_BUZZER_1.R_TRIG_DEBAL_VV_AL_S.Q OR ALARM_BUZZER_1.R_TRIG_DEBAL_VV_AL_P.Q OR
ALARM_BUZZER_1.R_TRIG_STR_VV_AL_S.Q OR 
ALARM_BUZZER_1.R_TRIG_AP_LVL_LO.Q OR ALARM_BUZZER_1.R_TRIG_AP_LVL_LL.Q;

GROUP10_2 :=
ALARM_BUZZER_1.R_FU_BYPASS_1.Q OR ALARM_BUZZER_1.R_FU_BYPASS_2.Q OR ALARM_BUZZER_1.R_FU_BYPASS_3.Q OR ALARM_BUZZER_1.R_GAS_LEAK_AL.Q;

// SD
GROUP11 := 
ALARM_BUZZER_1.R_TRIG_ESD.Q OR ALARM_BUZZER_1.R_TRIG_PSD_11.Q OR ALARM_BUZZER_1.R_TRIG_PSD_12.Q OR
ALARM_BUZZER_1.R_TRIG_PSD_21.Q OR ALARM_BUZZER_1.R_TRIG_PSD_22.Q OR
ALARM_BUZZER_1.R_TRIG_PSD_31.Q OR ALARM_BUZZER_1.R_TRIG_PSD_41.Q OR ALARM_BUZZER_1.R_TRIG_PSD_42.Q;

// SYSTEM
GROUP12 := GROUP12_1 OR GROUP12_2 OR GROUP12_3 OR GROUP12_4; 

GROUP12_1 := 
ALARM_BUZZER_1.R_TRIG_DISABLE1.Q OR ALARM_BUZZER_1.R_TRIG_DISABLE2.Q OR ALARM_BUZZER_1.R_TRIG_DISABLE3.Q OR ALARM_BUZZER_1.R_TRIG_DISABLE4.Q OR
ALARM_BUZZER_1.R_TRIG_MM_AIT1121.Q OR ALARM_BUZZER_1.R_TRIG_MM_AIT1122.Q OR ALARM_BUZZER_1.R_TRIG_MM_AIT1123.Q OR ALARM_BUZZER_1.R_TRIG_MM_REPAIR.Q;

GROUP12_2 :=
ALARM_BUZZER_1.R_TRIG_GPS_ALARM.Q
;

GROUP12_4 :=
ALARM_BUZZER_1.R_TRIG_MCC_100_OFF.Q OR ALARM_BUZZER_1.R_TRIG_PR_FAN_OFF.Q OR
ALARM_BUZZER_1.R_TRIG_CC100_TEMP_HI.Q OR ALARM_BUZZER_1.R_TRIG_ESTOP_HMI.Q OR ALARM_BUZZER_1.R_TRIG_ESTOP_CC.Q OR ALARM_BUZZER_1.R_TRIG_ESTOP_RF.Q OR
ALARM_BUZZER_1.R_TRIG_RH_EU_AL.Q OR ALARM_BUZZER_1.R_TRIG_RH_AIT1121_AL.Q OR ALARM_BUZZER_1.R_TRIG_RH_AIT1122_AL.Q OR ALARM_BUZZER_1.R_TRIG_RH_AIT1123_AL.Q OR
ALARM_BUZZER_1.R_TRIG_RH_AIT151_AL.Q OR ALARM_BUZZER_1.R_TRIG_RH_AIT251_AL.Q OR 
ALARM_BUZZER_1.R_TRIG_RH_P171A_AL.Q OR ALARM_BUZZER_1.R_TRIG_RH_P171B_AL.Q OR
ALARM_BUZZER_1.R_TRIG_RH_P132_AL.Q OR ALARM_BUZZER_1.R_TRIG_RH_P232_AL.Q; 

// SEQUENCE FAIL
GROUP13 := GROUP13_1 OR GROUP13_2 OR GROUP13_3 OR GROUP13_4 OR GROUP13_5 OR GROUP13_6 OR GROUP13_7 OR GROUP13_8 OR GROUP13_9 OR GROUP13_10 OR GROUP13_11 OR GROUP13_12 OR GROUP13_13 OR GROUP13_14; 

// SEQUENCE FAIL BALLASTING START STBD
GROUP13_1 := 
ALARM_BUZZER_1.R_TRIG_BST_S_T01.Q OR

ALARM_BUZZER_1.R_TRIG_BST_S_T03.Q OR
ALARM_BUZZER_1.R_TRIG_BST_S_T04.Q OR
ALARM_BUZZER_1.R_TRIG_BST_S_T05.Q OR 
ALARM_BUZZER_1.R_TRIG_BST_S_T06.Q OR
ALARM_BUZZER_1.R_TRIG_BST_S_T07.Q OR
ALARM_BUZZER_1.R_TRIG_BST_S_T08.Q OR

ALARM_BUZZER_1.R_TRIG_BST_S_T10.Q OR

ALARM_BUZZER_1.R_TRIG_BST_S_T12.Q OR
ALARM_BUZZER_1.R_TRIG_BST_S_T13.Q OR
ALARM_BUZZER_1.R_TRIG_BST_S_T14.Q OR
ALARM_BUZZER_1.R_TRIG_BST_S_T15.Q OR
ALARM_BUZZER_1.R_TRIG_BST_S_T16.Q OR

ALARM_BUZZER_1.R_TRIG_BST_S_T18.Q;
 
// SEQUENCE FAIL BALLASTING STOP STBD
GROUP13_2 :=
ALARM_BUZZER_1.R_TRIG_BSP_S_T01.Q OR

ALARM_BUZZER_1.R_TRIG_BSP_S_T03.Q OR
ALARM_BUZZER_1.R_TRIG_BSP_S_T04.Q OR
ALARM_BUZZER_1.R_TRIG_BSP_S_T05.Q OR

ALARM_BUZZER_1.R_TRIG_BSP_S_T07.Q OR
ALARM_BUZZER_1.R_TRIG_BSP_S_T08.Q OR
ALARM_BUZZER_1.R_TRIG_BSP_S_T09.Q OR
ALARM_BUZZER_1.R_TRIG_BSP_S_T10.Q OR

ALARM_BUZZER_1.R_TRIG_BSP_S_T12.Q;

// SEQUENCE FAIL BALLASTING START PORT
GROUP13_3 :=
ALARM_BUZZER_1.R_TRIG_BST_P_T01.Q OR

ALARM_BUZZER_1.R_TRIG_BST_P_T03.Q OR
ALARM_BUZZER_1.R_TRIG_BST_P_T04.Q OR
ALARM_BUZZER_1.R_TRIG_BST_P_T05.Q OR
ALARM_BUZZER_1.R_TRIG_BST_P_T06.Q OR
ALARM_BUZZER_1.R_TRIG_BST_P_T07.Q OR
ALARM_BUZZER_1.R_TRIG_BST_P_T08.Q OR

ALARM_BUZZER_1.R_TRIG_BST_P_T10.Q OR

ALARM_BUZZER_1.R_TRIG_BST_P_T12.Q OR
ALARM_BUZZER_1.R_TRIG_BST_P_T13.Q OR
ALARM_BUZZER_1.R_TRIG_BST_P_T14.Q OR
ALARM_BUZZER_1.R_TRIG_BST_P_T15.Q OR
ALARM_BUZZER_1.R_TRIG_BST_P_T16.Q OR

ALARM_BUZZER_1.R_TRIG_BST_P_T18.Q; 

// SEQUENCE FAIL BALLASTING STOP PORT
GROUP13_4 :=
ALARM_BUZZER_1.R_TRIG_BSP_P_T01.Q OR

ALARM_BUZZER_1.R_TRIG_BSP_P_T03.Q OR
ALARM_BUZZER_1.R_TRIG_BSP_P_T04.Q OR
ALARM_BUZZER_1.R_TRIG_BSP_P_T05.Q OR

ALARM_BUZZER_1.R_TRIG_BSP_P_T07.Q OR
ALARM_BUZZER_1.R_TRIG_BSP_P_T08.Q OR
ALARM_BUZZER_1.R_TRIG_BSP_P_T09.Q OR
ALARM_BUZZER_1.R_TRIG_BSP_P_T10.Q OR

ALARM_BUZZER_1.R_TRIG_BSP_P_T12.Q;

// SEQUENCE FAIL DEBALLASTING START STBD
GROUP13_5 :=

ALARM_BUZZER_1.R_TRIG_DST_S_T02.Q OR
ALARM_BUZZER_1.R_TRIG_DST_S_T03.Q OR
ALARM_BUZZER_1.R_TRIG_DST_S_T04.Q OR
ALARM_BUZZER_1.R_TRIG_DST_S_T05.Q OR
ALARM_BUZZER_1.R_TRIG_DST_S_T06.Q OR
ALARM_BUZZER_1.R_TRIG_DST_S_T07.Q OR
ALARM_BUZZER_1.R_TRIG_DST_S_T08.Q OR
ALARM_BUZZER_1.R_TRIG_DST_S_T09.Q;

// SEQUENCE FAIL DEBALLASTING STOP STBD
GROUP13_6 :=
ALARM_BUZZER_1.R_TRIG_DSP_S_T01.Q OR
ALARM_BUZZER_1.R_TRIG_DSP_S_T02.Q OR
ALARM_BUZZER_1.R_TRIG_DSP_S_T03.Q OR

ALARM_BUZZER_1.R_TRIG_DSP_S_T05.Q OR
ALARM_BUZZER_1.R_TRIG_DSP_S_T06.Q OR
ALARM_BUZZER_1.R_TRIG_DSP_S_T07.Q;

// SEQUENCE FAIL DEBALLASTING START PORT
GROUP13_7 :=

ALARM_BUZZER_1.R_TRIG_DST_P_T02.Q OR
ALARM_BUZZER_1.R_TRIG_DST_P_T03.Q OR
ALARM_BUZZER_1.R_TRIG_DST_P_T04.Q OR
ALARM_BUZZER_1.R_TRIG_DST_P_T05.Q OR
ALARM_BUZZER_1.R_TRIG_DST_P_T06.Q OR
ALARM_BUZZER_1.R_TRIG_DST_P_T07.Q OR
ALARM_BUZZER_1.R_TRIG_DST_P_T08.Q OR
ALARM_BUZZER_1.R_TRIG_DST_P_T09.Q;

// SEQUENCE FAIL DEBALLASTING STOP PORT
GROUP13_8 :=
ALARM_BUZZER_1.R_TRIG_DSP_P_T01.Q OR
ALARM_BUZZER_1.R_TRIG_DSP_P_T02.Q OR
ALARM_BUZZER_1.R_TRIG_DSP_P_T03.Q OR

ALARM_BUZZER_1.R_TRIG_DSP_P_T05.Q OR
ALARM_BUZZER_1.R_TRIG_DSP_P_T06.Q OR
ALARM_BUZZER_1.R_TRIG_DSP_P_T07.Q;

// SEQUENCE FAIL STRIPPING START STBD
GROUP13_9 :=
ALARM_BUZZER_1.R_TRIG_SST_S_T01.Q OR
ALARM_BUZZER_1.R_TRIG_SST_S_T02.Q OR
ALARM_BUZZER_1.R_TRIG_SST_S_T03.Q OR
ALARM_BUZZER_1.R_TRIG_SST_S_T04.Q OR

ALARM_BUZZER_1.R_TRIG_SST_S_T06.Q OR
ALARM_BUZZER_1.R_TRIG_SST_S_T07.Q OR
ALARM_BUZZER_1.R_TRIG_SST_S_T08.Q OR
ALARM_BUZZER_1.R_TRIG_SST_S_T09.Q;

// SEQUENCE FAIL STRIPPING STOP STBD
GROUP13_10 :=
ALARM_BUZZER_1.R_TRIG_SSP_S_T01.Q OR
ALARM_BUZZER_1.R_TRIG_SSP_S_T02.Q OR
ALARM_BUZZER_1.R_TRIG_SSP_S_T03.Q OR
ALARM_BUZZER_1.R_TRIG_SSP_S_T04.Q OR

ALARM_BUZZER_1.R_TRIG_SSP_S_T06.Q OR
ALARM_BUZZER_1.R_TRIG_SSP_S_T07.Q;

END_PROGRAM

// Device/Application/Logic/0.ALARM/ALARM_COMMON
PROGRAM ALARM_COMMON
VAR
	SR_0 : SR;
	SECOND_FAULT : BOOL;
	TOF_0 : TOF;
	
	GROUP01 : BOOL;	// SENSOR FAULT
	GROUP02, GROUP02_1, GROUP02_2 : BOOL;	// EU
	GROUP03 : BOOL;	// SWFU
	GROUP04 : BOOL;	// INJECTION
	GROUP05 : BOOL;	// MAIN TRC
	GROUP06 : BOOL;	// NU
	GROUP07, GROUP07_1, GROUP07_2, GROUP07_3, GROUP07_4, GROUP07_5, GROUP07_6 : BOOL;		// RECTIFIER
	GROUP08 : BOOL;		// FU
	GROUP09 : BOOL;		// TRO
	GROUP10, GROUP10_1, GROUP10_2 : BOOL;		// BALLAST SYSTEM
	GROUP11 : BOOL;		// SD
	GROUP12, GROUP12_1, GROUP12_2, GROUP12_3, GROUP12_4, GROUP12_5 : BOOL;		// SYSTEM 
	GROUP13, GROUP13_1, GROUP13_2, GROUP13_3, GROUP13_4, GROUP13_5, GROUP13_6, GROUP13_7, GROUP13_8, GROUP13_9, GROUP13_10, GROUP13_11, GROUP13_12, GROUP13_13, GROUP13_14 : BOOL;	// SEQUENCE FAIL	
END_VAR

/////////////////////////////////////////////////////////////////////////COMMON ALARM FOR HMI/////////////////////////////////////////////////////////////////////////////////////////////
//SR_0(SET1:= GROUP01 OR GROUP02 OR GROUP03 OR GROUP04 OR GROUP05 OR GROUP06 OR GROUP07 OR GROUP08 OR GROUP09 OR GROUP10 OR GROUP11 OR GROUP12 OR GROUP13 , RESET:= MP_RESET, Q1 => BWTS_004);
BWTS_004 := GROUP01 OR GROUP02 OR GROUP03 OR GROUP04 OR GROUP05 OR GROUP06 OR GROUP07 OR GROUP08 OR GROUP09 OR GROUP10 OR GROUP11 OR GROUP12 OR GROUP13;

/////////////////////////////////////////////////////////////////////////COMMON ALARM TO AMS (SECOND FAULT ALARM)/////////////////////////////////////////////////////////
TOF_0(IN := NOT (BWTS_004 AND NOT ALARM_BUZZER_2.BUZZER_ON), PT := T#2S, Q=> SECOND_FAULT);
BWTS_005 := SECOND_FAULT; 

/////////////////////////////////////////////////////////////////////////SHUTDOWN TO AMS/////////////////////////////////////////////////////////////////////////
BWTS_003 := (PSD_11 OR PSD_12 OR PSD_21 OR PSD_22 OR PSD_31 OR ESD);
BWTS_006 := NOT (PSD_11 OR PSD_12 OR PSD_21 OR PSD_22 OR PSD_31 OR ESD);

/////////////////////////////////////////////////////////////////////////GROUP01 (SENSOR FAULT)/////////////////////////////////////////////////////////////////////////


/////////////////////////////////////////////////////////////////////////GROUP02 (EU)/////////////////////////////////////////////////////////////////////////
GROUP02 := GROUP02_1 OR GROUP02_2;

GROUP02_1 :=
B117A_STF OR B117A_SPF OR B117B_STF OR B117B_SPF OR XV1171A_OPF OR XV1171A_CLF OR XV1171B_OPF OR XV1171B_CLF OR B_117A_F OR B_117B_F OR B_117A_OFF OR B_117B_OFF OR BLR_BYPASS OR BLR_BOTH_F OR
PT_1121_HI OR PT_1121_LO OR PT_1121_LL OR LS_1111_LL OR LS_1141_HI OR ER_FAN_OFF OR AIT_1121_HH OR AIT_1121_HI OR AIT_1122_HH OR AIT_1122_HI OR AIT_1123_HH;

GROUP02_2 :=
AIT_1123_HI OR TE_1111_HI OR TE_1111_LO OR TE_1111_LL OR CT_1111_LO OR CT_1111_LL OR ZS_1112A_CL OR ZS_1112A_OP OR ZS_1113A_CL OR ZS_1113A_OP OR ZS_1114A_CL OR ZS_1114A_OP;

/////////////////////////////////////////////////////////////////////////GROUP03 (SWFU)/////////////////////////////////////////////////////////////////////////
GROUP03 := 
P171A_STF OR P171A_SPF OR P171B_STF OR P171B_SPF OR SWFP_BOTH_F OR P_171A_F OR P_171B_F OR P_171A_OFF OR P_171B_OFF OR PT_1721_HI OR
PT_1721_LO OR PT_1721_LL OR PT_1722_HH OR PT_1722_HI OR PT_1722_LO OR SWFU_DP_HI OR  SWFU_DP_HH;

/////////////////////////////////////////////////////////////////////////GROUP04 (INJECTION)////////////////////////////////////////////////////////////////////
GROUP04 :=
FCV1131_CF OR  FIT_1131_LO OR  FIT_1131_LL OR RFS_1131 OR
FCV2131_CF OR  FIT_2131_LO OR  FIT_2131_LL OR RFS_2131
; 

/////////////////////////////////////////////////////////////////////////GROUP05 (MAIN TRC)////////////////////////////////////////////////////////////////////
GROUP05 :=
FCV1211_CF OR FIT_1211_HH OR FIT_1211_HI OR FIT_1211_LO OR 
FCV2211_CF OR FIT_2211_HH OR FIT_2211_HI OR FIT_2211_LO
;

/////////////////////////////////////////////////////////////////////////GROUP06 (NU)////////////////////////////////////////////////////////////////////
GROUP06 :=
P_132_TRIP OR P132_STF OR  P132_SPF OR DPS_1321 OR
P_232_TRIP OR P232_STF OR  P232_SPF OR DPS_2321 OR 
LIT_1311_HI OR  LIT_1311_LO OR  LIT_1311_LL;

/////////////////////////////////////////////////////////////////////////GROUP07 (RECTIFIER)////////////////////////////////////////////////////////////////////
GROUP07 :=
GROUP07_1 OR GROUP07_2 OR GROUP07_3 OR GROUP07_4 OR GROUP07_5 OR GROUP07_6;

GROUP07_1 :=
RF142A_STF OR RF142A_SPF OR RF142B_STF OR RF142B_SPF OR RF_142A_E OR RF_142B_E OR RF_ALL_SPD;

GROUP07_2 :=
REC1001 OR REC1002 OR REC1003 OR REC1004 OR REC1005 OR REC1006 OR REC1007 OR REC1008 OR REC1009 OR REC1010 OR REC1011 OR
REC1012 OR REC1013 OR REC1014 OR REC1015 OR REC1022 OR REC1023 OR REC1024 OR REC1025 OR REC1026 OR REC1032 OR REC1033;

GROUP07_3 :=
REC1017_HH OR REC1017_HI OR REC1018_HH OR REC1018_HI OR REC1019_HH OR REC1019_HI OR REC1020_HH OR REC1020_HI OR REC1021_HH OR REC1021_HI OR REC1027_HH OR REC1027_HI;

GROUP07_4 := 
REC2001 OR REC2002 OR REC2003 OR REC2004 OR REC2005 OR REC2006 OR REC2007 OR REC2008 OR REC2009 OR REC2010 OR REC2011 OR
REC2012 OR REC2013 OR REC2014 OR REC2015 OR REC2022 OR REC2023 OR REC2024 OR REC2025 OR REC2026 OR REC2032 OR REC2033;

GROUP07_5 :=
REC2017_HH OR REC2017_HI OR REC2018_HH OR REC2018_HI OR REC2019_HH OR REC2019_HI OR REC2020_HH OR REC2020_HI OR REC2021_HH OR REC2021_HI OR REC2027_HH OR REC2027_HI;

/////////////////////////////////////////////////////////////////////////GROUP09 (TRO)////////////////////////////////////////////////////////////////////
GROUP09 :=
BTRO_HH_S OR BTRO_HI_S OR BTRO_LO_S OR BTRO_LL_S OR DTRO_HH_S OR DTRO_HI_S OR
BTRO_HH_P OR BTRO_HI_P OR BTRO_LO_P OR BTRO_LL_P OR DTRO_HH_P OR DTRO_HI_P OR
STRO_HH OR STRO_HI OR
AIT_151_E OR AIT_151_F OR
AIT_251_E OR AIT_251_F OR
LS_1901_HH
;

/////////////////////////////////////////////////////////////////////////GROUP10 (BALLAST SYSTEM)/////////////////////////////////////////////////////////
GROUP10 := GROUP10_1 OR GROUP10_2; 

GROUP10_1 := 
WBP01_STF OR WBP01_SPF OR WBP_01_AL OR WBP_01_FAULT OR
WBP02_STF OR WBP02_SPF OR WBP_02_AL OR WBP_02_FAULT OR
GSP01_STF OR GSP01_SPF OR GSP_01_AL OR GSP_01_FAULT OR
GSP02_STF OR GSP02_SPF OR GSP_02_AL OR GSP_02_FAULT OR
SYS_BYPASS_1 OR SYS_BYPASS_2 OR SYS_BYPASS_3 OR SYS_BYPASS_4 OR
BAL_VV_AL_S OR BAL_VV_AL_P OR DEBAL_VV_AL_S OR DEBAL_VV_AL_P OR STR_VV_AL_S OR
AP_LVL_LO OR AP_LVL_LL OR GAS_LEAK_AL
;

/////////////////////////////////////////////////////////////////////////GROUP11 (SD)/////////////////////////////////////////////////////////////////////
GROUP11 := 
ESD OR PSD_11 OR PSD_12 OR PSD_21 OR PSD_22 OR PSD_31 OR PSD_41 OR PSD_42;

/////////////////////////////////////////////////////////////////////////GROUP12 (SYSTEM)/////////////////////////////////////////////////////////////////
GROUP12 :=
GROUP12_1 OR GROUP12_2 OR GROUP12_3 OR GROUP12_4;

GROUP12_1 := 
DISABLE1 OR DISABLE2 OR DISABLE3 OR DISABLE4 OR MM_AIT1121 OR MM_AIT1122 OR MM_AIT1123 OR MM_REPAIR;

GROUP12_4 :=
GPS_ALARM OR MCC_100_OFF OR PR_FAN_OFF OR CC100_TEMP_HI OR ESTOP_HMI OR ESTOP_CC OR ESTOP_RF OR
RH_EU_AL OR RH_AIT1121_AL OR RH_AIT1122_AL OR RH_AIT1123_AL OR RH_AIT151_AL OR RH_AIT251_AL OR
RH_P132_AL OR RH_P232_AL OR RH_P171A_AL OR RH_P171B_AL
;

GROUP13 := GROUP13_1 OR GROUP13_2 OR GROUP13_3 OR GROUP13_4 OR GROUP13_5 OR GROUP13_6 OR GROUP13_7 OR GROUP13_8 OR GROUP13_9 OR GROUP13_10 OR GROUP13_11 OR GROUP13_12 OR GROUP13_13 OR GROUP13_14; 

// SEQUENCE FAIL BALLASTING START STBD
GROUP13_1 := 
BST_S_01.TIMEOUT OR BST_S_03.TIMEOUT OR BST_S_04.TIMEOUT OR BST_S_05.TIMEOUT OR BST_S_06.TIMEOUT OR BST_S_07.TIMEOUT OR BST_S_08.TIMEOUT OR
BST_S_10.TIMEOUT OR BST_S_12.TIMEOUT OR BST_S_13.TIMEOUT OR BST_S_14.TIMEOUT OR BST_S_15.TIMEOUT OR BST_S_16.TIMEOUT OR BST_S_18.TIMEOUT;
 
// SEQUENCE FAIL BALLASTING STOP STBD
GROUP13_2 :=
BSP_S_01.TIMEOUT OR BSP_S_03.TIMEOUT OR BSP_S_04.TIMEOUT OR BSP_S_05.TIMEOUT OR BSP_S_07.TIMEOUT OR BSP_S_08.TIMEOUT OR BSP_S_09.TIMEOUT OR
BSP_S_10.TIMEOUT OR BSP_S_12.TIMEOUT;

// SEQUENCE FAIL BALLASTING START STBD
GROUP13_3 :=
BST_P_01.TIMEOUT OR BST_P_03.TIMEOUT OR BST_P_04.TIMEOUT OR BST_P_05.TIMEOUT OR BST_P_06.TIMEOUT OR BST_P_07.TIMEOUT OR BST_P_08.TIMEOUT OR 
BST_P_10.TIMEOUT OR BST_P_12.TIMEOUT OR BST_P_13.TIMEOUT OR BST_P_14.TIMEOUT OR BST_P_15.TIMEOUT OR BST_P_16.TIMEOUT OR BST_P_18.TIMEOUT;

// SEQUENCE FAIL BALLASTING STOP PORT
GROUP13_4 :=
BSP_P_01.TIMEOUT OR BSP_P_03.TIMEOUT OR BSP_P_04.TIMEOUT OR BSP_P_05.TIMEOUT OR BSP_P_07.TIMEOUT OR BSP_P_08.TIMEOUT OR BSP_P_09.TIMEOUT OR
BSP_P_10.TIMEOUT OR BSP_P_12.TIMEOUT;

// SEQUENCE FAIL DEBALLASTING START STBD
GROUP13_5 :=
DST_S_02.TIMEOUT OR DST_S_03.TIMEOUT OR DST_S_04.TIMEOUT OR DST_S_05.TIMEOUT OR DST_S_06.TIMEOUT OR DST_S_07.TIMEOUT OR DST_S_08.TIMEOUT OR DST_S_09.TIMEOUT;

// SEQUENCE FAIL DEBALLASTING STOP STBD
GROUP13_6 :=
DSP_S_01.TIMEOUT OR DSP_S_02.TIMEOUT OR DSP_S_03.TIMEOUT OR DSP_S_05.TIMEOUT OR DSP_S_06.TIMEOUT OR DSP_S_07.TIMEOUT;

// SEQUENCE FAIL DEBALLASTING START PORT
GROUP13_7 :=
DST_P_02.TIMEOUT OR DST_P_03.TIMEOUT OR DST_P_04.TIMEOUT OR DST_P_05.TIMEOUT OR DST_P_06.TIMEOUT OR DST_P_07.TIMEOUT OR DST_P_08.TIMEOUT OR DST_P_09.TIMEOUT;

// SEQUENCE FAIL DEBALLASTING STOP PORT
GROUP13_8 :=
DSP_P_01.TIMEOUT OR DSP_P_02.TIMEOUT OR DSP_P_03.TIMEOUT OR DSP_P_05.TIMEOUT OR DSP_P_06.TIMEOUT OR DSP_P_07.TIMEOUT;

// SEQUENCE FAIL STRIPPING START STBD
GROUP13_9 :=
SST_S_01.TIMEOUT OR SST_S_02.TIMEOUT OR SST_S_03.TIMEOUT OR SST_S_04.TIMEOUT OR SST_S_06.TIMEOUT OR SST_S_07.TIMEOUT OR SST_S_08.TIMEOUT OR SST_S_09.TIMEOUT;

// SEQUENCE FAIL STRIPPING STOP STBD
GROUP13_10 :=
SSP_S_01.TIMEOUT OR SSP_S_02.TIMEOUT OR SSP_S_03.TIMEOUT OR SSP_S_04.TIMEOUT OR SSP_S_06.TIMEOUT OR SSP_S_07.TIMEOUT;

END_PROGRAM

// Device/Application/Logic/0.SIMULATION/AMS
PROGRAM AMS
VAR
	RS_BA30 : RS;
	RS_BA31 : RS;
	RS_BA32 : RS;
	RS_BA33 : RS;
	RS_BA34 : RS;
	RS_BA35 : RS;
	RS_BA36 : RS;
	RS_BA37 : RS;
	RS_BA38 : RS;
	RS_BA39 : RS;
END_VAR

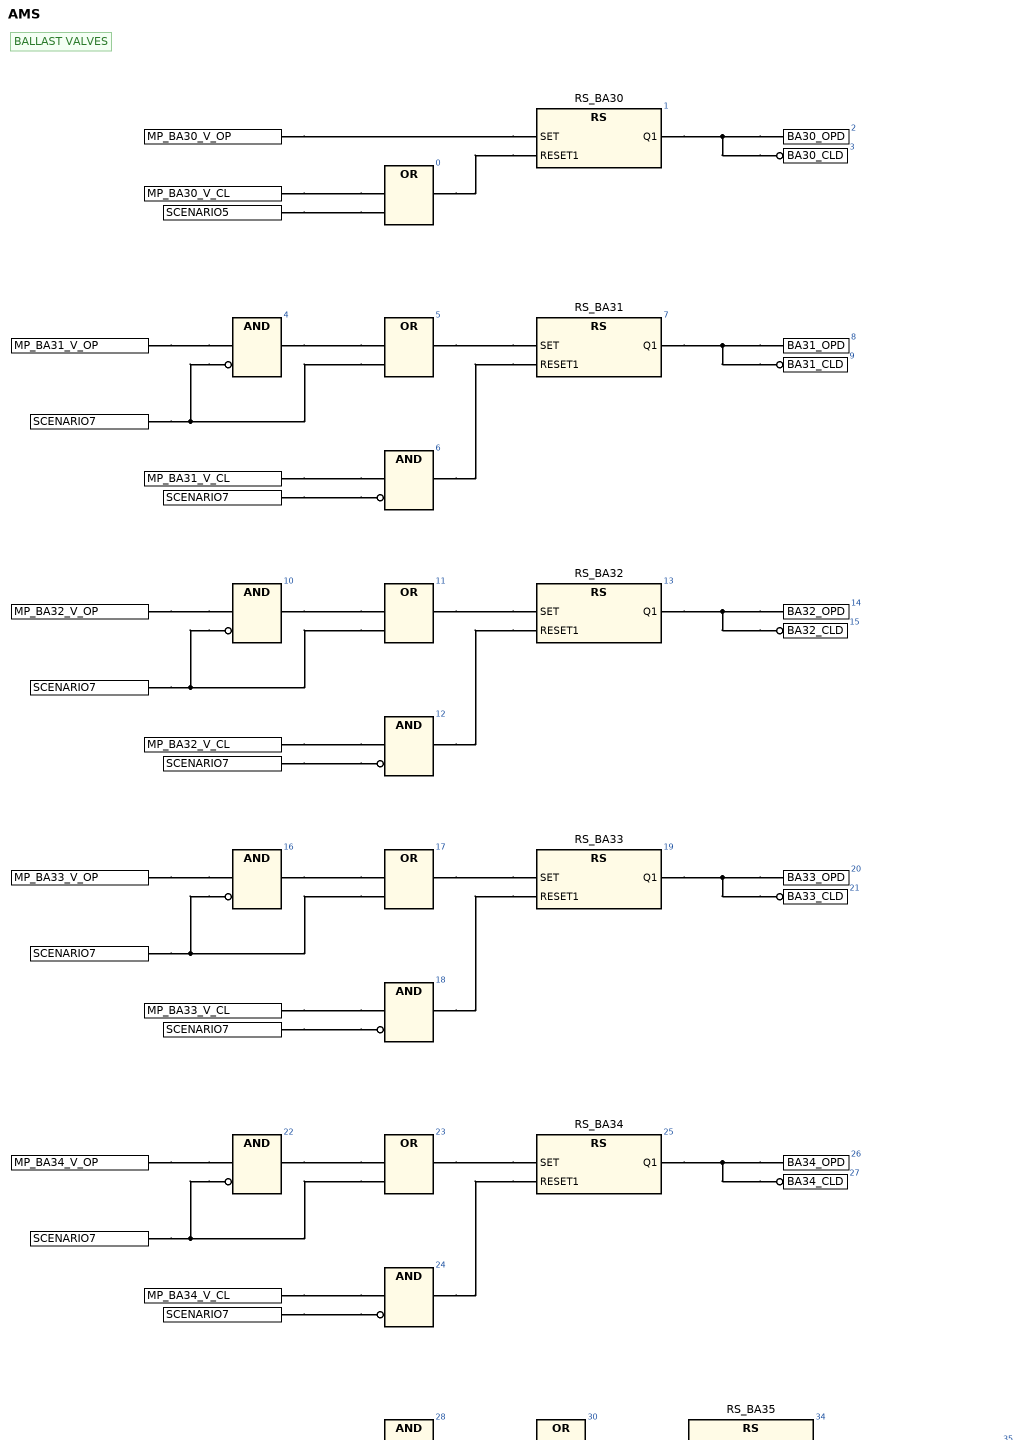
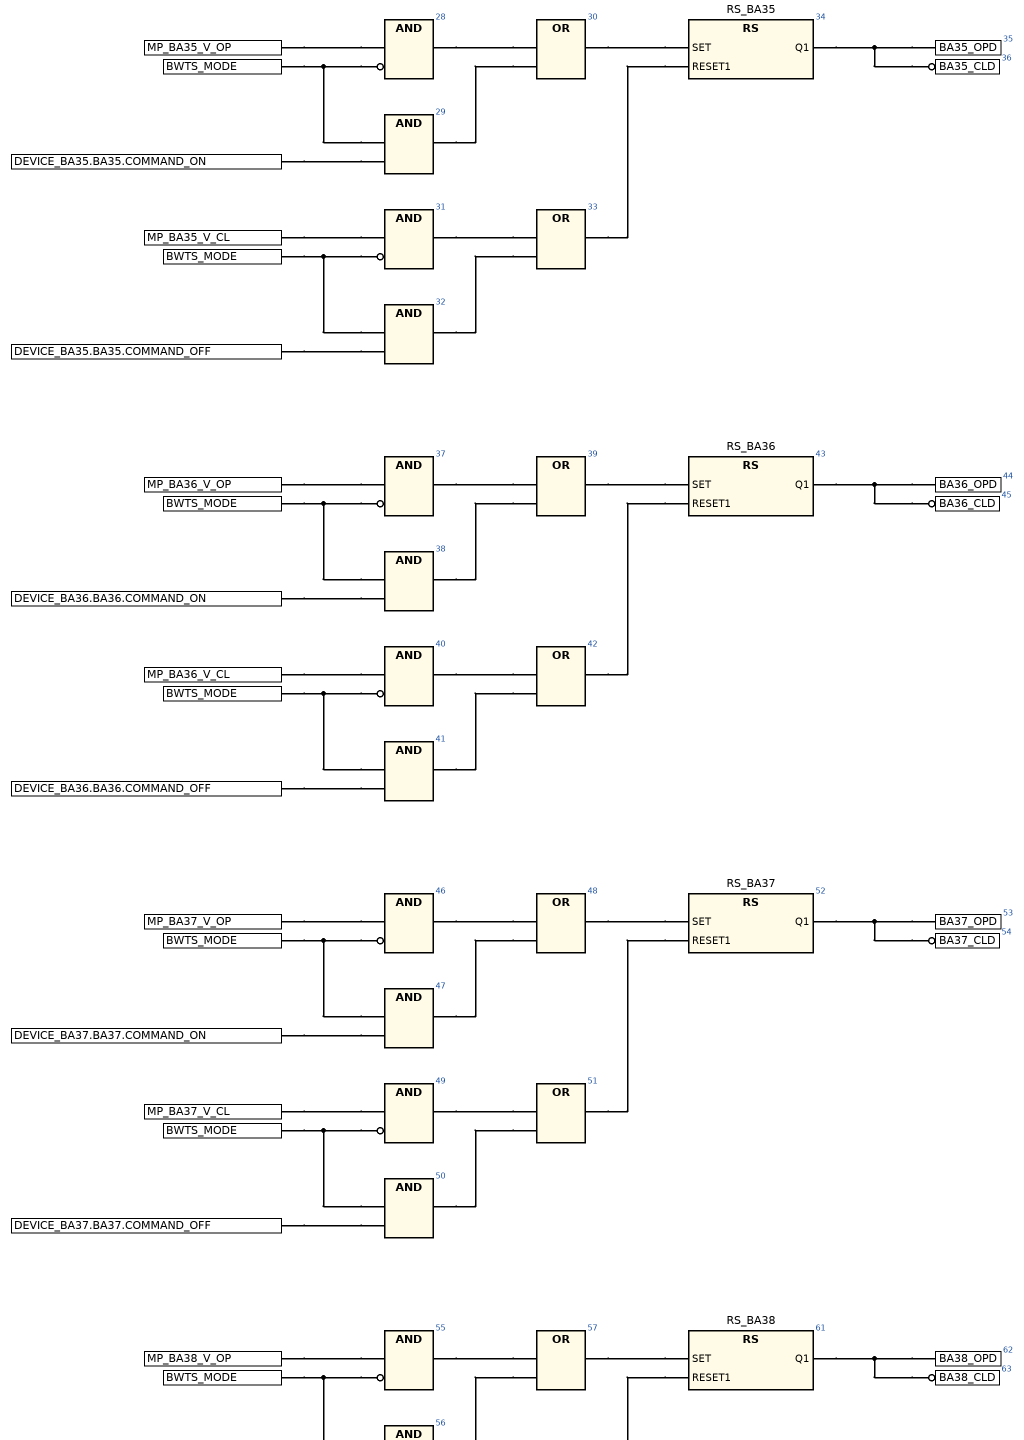
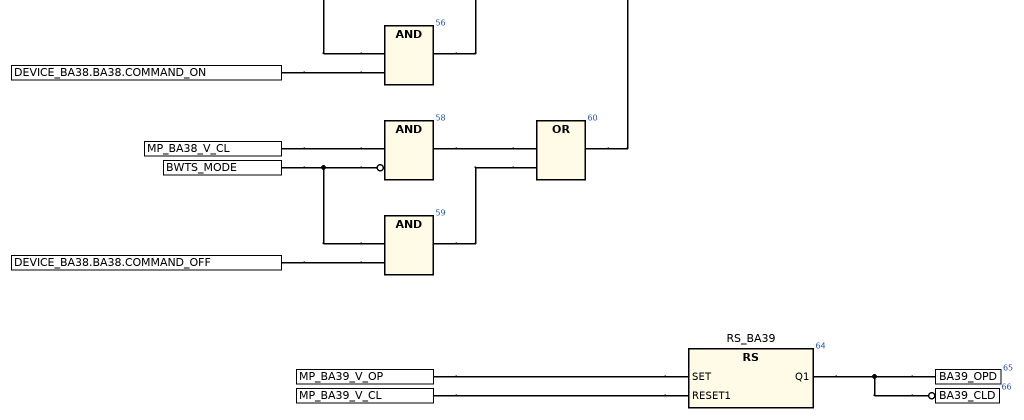
// BALLAST VALVES
RS_BA30(SET := MP_BA30_V_OP, RESET1 := MP_BA30_V_CL OR SCENARIO5); // RS
BA30_OPD := RS_BA30.Q1;
BA30_CLD := NOT RS_BA30.Q1;
RS_BA31(SET := MP_BA31_V_OP AND NOT SCENARIO7 OR SCENARIO7, RESET1 := MP_BA31_V_CL AND NOT SCENARIO7); // RS
BA31_OPD := RS_BA31.Q1;
BA31_CLD := NOT RS_BA31.Q1;
RS_BA32(SET := MP_BA32_V_OP AND NOT SCENARIO7 OR SCENARIO7, RESET1 := MP_BA32_V_CL AND NOT SCENARIO7); // RS
BA32_OPD := RS_BA32.Q1;
BA32_CLD := NOT RS_BA32.Q1;
RS_BA33(SET := MP_BA33_V_OP AND NOT SCENARIO7 OR SCENARIO7, RESET1 := MP_BA33_V_CL AND NOT SCENARIO7); // RS
BA33_OPD := RS_BA33.Q1;
BA33_CLD := NOT RS_BA33.Q1;
RS_BA34(SET := MP_BA34_V_OP AND NOT SCENARIO7 OR SCENARIO7, RESET1 := MP_BA34_V_CL AND NOT SCENARIO7); // RS
BA34_OPD := RS_BA34.Q1;
BA34_CLD := NOT RS_BA34.Q1;
RS_BA35(SET := MP_BA35_V_OP AND NOT BWTS_MODE OR BWTS_MODE AND DEVICE_BA35.BA35.COMMAND_ON, RESET1 := MP_BA35_V_CL AND NOT BWTS_MODE OR BWTS_MODE AND DEVICE_BA35.BA35.COMMAND_OFF); // RS
BA35_OPD := RS_BA35.Q1;
BA35_CLD := NOT RS_BA35.Q1;
RS_BA36(SET := MP_BA36_V_OP AND NOT BWTS_MODE OR BWTS_MODE AND DEVICE_BA36.BA36.COMMAND_ON, RESET1 := MP_BA36_V_CL AND NOT BWTS_MODE OR BWTS_MODE AND DEVICE_BA36.BA36.COMMAND_OFF); // RS
BA36_OPD := RS_BA36.Q1;
BA36_CLD := NOT RS_BA36.Q1;
RS_BA37(SET := MP_BA37_V_OP AND NOT BWTS_MODE OR BWTS_MODE AND DEVICE_BA37.BA37.COMMAND_ON, RESET1 := MP_BA37_V_CL AND NOT BWTS_MODE OR BWTS_MODE AND DEVICE_BA37.BA37.COMMAND_OFF); // RS
BA37_OPD := RS_BA37.Q1;
BA37_CLD := NOT RS_BA37.Q1;
RS_BA38(SET := MP_BA38_V_OP AND NOT BWTS_MODE OR BWTS_MODE AND DEVICE_BA38.BA38.COMMAND_ON, RESET1 := MP_BA38_V_CL AND NOT BWTS_MODE OR BWTS_MODE AND DEVICE_BA38.BA38.COMMAND_OFF); // RS
BA38_OPD := RS_BA38.Q1;
BA38_CLD := NOT RS_BA38.Q1;
RS_BA39(SET := MP_BA39_V_OP, RESET1 := MP_BA39_V_CL); // RS
BA39_OPD := RS_BA39.Q1;
BA39_CLD := NOT RS_BA39.Q1;

END_PROGRAM

// Device/Application/Logic/4.Device/DEVICE_BA35
PROGRAM DEVICE_BA35
VAR
	BA35: BWTS.YARD_ONOFF;
END_VAR
VAR // added by the converter: edge detectors and wires of the graphical bodies
    _w1, _w2, _w3, _w4 : ANY;
END_VAR

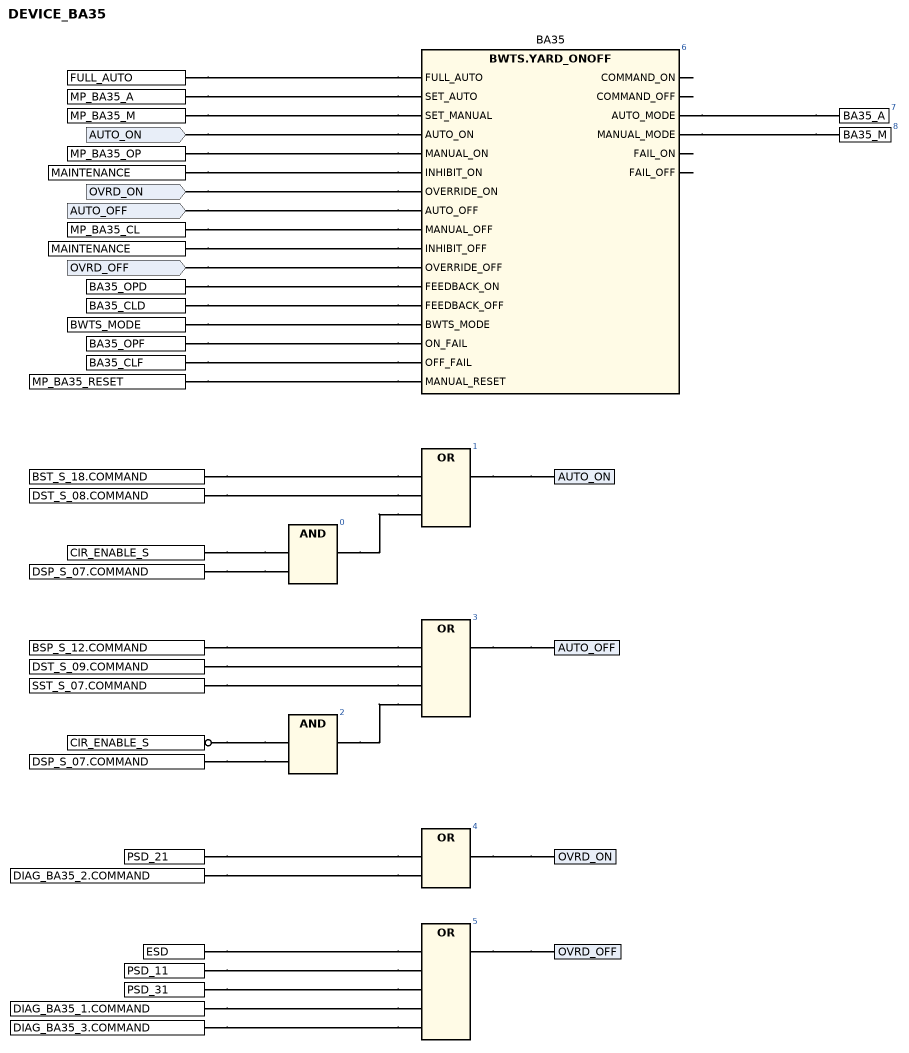
(* BST_S_18.COMMAND OR DST_S_08.COMMAND OR CIR_ENABLE_S AND DSP_S_07.COMMAND; result not used *)
(* BSP_S_12.COMMAND OR DST_S_09.COMMAND OR SST_S_07.COMMAND OR NOT CIR_ENABLE_S AND DSP_S_07.COMMAND; result not used *)
(* PSD_21 OR DIAG_BA35_2.COMMAND; result not used *)
(* ESD OR PSD_11 OR PSD_31 OR DIAG_BA35_1.COMMAND OR DIAG_BA35_3.COMMAND; result not used *)
BA35(
    FULL_AUTO := FULL_AUTO,
    SET_AUTO := MP_BA35_A,
    SET_MANUAL := MP_BA35_M,
    AUTO_ON := _w1,
    MANUAL_ON := MP_BA35_OP,
    INHIBIT_ON := MAINTENANCE,
    OVERRIDE_ON := _w2,
    AUTO_OFF := _w3,
    MANUAL_OFF := MP_BA35_CL,
    INHIBIT_OFF := MAINTENANCE,
    OVERRIDE_OFF := _w4,
    FEEDBACK_ON := BA35_OPD,
    FEEDBACK_OFF := BA35_CLD,
    BWTS_MODE := BWTS_MODE,
    ON_FAIL := BA35_OPF,
    OFF_FAIL := BA35_CLF,
    MANUAL_RESET := MP_BA35_RESET); // BWTS.YARD_ONOFF
BA35_A := BA35.AUTO_MODE;
BA35_M := BA35.MANUAL_MODE;

END_PROGRAM

// Device/Application/Logic/0.ETC/AUTO_MODE
PROGRAM AUTO_MODE
VAR
	TP_0: TP;
	TP_1: TP;
	TP_2: TP;
	TP_3: TP;
	TP_4: TP;
	TP_5: TP;
	TP_6: TP;
	TP_7: TP;
	TP_8: TP;
	TP_9: TP;	
	
	TP_14: TP;	
END_VAR
VAR // added by the converter: edge detectors and wires of the graphical bodies
    _w1, _w2, _w3, _w4, _w5, _w6, _w7, _w8, _w9, _w10, _w11 : BOOL;
END_VAR

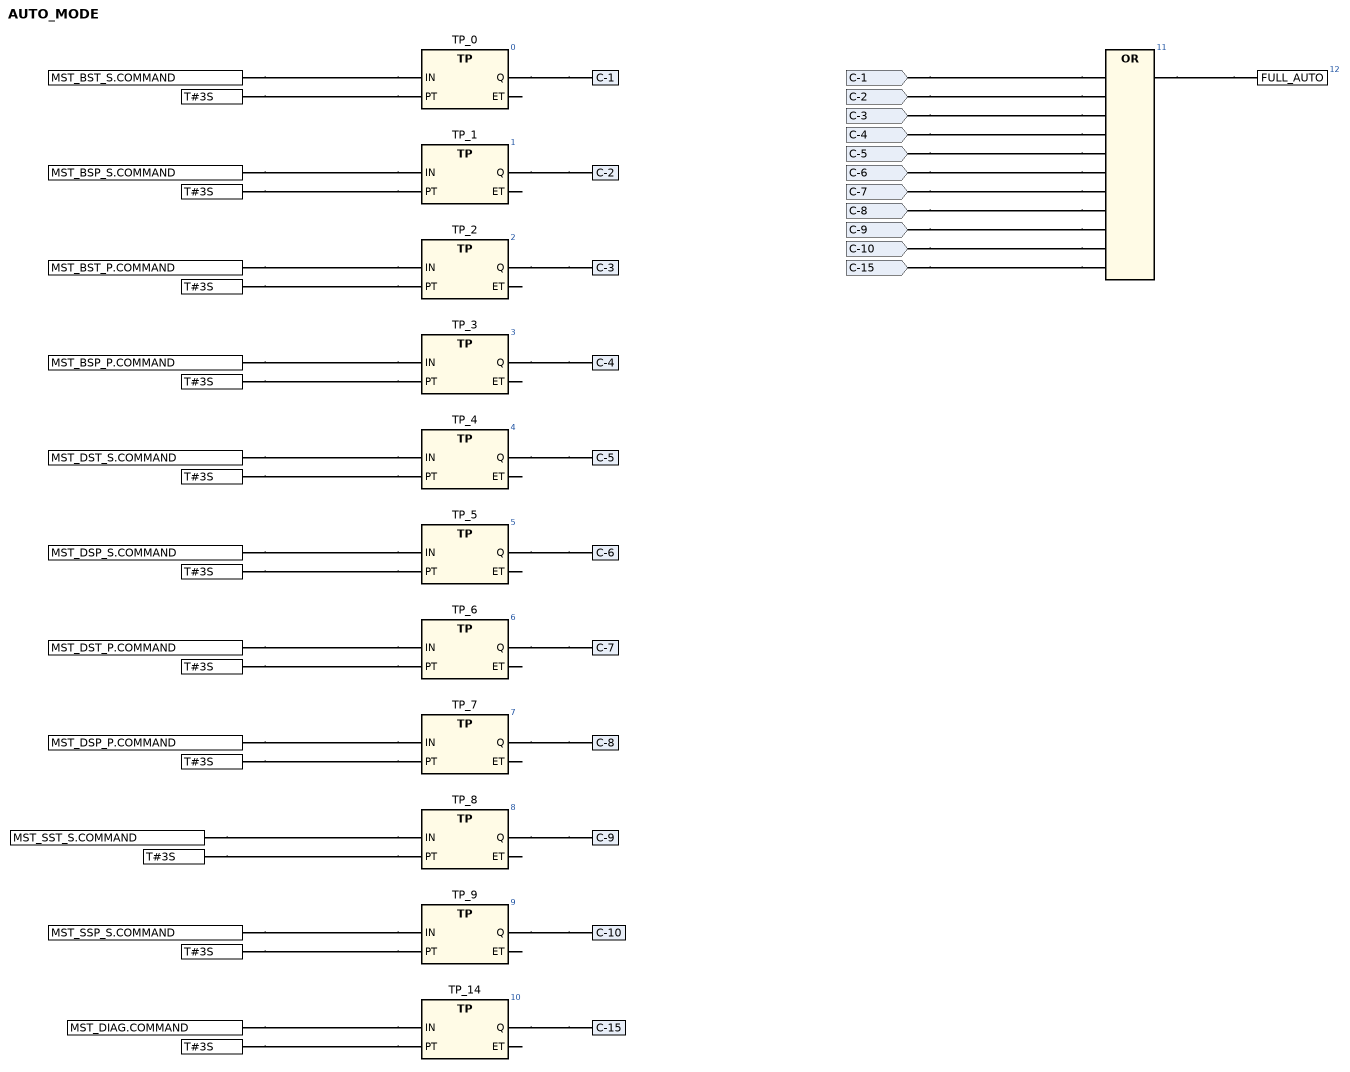
TP_0(IN := MST_BST_S.COMMAND, PT := T#3S); // TP
TP_1(IN := MST_BSP_S.COMMAND, PT := T#3S); // TP
TP_2(IN := MST_BST_P.COMMAND, PT := T#3S); // TP
TP_3(IN := MST_BSP_P.COMMAND, PT := T#3S); // TP
TP_4(IN := MST_DST_S.COMMAND, PT := T#3S); // TP
TP_5(IN := MST_DSP_S.COMMAND, PT := T#3S); // TP
TP_6(IN := MST_DST_P.COMMAND, PT := T#3S); // TP
TP_7(IN := MST_DSP_P.COMMAND, PT := T#3S); // TP
TP_8(IN := MST_SST_S.COMMAND, PT := T#3S); // TP
TP_9(IN := MST_SSP_S.COMMAND, PT := T#3S); // TP
TP_14(IN := MST_DIAG.COMMAND, PT := T#3S); // TP
FULL_AUTO := _w1 OR _w2 OR _w3 OR _w4 OR _w5 OR _w6 OR _w7 OR _w8 OR _w9 OR _w10 OR _w11;

END_PROGRAM

// Device/Application/Logic/4.Device/DEVICE_BA36
PROGRAM DEVICE_BA36
VAR
	BA36: BWTS.YARD_ONOFF;
END_VAR
VAR // added by the converter: edge detectors and wires of the graphical bodies
    _w1, _w2, _w3, _w4 : ANY;
END_VAR

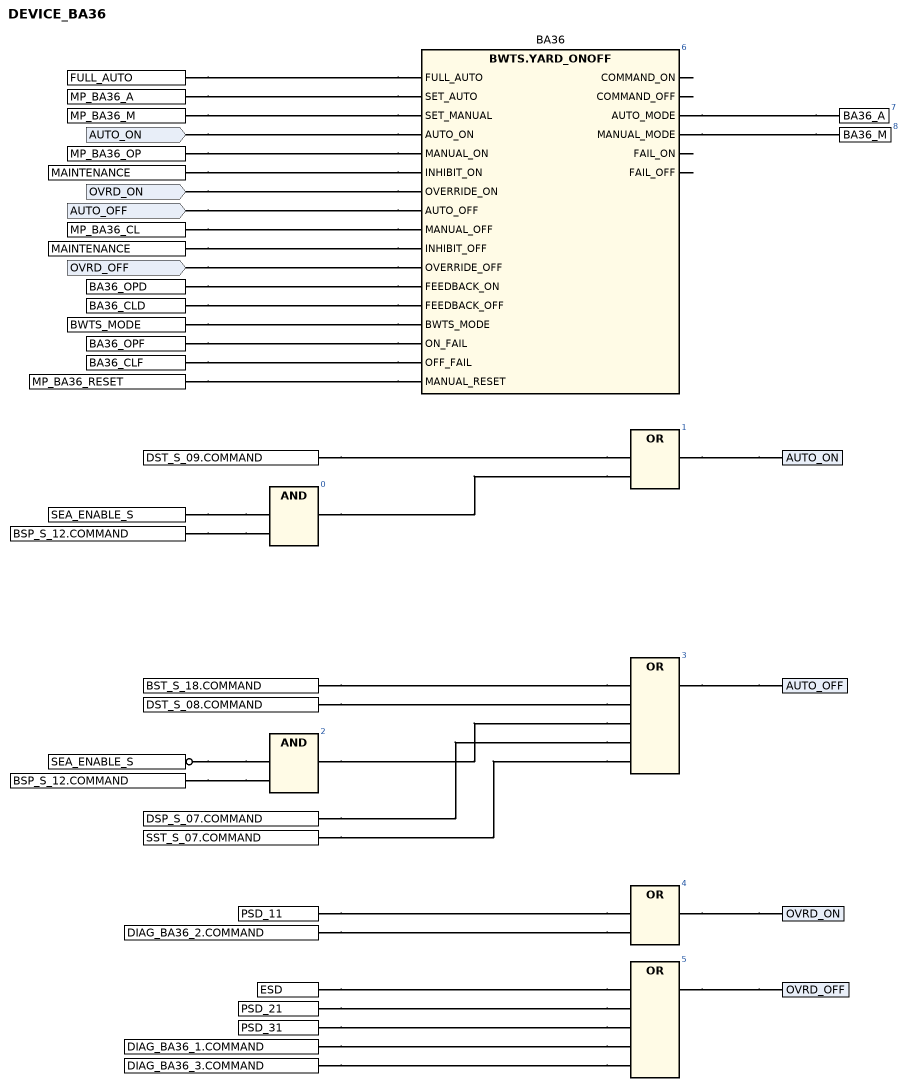
(* DST_S_09.COMMAND OR SEA_ENABLE_S AND BSP_S_12.COMMAND; result not used *)
(* BST_S_18.COMMAND OR DST_S_08.COMMAND OR NOT SEA_ENABLE_S AND BSP_S_12.COMMAND OR DSP_S_07.COMMAND OR SST_S_07.COMMAND; result not used *)
(* PSD_11 OR DIAG_BA36_2.COMMAND; result not used *)
(* ESD OR PSD_21 OR PSD_31 OR DIAG_BA36_1.COMMAND OR DIAG_BA36_3.COMMAND; result not used *)
BA36(
    FULL_AUTO := FULL_AUTO,
    SET_AUTO := MP_BA36_A,
    SET_MANUAL := MP_BA36_M,
    AUTO_ON := _w1,
    MANUAL_ON := MP_BA36_OP,
    INHIBIT_ON := MAINTENANCE,
    OVERRIDE_ON := _w2,
    AUTO_OFF := _w3,
    MANUAL_OFF := MP_BA36_CL,
    INHIBIT_OFF := MAINTENANCE,
    OVERRIDE_OFF := _w4,
    FEEDBACK_ON := BA36_OPD,
    FEEDBACK_OFF := BA36_CLD,
    BWTS_MODE := BWTS_MODE,
    ON_FAIL := BA36_OPF,
    OFF_FAIL := BA36_CLF,
    MANUAL_RESET := MP_BA36_RESET); // BWTS.YARD_ONOFF
BA36_A := BA36.AUTO_MODE;
BA36_M := BA36.MANUAL_MODE;

END_PROGRAM

// Device/Application/Logic/4.Device/DEVICE_BA37
PROGRAM DEVICE_BA37
VAR
	BA37: BWTS.YARD_ONOFF;
END_VAR
VAR // added by the converter: edge detectors and wires of the graphical bodies
    _w1, _w2, _w3, _w4 : ANY;
END_VAR

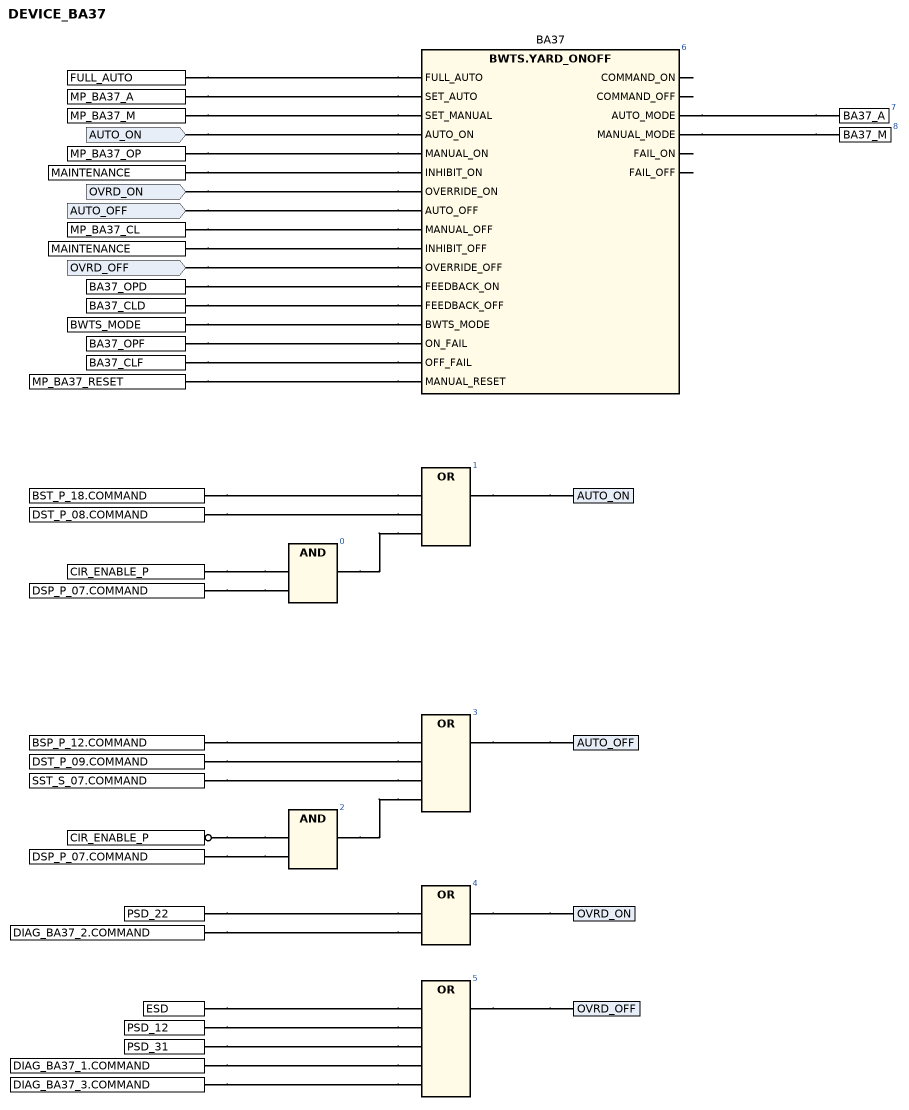
(* BST_P_18.COMMAND OR DST_P_08.COMMAND OR CIR_ENABLE_P AND DSP_P_07.COMMAND; result not used *)
(* BSP_P_12.COMMAND OR DST_P_09.COMMAND OR SST_S_07.COMMAND OR NOT CIR_ENABLE_P AND DSP_P_07.COMMAND; result not used *)
(* PSD_22 OR DIAG_BA37_2.COMMAND; result not used *)
(* ESD OR PSD_12 OR PSD_31 OR DIAG_BA37_1.COMMAND OR DIAG_BA37_3.COMMAND; result not used *)
BA37(
    FULL_AUTO := FULL_AUTO,
    SET_AUTO := MP_BA37_A,
    SET_MANUAL := MP_BA37_M,
    AUTO_ON := _w1,
    MANUAL_ON := MP_BA37_OP,
    INHIBIT_ON := MAINTENANCE,
    OVERRIDE_ON := _w2,
    AUTO_OFF := _w3,
    MANUAL_OFF := MP_BA37_CL,
    INHIBIT_OFF := MAINTENANCE,
    OVERRIDE_OFF := _w4,
    FEEDBACK_ON := BA37_OPD,
    FEEDBACK_OFF := BA37_CLD,
    BWTS_MODE := BWTS_MODE,
    ON_FAIL := BA37_OPF,
    OFF_FAIL := BA37_CLF,
    MANUAL_RESET := MP_BA37_RESET); // BWTS.YARD_ONOFF
BA37_A := BA37.AUTO_MODE;
BA37_M := BA37.MANUAL_MODE;

END_PROGRAM

// Device/Application/Logic/4.Device/DEVICE_BA38
PROGRAM DEVICE_BA38
VAR
	BA38: BWTS.YARD_ONOFF;
END_VAR
VAR // added by the converter: edge detectors and wires of the graphical bodies
    _w1, _w2, _w3, _w4 : ANY;
END_VAR

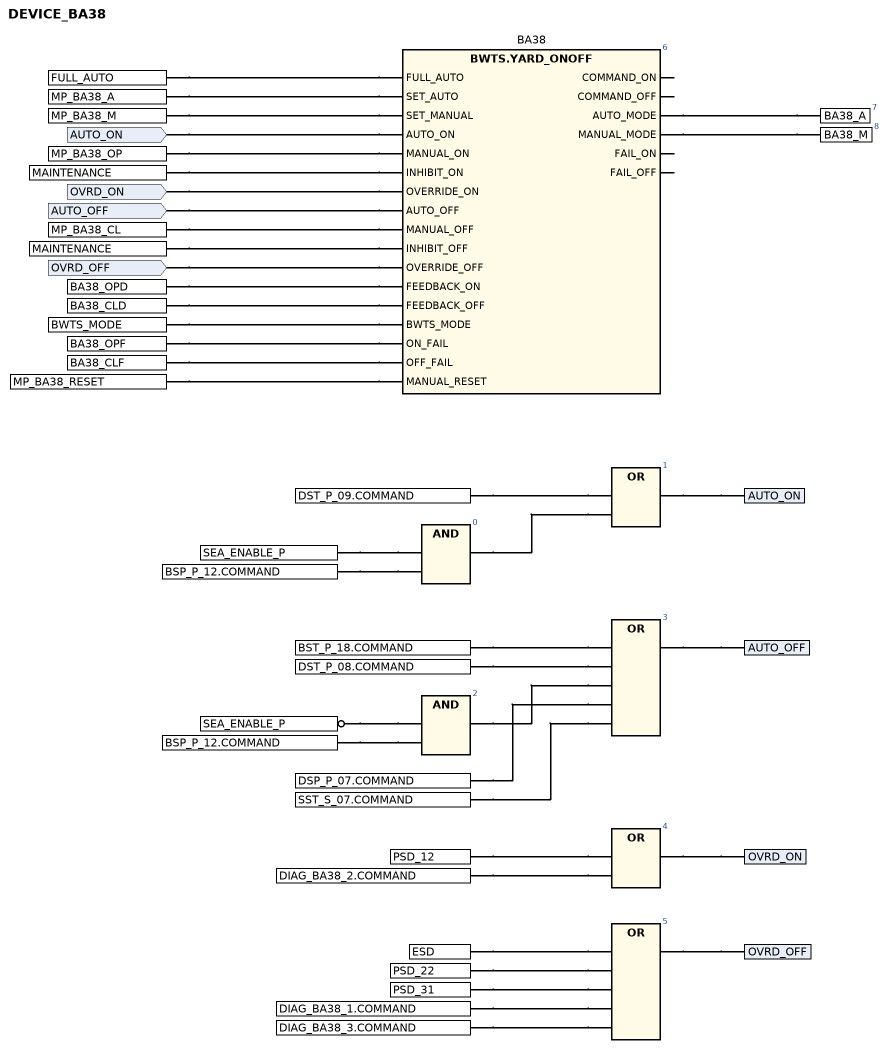
(* DST_P_09.COMMAND OR SEA_ENABLE_P AND BSP_P_12.COMMAND; result not used *)
(* BST_P_18.COMMAND OR DST_P_08.COMMAND OR NOT SEA_ENABLE_P AND BSP_P_12.COMMAND OR DSP_P_07.COMMAND OR SST_S_07.COMMAND; result not used *)
(* PSD_12 OR DIAG_BA38_2.COMMAND; result not used *)
(* ESD OR PSD_22 OR PSD_31 OR DIAG_BA38_1.COMMAND OR DIAG_BA38_3.COMMAND; result not used *)
BA38(
    FULL_AUTO := FULL_AUTO,
    SET_AUTO := MP_BA38_A,
    SET_MANUAL := MP_BA38_M,
    AUTO_ON := _w1,
    MANUAL_ON := MP_BA38_OP,
    INHIBIT_ON := MAINTENANCE,
    OVERRIDE_ON := _w2,
    AUTO_OFF := _w3,
    MANUAL_OFF := MP_BA38_CL,
    INHIBIT_OFF := MAINTENANCE,
    OVERRIDE_OFF := _w4,
    FEEDBACK_ON := BA38_OPD,
    FEEDBACK_OFF := BA38_CLD,
    BWTS_MODE := BWTS_MODE,
    ON_FAIL := BA38_OPF,
    OFF_FAIL := BA38_CLF,
    MANUAL_RESET := MP_BA38_RESET); // BWTS.YARD_ONOFF
BA38_A := BA38.AUTO_MODE;
BA38_M := BA38.MANUAL_MODE;

END_PROGRAM

// Device/Application/Logic/0.ALARM/ALARM_DEVICE
PROGRAM ALARM_DEVICE
VAR
	ALARM_D_B117A_STF: BWTS.ALARM_D;
	ALARM_D_B117A_SPF: BWTS.ALARM_D;
	ALARM_D_B117B_STF: BWTS.ALARM_D;
	ALARM_D_B117B_SPF: BWTS.ALARM_D;
	ALARM_D_P171A_STF: BWTS.ALARM_D;
	ALARM_D_P171A_SPF: BWTS.ALARM_D;
	ALARM_D_P171B_STF: BWTS.ALARM_D;
	ALARM_D_P171B_SPF: BWTS.ALARM_D;
	ALARM_D_RF142A_STF: BWTS.ALARM_D;
	ALARM_D_RF142A_SPF: BWTS.ALARM_D;
	ALARM_D_RF142B_STF: BWTS.ALARM_D;
	ALARM_D_RF142B_SPF: BWTS.ALARM_D;
	ALARM_D_RF142C_STF: BWTS.ALARM_D;
	ALARM_D_RF142C_SPF: BWTS.ALARM_D;
	ALARM_D_P132_STF: BWTS.ALARM_D;
	ALARM_D_P132_SPF: BWTS.ALARM_D;
	ALARM_D_P232_STF: BWTS.ALARM_D;
	ALARM_D_P232_SPF: BWTS.ALARM_D;
	ALARM_D_XV1171A_OPF: BWTS.ALARM_D;
	ALARM_D_XV1171A_CLF: BWTS.ALARM_D;
	ALARM_D_XV1171B_OPF: BWTS.ALARM_D;
	ALARM_D_XV1171B_CLF: BWTS.ALARM_D;
	ALARM_D_FCV1131_CF: BWTS.ALARM_D;
	ALARM_D_FCV2131_CF: BWTS.ALARM_D;
	ALARM_D_FCV1211_CF: BWTS.ALARM_D;
	ALARM_D_FCV2211_CF: BWTS.ALARM_D;
	ALARM_D_WBP01_STF: BWTS.ALARM_D;
	ALARM_D_WBP01_SPF: BWTS.ALARM_D;
	ALARM_D_WBP02_STF: BWTS.ALARM_D;
	ALARM_D_WBP02_SPF: BWTS.ALARM_D;
	ALARM_D_GSP01_STF: BWTS.ALARM_D;
	ALARM_D_GSP01_SPF: BWTS.ALARM_D;
	ALARM_D_GSP02_STF: BWTS.ALARM_D;
	ALARM_D_GSP02_SPF: BWTS.ALARM_D;
	
	ALARM_D_BA35_OPF: BWTS.ALARM_D;
	ALARM_D_BA35_CLF: BWTS.ALARM_D;
	ALARM_D_BA36_OPF: BWTS.ALARM_D;
	ALARM_D_BA36_CLF: BWTS.ALARM_D;
	ALARM_D_BA37_OPF: BWTS.ALARM_D;
	ALARM_D_BA37_CLF: BWTS.ALARM_D;
	ALARM_D_BA38_OPF: BWTS.ALARM_D;
	ALARM_D_BA38_CLF: BWTS.ALARM_D;	

END_VAR

ALARM_D_B117A_STF(bTRIGGER := DEVICE_B117A.B117A.FAIL_ON, tDELAY:= T#10S, ALARM=>B117A_STF);
ALARM_D_B117A_SPF(bTRIGGER := DEVICE_B117A.B117A.FAIL_OFF, tDELAY:= T#10S, ALARM=>B117A_SPF);
ALARM_D_B117B_STF(bTRIGGER := DEVICE_B117B.B117B.FAIL_ON, tDELAY:= T#10S, ALARM=>B117B_STF);
ALARM_D_B117B_SPF(bTRIGGER := DEVICE_B117B.B117B.FAIL_OFF, tDELAY:= T#10S, ALARM=>B117B_SPF);
ALARM_D_P171A_STF(bTRIGGER := DEVICE_P171A.P171A.FAIL_ON, tDELAY:= T#10S, ALARM=>P171A_STF);
ALARM_D_P171A_SPF(bTRIGGER := DEVICE_P171A.P171A.FAIL_OFF, tDELAY:= T#10S, ALARM=>P171A_SPF);
ALARM_D_P171B_STF(bTRIGGER := DEVICE_P171B.P171B.FAIL_ON, tDELAY:= T#10S, ALARM=>P171B_STF);
ALARM_D_P171B_SPF(bTRIGGER := DEVICE_P171B.P171B.FAIL_OFF, tDELAY:= T#10S, ALARM=>P171B_SPF);
ALARM_D_RF142A_STF(bTRIGGER := DEVICE_RFA.RF142A.FAIL_ON, tDELAY:= T#15S, ALARM=>RF142A_STF);
ALARM_D_RF142A_SPF(bTRIGGER := DEVICE_RFA.RF142A.FAIL_OFF, tDELAY:= T#15S, ALARM=>RF142A_SPF);
ALARM_D_RF142B_STF(bTRIGGER := DEVICE_RFB.RF142B.FAIL_ON, tDELAY:= T#15S, ALARM=>RF142B_STF);
ALARM_D_RF142B_SPF(bTRIGGER := DEVICE_RFB.RF142B.FAIL_OFF, tDELAY:= T#15S, ALARM=>RF142B_SPF);
ALARM_D_RF142C_STF(bTRIGGER := DEVICE_RFC.RF142C.FAIL_ON, tDELAY:= T#15S, ALARM=>RF142C_STF);
ALARM_D_RF142C_SPF(bTRIGGER := DEVICE_RFC.RF142C.FAIL_OFF, tDELAY:= T#15S, ALARM=>RF142C_SPF);
ALARM_D_P132_STF(bTRIGGER := DEVICE_P132.P132.FAIL_ON, tDELAY:= T#10S, ALARM=>P132_STF);
ALARM_D_P132_SPF(bTRIGGER := DEVICE_P132.P132.FAIL_OFF, tDELAY:= T#10S, ALARM=>P132_SPF);
ALARM_D_P232_STF(bTRIGGER := DEVICE_P232.P232.FAIL_ON, tDELAY:= T#10S, ALARM=>P232_STF);
ALARM_D_P232_SPF(bTRIGGER := DEVICE_P232.P232.FAIL_OFF, tDELAY:= T#10S, ALARM=>P232_SPF);
ALARM_D_XV1171A_OPF(bTRIGGER := DEVICE_XV1171A.XV1171A.FAIL_ON, tDELAY:= T#10S, ALARM=>XV1171A_OPF);
ALARM_D_XV1171A_CLF(bTRIGGER := DEVICE_XV1171A.XV1171A.FAIL_OFF, tDELAY:= T#10S, ALARM=>XV1171A_CLF);
ALARM_D_XV1171B_OPF(bTRIGGER := DEVICE_XV1171B.XV1171B.FAIL_ON, tDELAY:= T#10S, ALARM=>XV1171B_OPF);
ALARM_D_XV1171B_CLF(bTRIGGER := DEVICE_XV1171B.XV1171B.FAIL_OFF, tDELAY:= T#10S, ALARM=>XV1171B_CLF);
ALARM_D_FCV1131_CF(bTRIGGER := DEVICE_FCV1131.FCV1131.CONTROL_FAIL, tDELAY:= T#30S, ALARM=>FCV1131_CF);
ALARM_D_FCV2131_CF(bTRIGGER := DEVICE_FCV2131.FCV2131.CONTROL_FAIL, tDELAY:= T#30S, ALARM=>FCV2131_CF);
ALARM_D_FCV1211_CF(bTRIGGER := DEVICE_FCV1211.FCV1211.CONTROL_FAIL, tDELAY:= T#120S, ALARM=>FCV1211_CF);
ALARM_D_FCV2211_CF(bTRIGGER := DEVICE_FCV2211.FCV2211.CONTROL_FAIL, tDELAY:= T#120S, ALARM=>FCV2211_CF);
ALARM_D_WBP01_STF(bTRIGGER := WBP01_ST_REQ, tDELAY:= T#60S, ALARM=>WBP01_STF);
ALARM_D_WBP01_SPF(bTRIGGER := WBP01_SP_REQ, tDELAY:= T#60S, ALARM=>WBP01_SPF);
ALARM_D_WBP02_STF(bTRIGGER := WBP02_ST_REQ, tDELAY:= T#60S, ALARM=>WBP02_STF);
ALARM_D_WBP02_SPF(bTRIGGER := WBP02_SP_REQ, tDELAY:= T#60S, ALARM=>WBP02_SPF);
ALARM_D_GSP01_STF(bTRIGGER := GSP01_ST_REQ, tDELAY:= T#60S, ALARM=>GSP01_STF);
ALARM_D_GSP01_SPF(bTRIGGER := GSP01_SP_REQ, tDELAY:= T#60S, ALARM=>GSP01_SPF);
ALARM_D_GSP02_STF(bTRIGGER := GSP02_ST_REQ, tDELAY:= T#60S, ALARM=>GSP02_STF);
ALARM_D_GSP02_SPF(bTRIGGER := GSP02_SP_REQ, tDELAY:= T#60S, ALARM=>GSP02_SPF);

ALARM_D_BA35_OPF(bTRIGGER := DEVICE_BA35.BA35.FAIL_ON, tDELAY:= T#120S, ALARM=>BA35_OPF);
ALARM_D_BA35_CLF(bTRIGGER := DEVICE_BA35.BA35.FAIL_OFF, tDELAY:= T#120S, ALARM=>BA35_CLF);
ALARM_D_BA36_OPF(bTRIGGER := DEVICE_BA36.BA36.FAIL_ON, tDELAY:= T#120S, ALARM=>BA36_OPF);
ALARM_D_BA36_CLF(bTRIGGER := DEVICE_BA36.BA36.FAIL_OFF, tDELAY:= T#120S, ALARM=>BA36_CLF);
ALARM_D_BA37_OPF(bTRIGGER := DEVICE_BA37.BA37.FAIL_ON, tDELAY:= T#120S, ALARM=>BA37_OPF);
ALARM_D_BA37_CLF(bTRIGGER := DEVICE_BA37.BA37.FAIL_OFF, tDELAY:= T#120S, ALARM=>BA37_CLF);
ALARM_D_BA38_OPF(bTRIGGER := DEVICE_BA38.BA38.FAIL_ON, tDELAY:= T#120S, ALARM=>BA38_OPF);
ALARM_D_BA38_CLF(bTRIGGER := DEVICE_BA38.BA38.FAIL_OFF, tDELAY:= T#120S, ALARM=>BA38_CLF);

END_PROGRAM

// Device/Application/Logic/4.Device/DEVICE_B117A
PROGRAM DEVICE_B117A
VAR
	B117A : BWTS.DEVICE;	
END_VAR
VAR // added by the converter: edge detectors and wires of the graphical bodies
    _w1, _w2, _w3, _w4 : ANY;
END_VAR

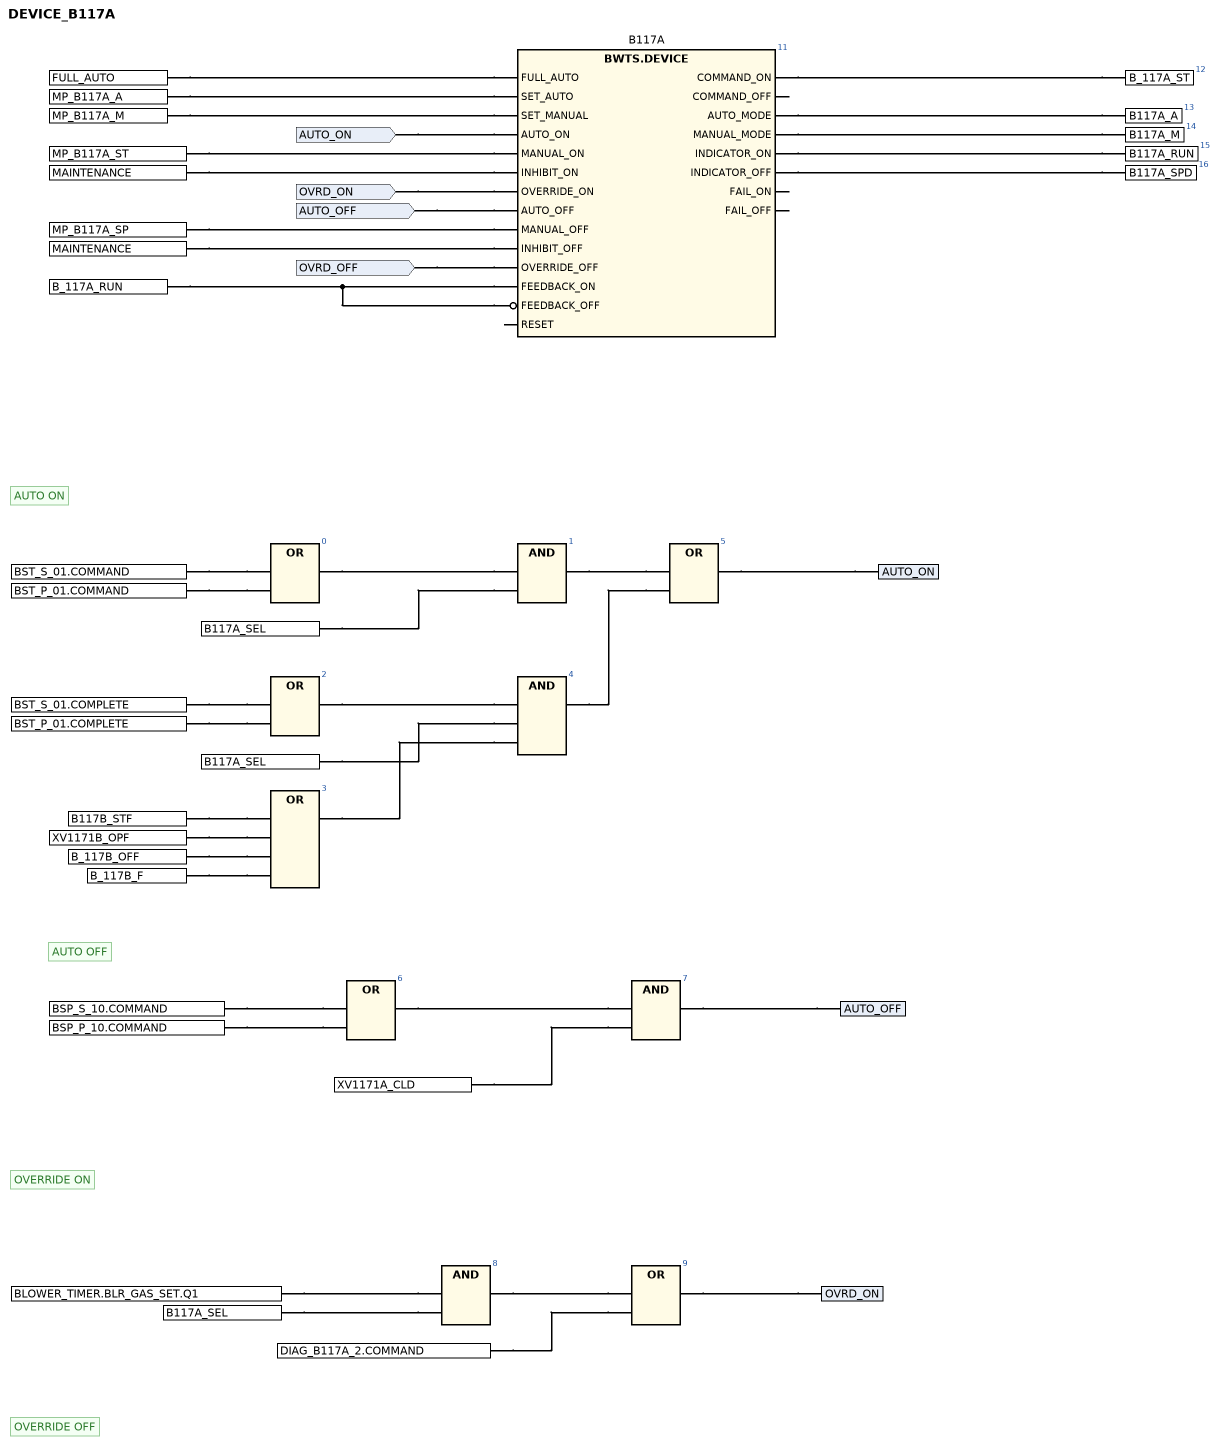
